// TIA Portal V20 export
// export: Created 2025-12-01T14:56:45.4401505Z, ExportSetting None, DisplayName Totally Integrated Automation Portal, DisplayVersion V20 Update 3, DisplayName TIA Portal Openness, DisplayVersion V20 Update 3, DisplayName TIA Portal Version Control Interface, DisplayVersion V20 Update 3, DisplayName STEP 7 Professional, DisplayVersion V20 Update 3, DisplayName STEP 7 Safety, DisplayVersion V20 Update 2, DisplayName WinCC Basic/Comfort/Advanced, DisplayVersion V20 Update 3, DisplayName WinCC Professional, DisplayVersion V20 Update 3, DisplayName WinCC Unified, DisplayVersion V20 Update 3
FUNCTION_BLOCK "FB262_M_FSS_Descarga"   // FB262, LAD
TITLE = Control del Ramal de Salidas
{ S7_Optimized_Access := 'FALSE' }
AUTHOR : TE_FSS
NAME : 20160509
VERSION : 3.3
// stored: AutoNumber false, SetENOAutomatically false
   VAR_INPUT
      Mesa : UInt;   // Mesa de la FB
      Error_Tx : Bool;   // Error en el Tx
      EnTension : Bool;   // Existe Tension en la Mesa
      Termico_T1 : Bool;   // Proteccion del T1
      Termico_T2 : Bool;   // Proteccion del T2
      Termico_T3 : Bool;   // Proteccion del T3
      Termico_T4 : Bool;   // Proteccion del T4
      pHsMx_1 : Bool;   // pHs 1 de la Mesa
      pHsMx_2 : Bool;   // pHs 2 de la Mesa
      pHsMx_3 : Bool;   // pHs 3 de la Mesa
      pHsMx_4 : Bool;   // pHs 4 de la Mesa
      Avance_T1 : Bool;   // Avance del T1
      Avance_T2 : Bool;   // Avance del T2
      Avance_T3 : Bool;   // Avance del T3
      Avance_T4 : Bool;   // Avance del T4
      Termico_TR1 : Bool;   // Proteccion del TR1
      Termico_TR2 : Bool;   // Proteccion del TR1
      Avance_TR1 : Bool;   // Avance del TR1
      Avance_TR2 : Bool;   // Avance del TR2
      TR1_Arriba : Bool;   // TR1 >> Arriba
      TR1_Abajo : Bool;   // TR1 >> Abajo
      TR1_EnMovimiento : Bool;   // TR1 >> En Movimiento
      TR2_Arriba : Bool;   // TR2 >> Arriba
      TR2_Abajo : Bool;   // TR2 >> Abajo
      TR2_EnMovimiento : Bool;   // TR2 >> En Movimiento
      TPE1_Arriba : Bool;   // TPE1 >> Arriba
      TPE1_Abajo : Bool;   // TPE1 >> Abajo
      TPE1_EnMovimiento : Bool;   // TPE1 >> En Movimiento
      TPE3_Arriba : Bool;   // TPE3 >> Arriba
      TPE3_Abajo : Bool;   // TPE3 >> Abajo
      TPE3_EnMovimiento : Bool;   // TPE3 >> En Movimiento
      MAnt_DescargaAct : Bool;   // E2 >> Mesa Anterior DescargaAct
      AVTF_MAnt_Mx_BGrande : Bool;   // E2 >> Mesa Anterior AVTF - Grande
      AVTF_MAnt_Mx_BPequena : Bool;   // E2 >> Mesa Anterior AVTF - Pequeña
      P_Mens_MAnt_Mx : Bool;   // E2 >> Mesa Anterior P_Mens
      E1_Arrival : Bool;   // E1 a FSS >> Arrival
      E1_Rotative : Bool;   // E1 a FSS >> Rotative
      E3_Arrival : Bool;   // E3 a FSS >> Arrival
      E3_Rotative : Bool;   // E3 a FSS >> Rotative
      PTF_Mx_MSig : Bool;   // S4 >> Mesa Siguiente PTF
      FTF_Mx_MSig : Bool;   // S4 >> Mesa Siguiente FTF
      MSig_CargaAct : Bool;
      F_EnvMens_Mx : Bool;   // Fin de Envio de Mensaje
      OrdSal_BGrande : Bool;   // Orden de Salida - Grande
      OrdSal_BPequena : Bool;   // Orden de Salida - Pequeña
      V_CNT_DesCargaFSS : Int := 1000;   // Valor de Posicionado FSS en la DesCarga
      V_CNT_PasarLentaFSS : Int := 100;
      V_CNT_pHsMx_E2 : Int := 100;   // Valor de Presencia
      V_CNT_pHsMx_FTF_E2 : Int := 250;   // Valor para activar FTF. Nota: < = V_CNT_pHsMx.
      V_CNTSeg_pHsMx_E2 : Int := 1000;   // Valor de Seguriadad para Presencia
      V_CNT_ApHsMx : Int := 200;   // Valor de Ausencia
      V_CNTSeg_ApHsMx : Int := 2000;   // Valor de Seguriadad para Ausencia
      V_CNT_Simultaneo : Int := 2000;   // Valor de Contador de Simultaneo
      V_TOut_Tx_Mx : Int := 7000;   // TImeOut de DesCarga del FSS
      V_TOut_TRx_Mx : Int := 7000;   // TimeOut de Entrada por E2
      V_TOut_TR : Int := 3000;   // TimeOut de Transfer
      V_TOut_TP : Int := 3000;   // TimeOut de Tope
      V_TOut_Interlock : Int := 5000;   // TimeOut de Interlock con el FSS
      V_CNT_PerdidapHs : Int := 1000;   // CNT de Perdida de pHs
      V_TIM_EstabilidadCarga : Time := T#100MS;   // Valor de Eastabilidad de Carga por DCC
      V_TIM_EsperaMesaLibre : Time;   // Valor de Espera para dar Mesa Libre
   END_VAR
   VAR_OUTPUT
      P_EnvMens_PMx : Bool;   // Permiso de Enviar Mensaje de Presencia
      P_RecepOK_Mx : Bool;   // Recepcion OK
      PTF_MAnt_Mx : Bool;   // E2 >> Mesa Anterior PTF
      FTF_MAnt_Mx : Bool;   // E2 >> Mesa Anterior FTF
      AVTF_Mx_Msig_BGrande : Bool;   // S4 >> Mesa Siguiente AVTF - Grande
      AVTF_Mx_MSig_BPequena : Bool;   // S4 >> Mesa Siguiente AVTF - Pequeña
      P_Mens_Mx_MSig : Bool;   // S4 >> Mesa Siguiente P_Mens
   END_VAR
   VAR
      Mx_ET00 : Bool;
      Mx_ET01 : Bool;
      Mx_ET02 : Bool;
      Mx_ET08_1PRE : Bool;
      Mx_ET08_1FIN : Bool;
      Mx_ET08_2PRE : Bool;
      Mx_ET08_2FIN : Bool;
      Mx_ET08_3PRE : Bool;
      Mx_ET08_3FIN : Bool;
      Mx_ET08_4PRE : Bool;
      Mx_ET08_4FIN : Bool;
      Mx_ET09 : Bool;
      Mx_ET10 : Bool;
      Mx_ET11 : Bool;
      Mx_ET12 : Bool;
      Mx_ET110_1PRE : Bool;
      Mx_ET110_1FIN : Bool;
      Mx_ET110_2PRE : Bool;
      Mx_ET110_2FIN : Bool;
      Mx_ET110_3PRE : Bool;
      Mx_ET110_3FIN : Bool;
      Mx_ET110_4PRE : Bool;
      Mx_ET110_4FIN : Bool;
      Mx_ET111 : Bool;
      Mx_ET20 : Bool;
      Mx_ET21 : Bool;
      Mx_ET22 : Bool;
      Mx_ET120 : Bool;
      Mx_ET121 : Bool;
      Mx_ET30 : Bool;
      Mx_ET31 : Bool;
      Mx_ET32 : Bool;
      Mx_ET130_1PRE : Bool;
      Mx_ET130_1FIN : Bool;
      Mx_ET130_2PRE : Bool;
      Mx_ET130_2FIN : Bool;
      Mx_ET130_3PRE : Bool;
      Mx_ET130_3FIN : Bool;
      Mx_ET130_4PRE : Bool;
      Mx_ET130_4FIN : Bool;
      Mx_ET131 : Bool;
      Mx_ET60 : Bool;
      Mx_ET61 : Bool;
      Mx_ET160 : Bool;
      Mx_ET161 : Bool;
      Mx_AutoArranque : Bool;   // Config >> Fin carga del FSS - Automatico
      Mx_NoEnvioPresEnFSS : Bool;   // Config >> No Envio de Presncia en la DesCarga del FSS
      FinDesCargaFSS_Auto : Bool;   // Intena >> AutoRearme Fin DesCarga del FSS
      Selec_E1 : Bool;   // Interna >> Selecionado Entrada por E1
      Selec_E2 : Bool;   // Interna >> Selecionado Entrada por E2
      Selec_E3 : Bool;   // Interna >> Selecionado Entrada por E3
      Selec_S4_BGrande : Bool;   // Interna >> Selecionado Salida por S4 - Grande
      Selec_S4_BPequena : Bool;   // Interna >> Selecionado Salida por S4 - Pequeña
      SaliendoCarga : Bool;   // Saliendo Carga de la Mesa
      Pos_TROK : Bool;   // Interna >> Posicion Correcta de los TRs
      Pos_TPOK : Bool;   // Interna >> Posicion Correcta de los TPs
      Entrando_BGrande : Bool;   // Interna >> Bandeja Grande en Entrada por E2
      PasarLenta_FSS : Bool;   // Interna >> Orden Pasar a Lenta la DesCarga FSS
      PosSalidaCarga_OK : Bool;   // Interna >> Posicionada la Carga para Salida
      ProtocoloIniciado : Bool;   // Iniciado el Envio del Mensaje de Presencia
      CNT_pHsMx_FTF_E2_OK : Bool;   // Enviar ya FTF
      Simultaneo_Mx : Bool;   // Activo Simultaneo E2
      STAT_EnvMens_PMx : Bool;   // Interna >> Envio del Mensaje de Presencia
      STAT_AVTF_MAnt_Mx : Bool;   // Interna >> Aviso de Entrada - Grande, Pequeña
      STAT_FTF_MAnt_Mx : Bool;   // Interna >> FTF de MAnt >> Mx
      STAT_AVTF_Mx_MSig : Bool;   // Interna >> AVTF de Mx >> MSig
      STAT_AvanceCarga_E1E3 : Bool;   // Interna >> Avance de Entrada de Carga por E1E3
      STAT_AvanceCarga_E2 : Bool;   // Interna >> Avance de Entrada de Carga por E2
      STAT_AvanceDescarga : Bool;   // Interna >> Avance de Salida de Carga
      STAT_Velocidad_TxBO : Bool;   // Interna >> Velocidad Bit 0 de los Rodillos
      STAT_Velocidad_TxB1 : Bool;   // Interna >> Velocidad Bit 1 de los Rodillos
      MA_Avance_T1 : Bool;
      MA_Avance_T2 : Bool;
      MA_Avance_T3 : Bool;
      MA_Avance_T4 : Bool;
      MA_Inversion_Tx : Bool;
      MA_VelocidadAnalogica : Int;
      MA_Avance_TR1 : Bool;
      MA_Avance_TR2 : Bool;
      MA_VelocidaLenta_TRx : Bool;
      MA_Subir_TR1 : Bool;
      MA_Bajar_TR1 : Bool;
      MA_Subir_TR2 : Bool;
      MA_Bajar_TR2 : Bool;
      MA_Subir_TPE1 : Bool;
      MA_Bajar_TPE1 : Bool;
      MA_Subir_TPE3 : Bool;
      MA_Bajar_TPE3 : Bool;
      MA_DepositOK_E1 : Bool;
      MA_Complete_E1 : Bool;
      MA_DepositOK_E3 : Bool;
      MA_Complete_E3 : Bool;
      TIM_EsperaMesaLibre { S7_SetPoint := 'True'} : TON_TIME;   // TIM De Espera para Dar la Mesa como Libre
      TIM_Estabilidad_E1 { S7_SetPoint := 'True'} : TON_TIME;   // TIM De Estabilidad de Carga en E1
      TIM_Estabilidad_E3 { S7_SetPoint := 'True'} : TON_TIME;   // TIM De Estabilidad de Carga en E3
      TIM_Estabilidad_E2 { S7_SetPoint := 'True'} : TON_TIME;   // TIM De Estabilidad de Carga en E2
      TIM_EstabilidadCarga { S7_SetPoint := 'True'} : TON_TIME;
      CNT_pHsMx_E1 { S7_SetPoint := 'True'} : "FB910_CNT_UHS";   // CNT de Presencia de FSS por E1
      CNT_pHsMx_E3 { S7_SetPoint := 'True'} : "FB910_CNT_UHS";   // CNT de Presencia de FSS por E3
      CNT_Reposiciona_E3 { S7_SetPoint := 'True'} : "FB910_CNT_UHS";   // CNT de Reposicionado de FSS por E3
      CNT_PasarLenta_FSS { S7_SetPoint := 'True'} : "FB910_CNT_UHS";   // CNT de Pasar a Lenta la DesCarga del FSS
      CNT_RecolocarCarga { S7_SetPoint := 'True'} : "FB910_CNT_UHS";   // CNT de Recolocar la Carga para la Salida
      CNT_pHsMx_E2 { S7_SetPoint := 'True'} : "FB910_CNT_UHS";   // CNT de la Presencia
      CNTSeg_pHsMx_E2 { S7_SetPoint := 'True'} : "FB910_CNT_UHS";   // CNT de Seguridad de la Presencia
      CNT_ApHsMx { S7_SetPoint := 'True'} : "FB910_CNT_UHS";   // CNT de la Ausencia
      CNTSeg_ApHsMx { S7_SetPoint := 'True'} : "FB910_CNT_UHS";   // CNT de Seguridad de la Ausencia
      CNT_Simultaneo { S7_SetPoint := 'True'} : "FB910_CNT_UHS";   // CNT de Simultaneo
      TMP_EnTension { S7_SetPoint := 'True'} : "FB910_CNT_UHS";
      TOut_Av_Tx { S7_SetPoint := 'True'} : "FB910_CNT_UHS";   // Time Out de Entrada de E1
      TOut_Rt_Tx { S7_SetPoint := 'True'} : "FB910_CNT_UHS";   // Time Out de Entrada de E3
      TOut_Av_TRx { S7_SetPoint := 'True'} : "FB910_CNT_UHS";   // Time Out de Entrada de E2
      TOut_Subir_TR { S7_SetPoint := 'True'} : "FB910_CNT_UHS";   // Time Out de Subida del TR
      TOut_Bajar_TR { S7_SetPoint := 'True'} : "FB910_CNT_UHS";   // Time Out de Bajada del TR
      TOut_Subir_TP_E1E3 { S7_SetPoint := 'True'} : "FB910_CNT_UHS";   // Time Out de Subida del TP >> E1E3
      TOut_Bajar_TP_E1E3 { S7_SetPoint := 'True'} : "FB910_CNT_UHS";   // Time Out de Bajada del TP >> E1E3
      TOut_Interlock { S7_SetPoint := 'True'} : "FB910_CNT_UHS";   // Time Out de Interlock con el FSS
      Interlock_manual { S7_SetPoint := 'True'} : "UDT_Interlock_manual_TE_FSS";
      Manual : "MoviManualMesa_FSS";
      CNT_PerdidapHs { S7_SetPoint := 'True'} : "FB910_CNT_UHS";   // CNT de Perdida de pHs
   END_VAR
   VAR_TEMP
      EstadoZona : "EstadoZona";   // Estado de Zona de la Mesa
      EstadoVI : "EstadosMesa_FSS";   // Estado del Vehiculo Inteliguente de la Mesa
      ConfigFB : "UDT_ConfigFB";   // Configuracion de la FB de la Mesa
      Interlock : "UDT_Interlock_TE_FSS";
      retval : Int;
      cero : USInt;
      Aux_ET00 : Bool;
      EvolucionEtapasEntrada : Bool;
      EvolucionEtapasSalida : Bool;
   END_VAR
   VAR_TEMP   // added for the SCL form of the ladder/FBD networks
      _w1 : Bool;
   END_VAR
BEGIN

REGION Network 1: CONFIGURACION ESPECIAL DE LA FB
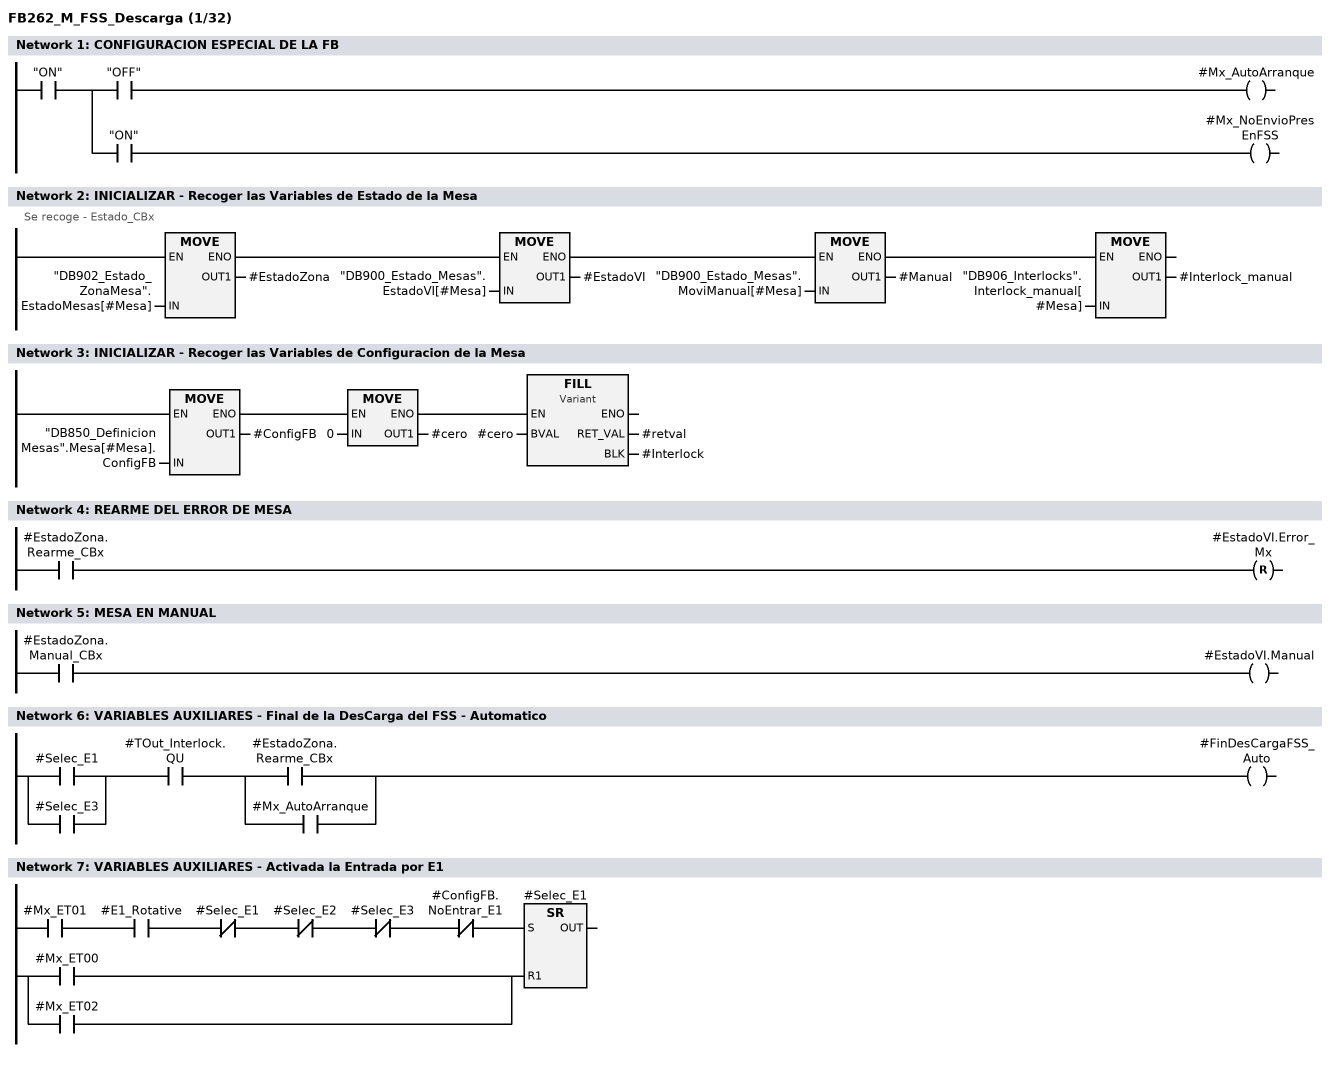
   RUNG wire#powerrail
      Contact( "ON" )
      wire#w1
      Contact( "OFF" )
      Coil( #Mx_AutoArranque )
   END_RUNG
   RUNG wire#w1
      Contact( "ON" )
      Coil( #Mx_NoEnvioPresEnFSS )
   END_RUNG
   // the same network as SCL:
   #Mx_AutoArranque := "ON" AND "OFF";
   #Mx_NoEnvioPresEnFSS := "ON" AND "ON";
END_REGION

REGION Network 2: INICIALIZAR - Recoger las Variables de Estado de la Mesa
   // Se recoge - Estado_CBx
   RUNG wire#powerrail
      Move(in := "DB902_Estado_ZonaMesa".EstadoMesas[#Mesa], out1 => #EstadoZona)
      Move(in := "DB900_Estado_Mesas".EstadoVI[#Mesa], out1 => #EstadoVI)
      Move(in := "DB900_Estado_Mesas".MoviManual[#Mesa], out1 => #Manual)
      Move(in := "DB906_Interlocks".Interlock_manual[#Mesa], out1 => #Interlock_manual)
   END_RUNG
   // the same network as SCL:
   #EstadoZona := "DB902_Estado_ZonaMesa".EstadoMesas[#Mesa];
   #EstadoVI := "DB900_Estado_Mesas".EstadoVI[#Mesa];
   #Manual := "DB900_Estado_Mesas".MoviManual[#Mesa];
   #Interlock_manual := "DB906_Interlocks".Interlock_manual[#Mesa];
END_REGION

REGION Network 3: INICIALIZAR - Recoger las Variables de Configuracion de la Mesa
   RUNG wire#powerrail
      Move(in := "DB850_DefinicionMesas".Mesa[#Mesa].ConfigFB, out1 => #ConfigFB)
      Move(in := 0, out1 => #cero)
      { S7_Templates := "ptr_type := Variant" } FILL(BVAL := #cero, RET_VAL => #retval, BLK => #Interlock)
   END_RUNG
   // the same network as SCL:
   #ConfigFB := "DB850_DefinicionMesas".Mesa[#Mesa].ConfigFB;
   #cero := 0;
   #retval := FILL(BVAL := #cero, BLK => #Interlock);
END_REGION

REGION Network 4: REARME DEL ERROR DE MESA
   RUNG wire#powerrail
      Contact( #EstadoZona.Rearme_CBx )
      R_Coil( #EstadoVI.Error_Mx )
   END_RUNG
   // the same network as SCL:
   IF #EstadoZona.Rearme_CBx THEN #EstadoVI.Error_Mx := FALSE; END_IF;
END_REGION

REGION Network 5: MESA EN MANUAL
   RUNG wire#powerrail
      Contact( #EstadoZona.Manual_CBx )
      Coil( #EstadoVI.Manual )
   END_RUNG
   // the same network as SCL:
   #EstadoVI.Manual := #EstadoZona.Manual_CBx;
END_REGION

REGION Network 6: VARIABLES AUXILIARES - Final de la DesCarga del FSS - Automatico
   RUNG wire#powerrail
      Contact( #Selec_E1 )
      wire#w1
      Contact( #TOut_Interlock.QU )
      wire#w2
      Contact( #EstadoZona.Rearme_CBx )
      wire#w3
      Coil( #FinDesCargaFSS_Auto )
   END_RUNG
   RUNG wire#powerrail
      Contact( #Selec_E3 )
   END_RUNG wire#w1
   RUNG wire#w2
      Contact( #Mx_AutoArranque )
   END_RUNG wire#w3
   // the same network as SCL:
   #FinDesCargaFSS_Auto := (#Selec_E1 OR #Selec_E3) AND #TOut_Interlock.QU AND (#EstadoZona.Rearme_CBx OR #Mx_AutoArranque);
END_REGION

REGION Network 7: VARIABLES AUXILIARES - Activada la Entrada por E1
   RUNG wire#powerrail
      Contact( #Mx_ET01 )
      Contact( #E1_Rotative )
      I_Contact( #Selec_E1 )
      I_Contact( #Selec_E2 )
      I_Contact( #Selec_E3 )
      I_Contact( #ConfigFB.NoEntrar_E1 )
      S_SR(operand := #Selec_E1, r1 := wire#w1)
   END_RUNG
   RUNG wire#powerrail
      Contact( #Mx_ET00 )
   END_RUNG wire#w1
   RUNG wire#powerrail
      Contact( #Mx_ET02 )
   END_RUNG wire#w1
   // the same network as SCL:
   IF #Mx_ET01 AND #E1_Rotative AND NOT #Selec_E1 AND NOT #Selec_E2 AND NOT #Selec_E3 AND NOT #ConfigFB.NoEntrar_E1 THEN
       #Selec_E1 := TRUE;   // SR flip-flop
   END_IF;
   IF #Mx_ET00 OR #Mx_ET02 THEN #Selec_E1 := FALSE; END_IF;
END_REGION

REGION Network 8: VARIABLES AUXILIARES - Activada la Entrada por E2
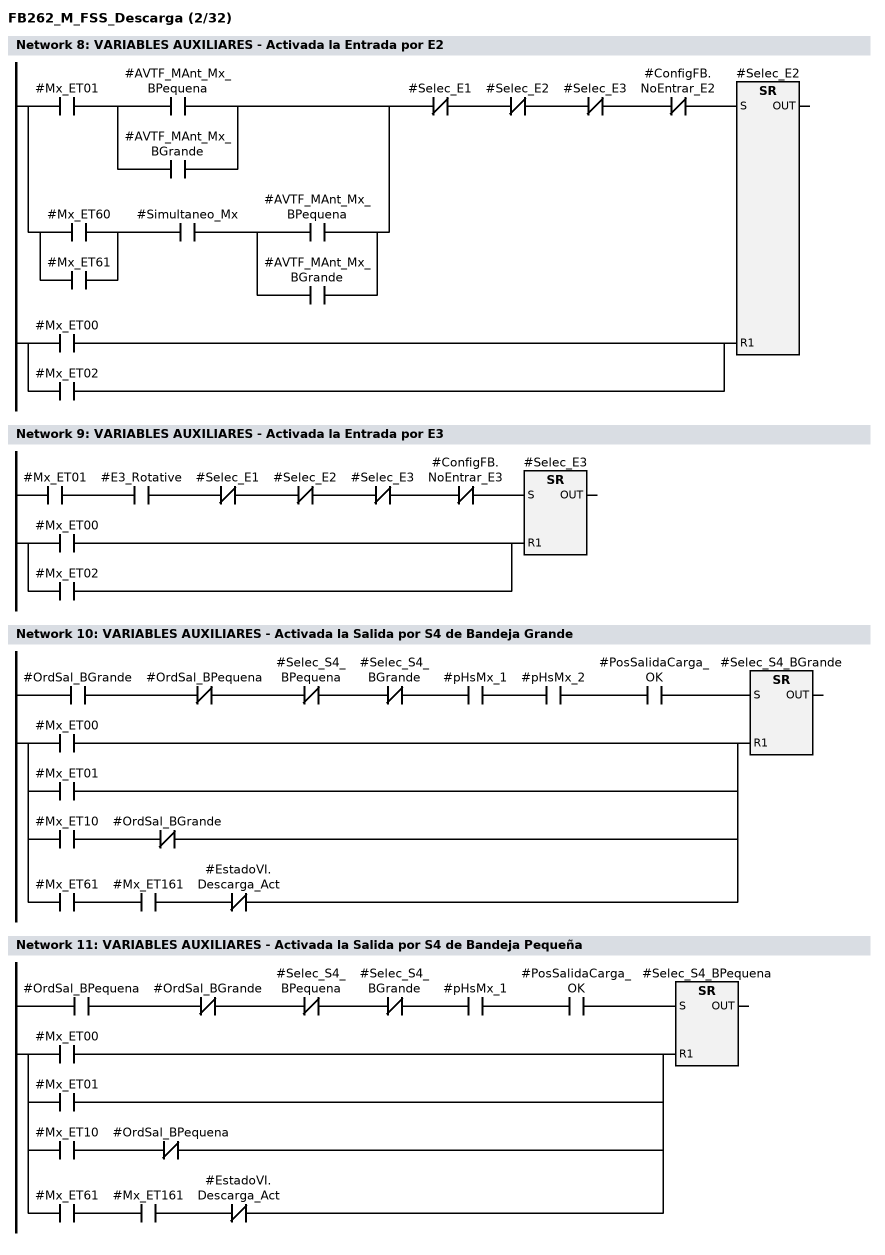
   RUNG wire#powerrail
      Contact( #Mx_ET01 )
      wire#w1
      Contact( #AVTF_MAnt_Mx_BPequena )
      wire#w2
      I_Contact( #Selec_E1 )
      I_Contact( #Selec_E2 )
      I_Contact( #Selec_E3 )
      I_Contact( #ConfigFB.NoEntrar_E2 )
      S_SR(operand := #Selec_E2, r1 := wire#w5)
   END_RUNG
   RUNG wire#w1
      Contact( #AVTF_MAnt_Mx_BGrande )
   END_RUNG wire#w2
   RUNG wire#powerrail
      Contact( #Mx_ET60 )
      wire#w3
      Contact( #Simultaneo_Mx )
      wire#w4
      Contact( #AVTF_MAnt_Mx_BPequena )
   END_RUNG wire#w2
   RUNG wire#powerrail
      Contact( #Mx_ET61 )
   END_RUNG wire#w3
   RUNG wire#w4
      Contact( #AVTF_MAnt_Mx_BGrande )
   END_RUNG wire#w2
   RUNG wire#powerrail
      Contact( #Mx_ET00 )
   END_RUNG wire#w5
   RUNG wire#powerrail
      Contact( #Mx_ET02 )
   END_RUNG wire#w5
   // the same network as SCL:
   IF ((#Mx_ET01 AND (#AVTF_MAnt_Mx_BPequena OR #AVTF_MAnt_Mx_BGrande)) OR ((#Mx_ET60 OR #Mx_ET61) AND #Simultaneo_Mx AND (#AVTF_MAnt_Mx_BPequena OR #AVTF_MAnt_Mx_BGrande))) AND NOT #Selec_E1 AND NOT #Selec_E2 AND NOT #Selec_E3 AND NOT #ConfigFB.NoEntrar_E2 THEN
       #Selec_E2 := TRUE;   // SR flip-flop
   END_IF;
   IF #Mx_ET00 OR #Mx_ET02 THEN #Selec_E2 := FALSE; END_IF;
END_REGION

REGION Network 9: VARIABLES AUXILIARES - Activada la Entrada por E3
   RUNG wire#powerrail
      Contact( #Mx_ET01 )
      Contact( #E3_Rotative )
      I_Contact( #Selec_E1 )
      I_Contact( #Selec_E2 )
      I_Contact( #Selec_E3 )
      I_Contact( #ConfigFB.NoEntrar_E3 )
      S_SR(operand := #Selec_E3, r1 := wire#w1)
   END_RUNG
   RUNG wire#powerrail
      Contact( #Mx_ET00 )
   END_RUNG wire#w1
   RUNG wire#powerrail
      Contact( #Mx_ET02 )
   END_RUNG wire#w1
   // the same network as SCL:
   IF #Mx_ET01 AND #E3_Rotative AND NOT #Selec_E1 AND NOT #Selec_E2 AND NOT #Selec_E3 AND NOT #ConfigFB.NoEntrar_E3 THEN
       #Selec_E3 := TRUE;   // SR flip-flop
   END_IF;
   IF #Mx_ET00 OR #Mx_ET02 THEN #Selec_E3 := FALSE; END_IF;
END_REGION

REGION Network 10: VARIABLES AUXILIARES - Activada la Salida por S4 de Bandeja Grande
   RUNG wire#powerrail
      Contact( #OrdSal_BGrande )
      I_Contact( #OrdSal_BPequena )
      I_Contact( #Selec_S4_BPequena )
      I_Contact( #Selec_S4_BGrande )
      Contact( #pHsMx_1 )
      Contact( #pHsMx_2 )
      Contact( #PosSalidaCarga_OK )
      S_SR(operand := #Selec_S4_BGrande, r1 := wire#w1)
   END_RUNG
   RUNG wire#powerrail
      Contact( #Mx_ET00 )
   END_RUNG wire#w1
   RUNG wire#powerrail
      Contact( #Mx_ET01 )
   END_RUNG wire#w1
   RUNG wire#powerrail
      Contact( #Mx_ET10 )
      I_Contact( #OrdSal_BGrande )
   END_RUNG wire#w1
   RUNG wire#powerrail
      Contact( #Mx_ET61 )
      Contact( #Mx_ET161 )
      I_Contact( #EstadoVI.Descarga_Act )
   END_RUNG wire#w1
   // the same network as SCL:
   IF #OrdSal_BGrande AND NOT #OrdSal_BPequena AND NOT #Selec_S4_BPequena AND NOT #Selec_S4_BGrande AND #pHsMx_1 AND #pHsMx_2 AND #PosSalidaCarga_OK THEN
       #Selec_S4_BGrande := TRUE;   // SR flip-flop
   END_IF;
   IF #Mx_ET00 OR #Mx_ET01 OR (#Mx_ET10 AND NOT #OrdSal_BGrande) OR (#Mx_ET61 AND #Mx_ET161 AND NOT #EstadoVI.Descarga_Act) THEN
       #Selec_S4_BGrande := FALSE;
   END_IF;
END_REGION

REGION Network 11: VARIABLES AUXILIARES - Activada la Salida por S4 de Bandeja Pequeña
   RUNG wire#powerrail
      Contact( #OrdSal_BPequena )
      I_Contact( #OrdSal_BGrande )
      I_Contact( #Selec_S4_BPequena )
      I_Contact( #Selec_S4_BGrande )
      Contact( #pHsMx_1 )
      Contact( #PosSalidaCarga_OK )
      S_SR(operand := #Selec_S4_BPequena, r1 := wire#w1)
   END_RUNG
   RUNG wire#powerrail
      Contact( #Mx_ET00 )
   END_RUNG wire#w1
   RUNG wire#powerrail
      Contact( #Mx_ET01 )
   END_RUNG wire#w1
   RUNG wire#powerrail
      Contact( #Mx_ET10 )
      I_Contact( #OrdSal_BPequena )
   END_RUNG wire#w1
   RUNG wire#powerrail
      Contact( #Mx_ET61 )
      Contact( #Mx_ET161 )
      I_Contact( #EstadoVI.Descarga_Act )
   END_RUNG wire#w1
   // the same network as SCL:
   IF #OrdSal_BPequena AND NOT #OrdSal_BGrande AND NOT #Selec_S4_BPequena AND NOT #Selec_S4_BGrande AND #pHsMx_1 AND #PosSalidaCarga_OK THEN
       #Selec_S4_BPequena := TRUE;   // SR flip-flop
   END_IF;
   IF #Mx_ET00 OR #Mx_ET01 OR (#Mx_ET10 AND NOT #OrdSal_BPequena) OR (#Mx_ET61 AND #Mx_ET161 AND NOT #EstadoVI.Descarga_Act) THEN
       #Selec_S4_BPequena := FALSE;
   END_IF;
END_REGION

REGION Network 12: VARIABLES AUXILIARES - Saliendo Carga de la Mesa
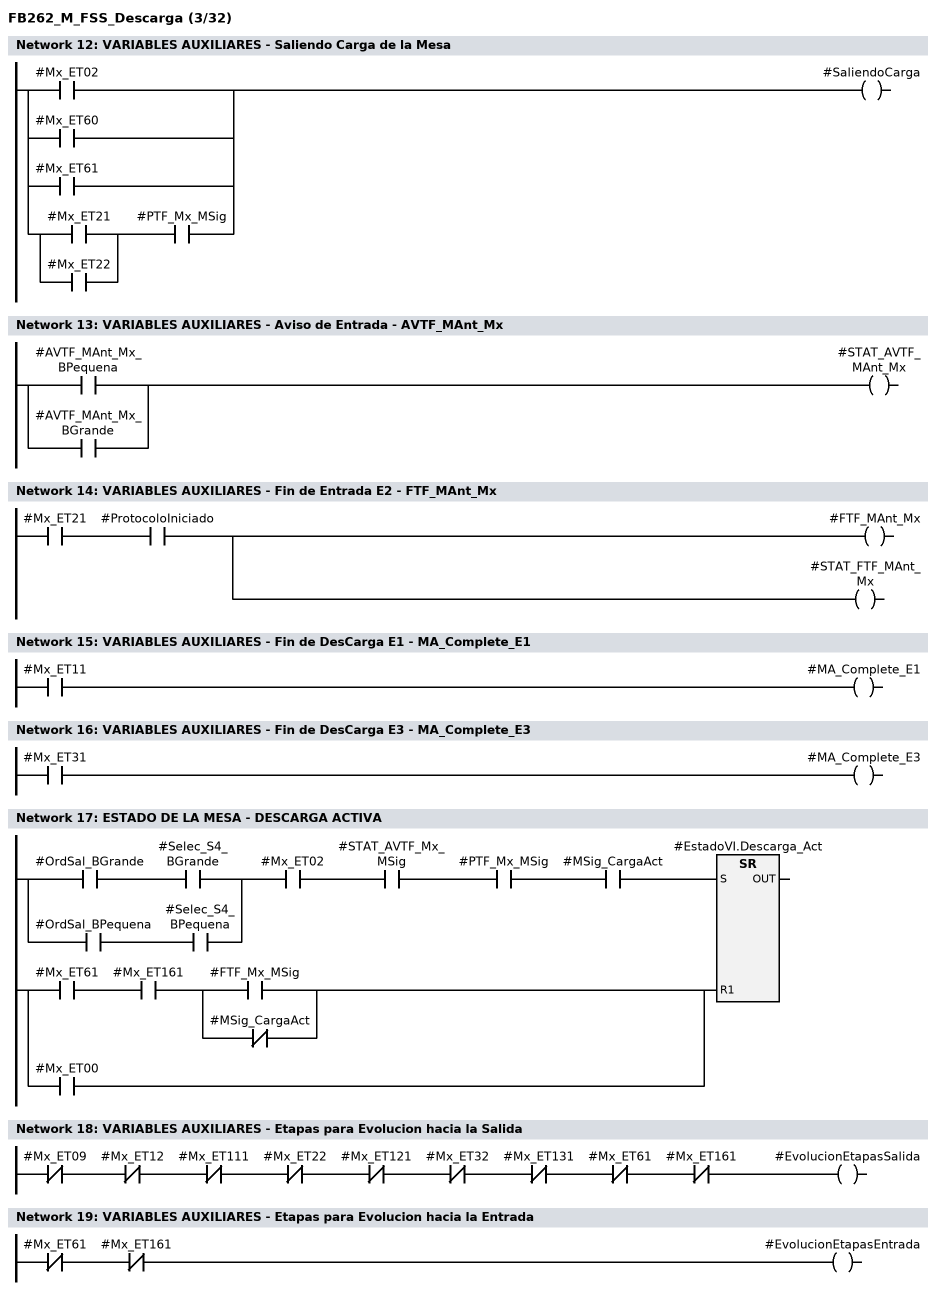
   RUNG wire#powerrail
      Contact( #Mx_ET02 )
      wire#w1
      Coil( #SaliendoCarga )
   END_RUNG
   RUNG wire#powerrail
      Contact( #Mx_ET60 )
   END_RUNG wire#w1
   RUNG wire#powerrail
      Contact( #Mx_ET61 )
   END_RUNG wire#w1
   RUNG wire#powerrail
      Contact( #Mx_ET21 )
      wire#w2
      Contact( #PTF_Mx_MSig )
   END_RUNG wire#w1
   RUNG wire#powerrail
      Contact( #Mx_ET22 )
   END_RUNG wire#w2
   // the same network as SCL:
   #SaliendoCarga := #Mx_ET02 OR #Mx_ET60 OR #Mx_ET61 OR ((#Mx_ET21 OR #Mx_ET22) AND #PTF_Mx_MSig);
END_REGION

REGION Network 13: VARIABLES AUXILIARES - Aviso de Entrada - AVTF_MAnt_Mx
   RUNG wire#powerrail
      Contact( #AVTF_MAnt_Mx_BPequena )
      wire#w1
      Coil( #STAT_AVTF_MAnt_Mx )
   END_RUNG
   RUNG wire#powerrail
      Contact( #AVTF_MAnt_Mx_BGrande )
   END_RUNG wire#w1
   // the same network as SCL:
   #STAT_AVTF_MAnt_Mx := #AVTF_MAnt_Mx_BPequena OR #AVTF_MAnt_Mx_BGrande;
END_REGION

REGION Network 14: VARIABLES AUXILIARES - Fin de Entrada E2 - FTF_MAnt_Mx
   RUNG wire#powerrail
      Contact( #Mx_ET21 )
      Contact( #ProtocoloIniciado )
      wire#w1
      Coil( #FTF_MAnt_Mx )
   END_RUNG
   RUNG wire#w1
      Coil( #STAT_FTF_MAnt_Mx )
   END_RUNG
   // the same network as SCL:
   #FTF_MAnt_Mx := #Mx_ET21 AND #ProtocoloIniciado;
   #STAT_FTF_MAnt_Mx := #FTF_MAnt_Mx;
END_REGION

REGION Network 15: VARIABLES AUXILIARES - Fin de DesCarga E1 - MA_Complete_E1
   RUNG wire#powerrail
      Contact( #Mx_ET11 )
      Coil( #MA_Complete_E1 )
   END_RUNG
   // the same network as SCL:
   #MA_Complete_E1 := #Mx_ET11;
END_REGION

REGION Network 16: VARIABLES AUXILIARES - Fin de DesCarga E3 - MA_Complete_E3
   RUNG wire#powerrail
      Contact( #Mx_ET31 )
      Coil( #MA_Complete_E3 )
   END_RUNG
   // the same network as SCL:
   #MA_Complete_E3 := #Mx_ET31;
END_REGION

REGION Network 17: ESTADO DE LA MESA - DESCARGA ACTIVA
   RUNG wire#powerrail
      Contact( #OrdSal_BGrande )
      Contact( #Selec_S4_BGrande )
      wire#w1
      Contact( #Mx_ET02 )
      Contact( #STAT_AVTF_Mx_MSig )
      Contact( #PTF_Mx_MSig )
      Contact( #MSig_CargaAct )
      S_SR(operand := #EstadoVI.Descarga_Act, r1 := wire#w3)
   END_RUNG
   RUNG wire#powerrail
      Contact( #OrdSal_BPequena )
      Contact( #Selec_S4_BPequena )
   END_RUNG wire#w1
   RUNG wire#powerrail
      Contact( #Mx_ET61 )
      Contact( #Mx_ET161 )
      wire#w2
      Contact( #FTF_Mx_MSig )
   END_RUNG wire#w3
   RUNG wire#w2
      I_Contact( #MSig_CargaAct )
   END_RUNG wire#w3
   RUNG wire#powerrail
      Contact( #Mx_ET00 )
   END_RUNG wire#w3
   // the same network as SCL:
   IF ((#OrdSal_BGrande AND #Selec_S4_BGrande) OR (#OrdSal_BPequena AND #Selec_S4_BPequena)) AND #Mx_ET02 AND #STAT_AVTF_Mx_MSig AND #PTF_Mx_MSig AND #MSig_CargaAct THEN
       #EstadoVI.Descarga_Act := TRUE;   // SR flip-flop
   END_IF;
   IF (#Mx_ET61 AND #Mx_ET161 AND (#FTF_Mx_MSig OR NOT #MSig_CargaAct)) OR #Mx_ET00 THEN
       #EstadoVI.Descarga_Act := FALSE;
   END_IF;
END_REGION

REGION Network 18: VARIABLES AUXILIARES - Etapas para Evolucion hacia la Salida
   RUNG wire#powerrail
      I_Contact( #Mx_ET09 )
      I_Contact( #Mx_ET12 )
      I_Contact( #Mx_ET111 )
      I_Contact( #Mx_ET22 )
      I_Contact( #Mx_ET121 )
      I_Contact( #Mx_ET32 )
      I_Contact( #Mx_ET131 )
      I_Contact( #Mx_ET61 )
      I_Contact( #Mx_ET161 )
      Coil( #EvolucionEtapasSalida )
   END_RUNG
   // the same network as SCL:
   #EvolucionEtapasSalida := NOT #Mx_ET09 AND NOT #Mx_ET12 AND NOT #Mx_ET111 AND NOT #Mx_ET22 AND NOT #Mx_ET121 AND NOT #Mx_ET32 AND NOT #Mx_ET131 AND NOT #Mx_ET61 AND NOT #Mx_ET161;
END_REGION

REGION Network 19: VARIABLES AUXILIARES - Etapas para Evolucion hacia la Entrada
   RUNG wire#powerrail
      I_Contact( #Mx_ET61 )
      I_Contact( #Mx_ET161 )
      Coil( #EvolucionEtapasEntrada )
   END_RUNG
   // the same network as SCL:
   #EvolucionEtapasEntrada := NOT #Mx_ET61 AND NOT #Mx_ET161;
END_REGION

REGION Network 20: ET161 - CONTROL DESCARGA MESA - PROTOCOLO ORDEN
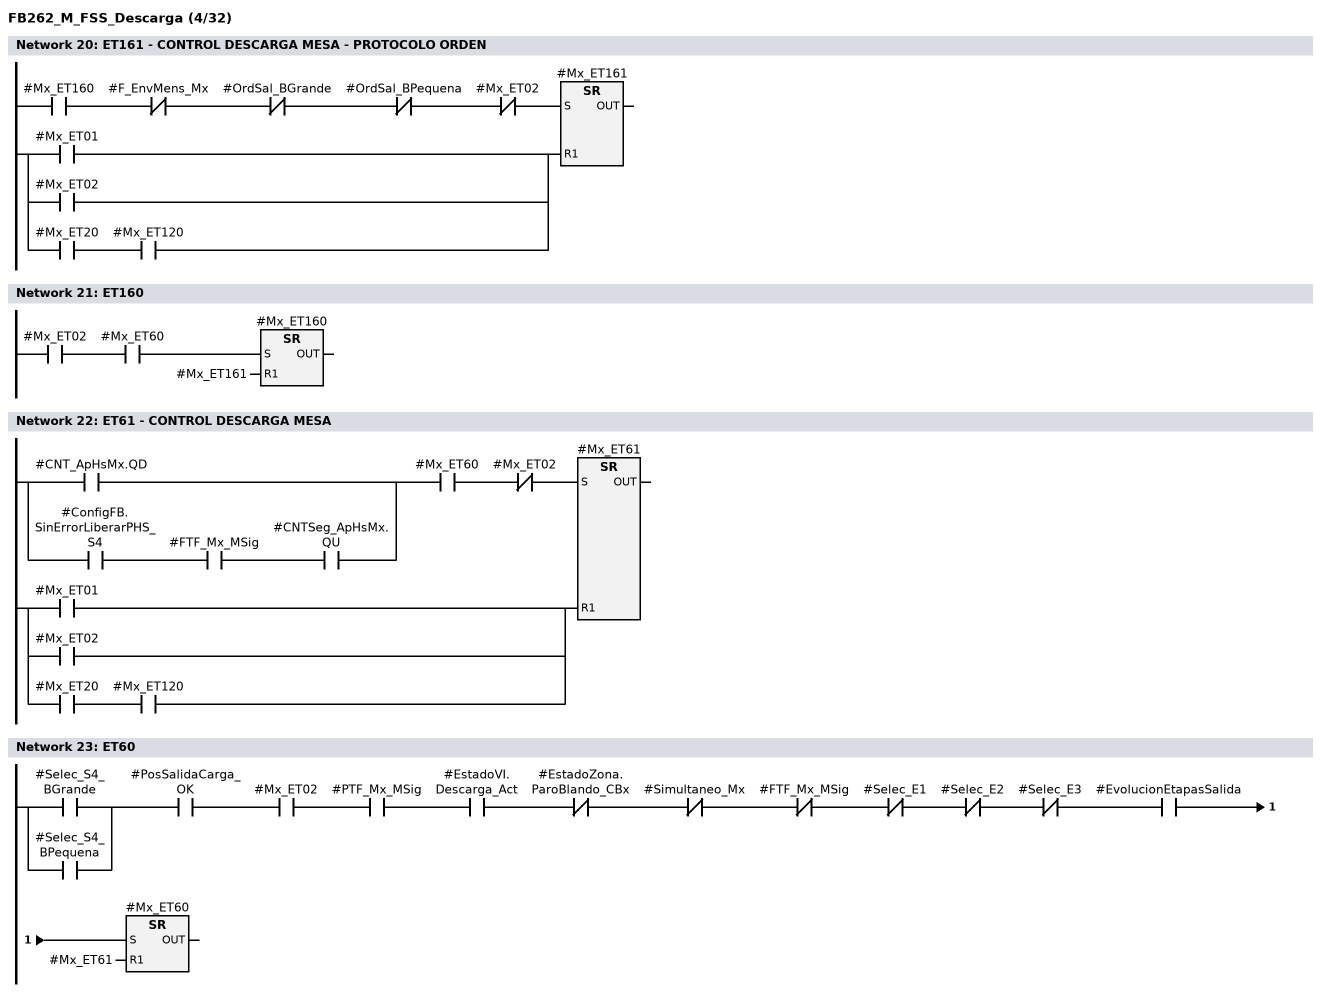
   RUNG wire#powerrail
      Contact( #Mx_ET160 )
      I_Contact( #F_EnvMens_Mx )
      I_Contact( #OrdSal_BGrande )
      I_Contact( #OrdSal_BPequena )
      I_Contact( #Mx_ET02 )
      S_SR(operand := #Mx_ET161, r1 := wire#w1)
   END_RUNG
   RUNG wire#powerrail
      Contact( #Mx_ET01 )
   END_RUNG wire#w1
   RUNG wire#powerrail
      Contact( #Mx_ET02 )
   END_RUNG wire#w1
   RUNG wire#powerrail
      Contact( #Mx_ET20 )
      Contact( #Mx_ET120 )
   END_RUNG wire#w1
   // the same network as SCL:
   IF #Mx_ET160 AND NOT #F_EnvMens_Mx AND NOT #OrdSal_BGrande AND NOT #OrdSal_BPequena AND NOT #Mx_ET02 THEN
       #Mx_ET161 := TRUE;   // SR flip-flop
   END_IF;
   IF #Mx_ET01 OR #Mx_ET02 OR (#Mx_ET20 AND #Mx_ET120) THEN #Mx_ET161 := FALSE; END_IF;
END_REGION

REGION Network 21: ET160
   RUNG wire#powerrail
      Contact( #Mx_ET02 )
      Contact( #Mx_ET60 )
      S_SR(operand := #Mx_ET160, r1 := #Mx_ET161)
   END_RUNG
   // the same network as SCL:
   IF #Mx_ET02 AND #Mx_ET60 THEN
       #Mx_ET160 := TRUE;   // SR flip-flop
   END_IF;
   IF #Mx_ET161 THEN #Mx_ET160 := FALSE; END_IF;
END_REGION

REGION Network 22: ET61 - CONTROL DESCARGA MESA
   RUNG wire#powerrail
      Contact( #CNT_ApHsMx.QD )
      wire#w1
      Contact( #Mx_ET60 )
      I_Contact( #Mx_ET02 )
      S_SR(operand := #Mx_ET61, r1 := wire#w2)
   END_RUNG
   RUNG wire#powerrail
      Contact( #ConfigFB.SinErrorLiberarPHS_S4 )
      Contact( #FTF_Mx_MSig )
      Contact( #CNTSeg_ApHsMx.QU )
   END_RUNG wire#w1
   RUNG wire#powerrail
      Contact( #Mx_ET01 )
   END_RUNG wire#w2
   RUNG wire#powerrail
      Contact( #Mx_ET02 )
   END_RUNG wire#w2
   RUNG wire#powerrail
      Contact( #Mx_ET20 )
      Contact( #Mx_ET120 )
   END_RUNG wire#w2
   // the same network as SCL:
   IF (#CNT_ApHsMx.QD OR (#ConfigFB.SinErrorLiberarPHS_S4 AND #FTF_Mx_MSig AND #CNTSeg_ApHsMx.QU)) AND #Mx_ET60 AND NOT #Mx_ET02 THEN
       #Mx_ET61 := TRUE;   // SR flip-flop
   END_IF;
   IF #Mx_ET01 OR #Mx_ET02 OR (#Mx_ET20 AND #Mx_ET120) THEN #Mx_ET61 := FALSE; END_IF;
END_REGION

REGION Network 23: ET60
   RUNG wire#powerrail
      Contact( #Selec_S4_BGrande )
      wire#w1
      Contact( #PosSalidaCarga_OK )
      Contact( #Mx_ET02 )
      Contact( #PTF_Mx_MSig )
      Contact( #EstadoVI.Descarga_Act )
      I_Contact( #EstadoZona.ParoBlando_CBx )
      I_Contact( #Simultaneo_Mx )
      I_Contact( #FTF_Mx_MSig )
      I_Contact( #Selec_E1 )
      I_Contact( #Selec_E2 )
      I_Contact( #Selec_E3 )
      Contact( #EvolucionEtapasSalida )
      S_SR(operand := #Mx_ET60, r1 := #Mx_ET61)
   END_RUNG
   RUNG wire#powerrail
      Contact( #Selec_S4_BPequena )
   END_RUNG wire#w1
   // the same network as SCL:
   IF (#Selec_S4_BGrande OR #Selec_S4_BPequena) AND #PosSalidaCarga_OK AND #Mx_ET02 AND #PTF_Mx_MSig AND #EstadoVI.Descarga_Act AND NOT #EstadoZona.ParoBlando_CBx AND NOT #Simultaneo_Mx AND NOT #FTF_Mx_MSig AND NOT #Selec_E1 AND NOT #Selec_E2 AND NOT #Selec_E3 AND #EvolucionEtapasSalida THEN
       #Mx_ET60 := TRUE;   // SR flip-flop
   END_IF;
   IF #Mx_ET61 THEN #Mx_ET60 := FALSE; END_IF;
END_REGION

REGION Network 24: ET02 - ESTADO REPOSO CARGADA
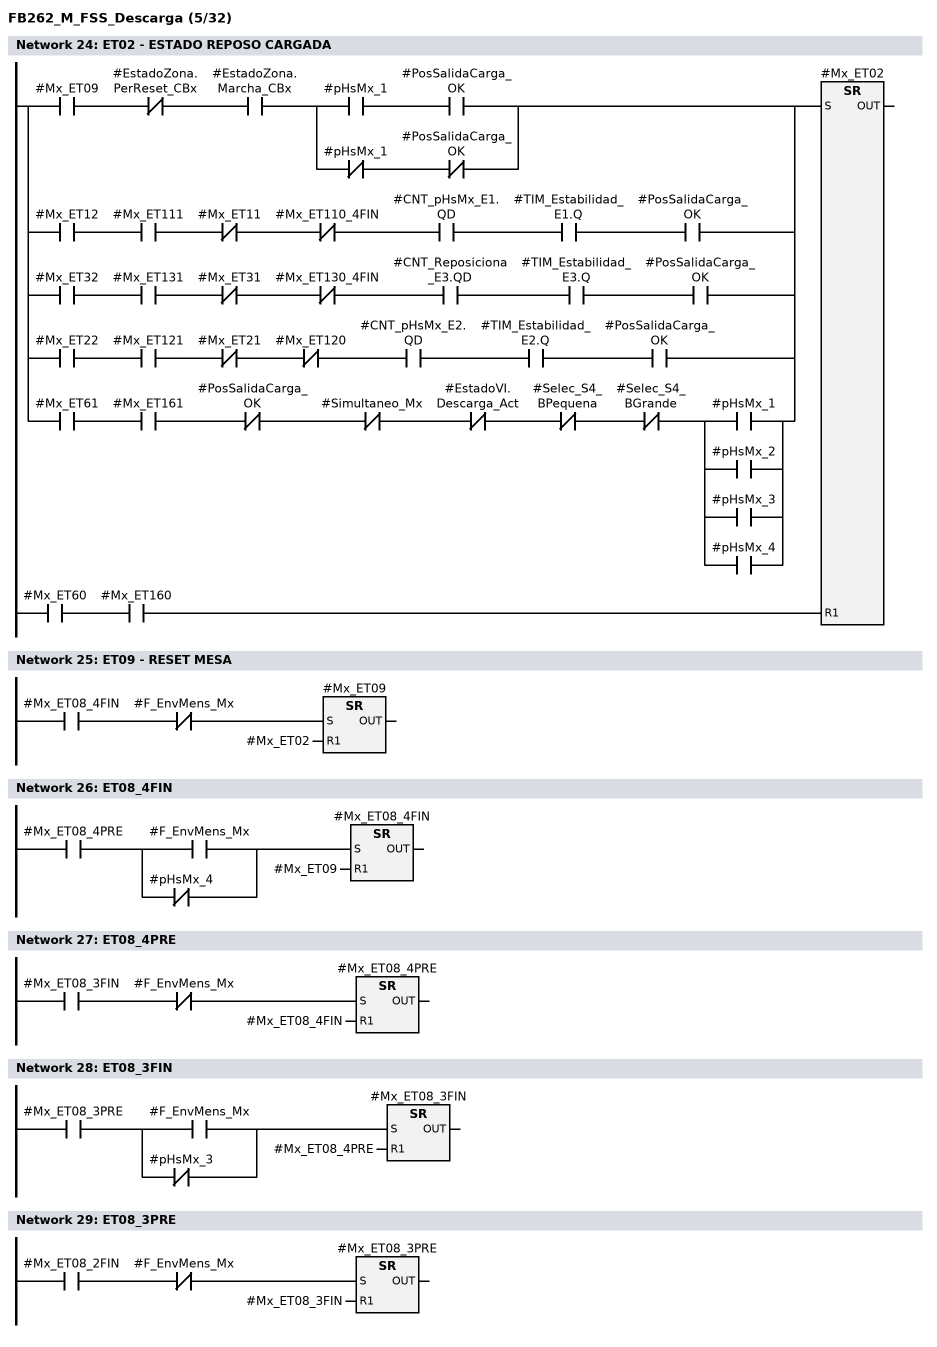
   RUNG wire#powerrail
      Contact( #Mx_ET09 )
      I_Contact( #EstadoZona.PerReset_CBx )
      Contact( #EstadoZona.Marcha_CBx )
      wire#w1
      Contact( #pHsMx_1 )
      Contact( #PosSalidaCarga_OK )
      wire#w2
      S_SR(operand := #Mx_ET02, r1 := wire#w4)
   END_RUNG
   RUNG wire#w1
      I_Contact( #pHsMx_1 )
      I_Contact( #PosSalidaCarga_OK )
   END_RUNG wire#w2
   RUNG wire#powerrail
      Contact( #Mx_ET12 )
      Contact( #Mx_ET111 )
      I_Contact( #Mx_ET11 )
      I_Contact( #Mx_ET110_4FIN )
      Contact( #CNT_pHsMx_E1.QD )
      Contact( #TIM_Estabilidad_E1.Q )
      Contact( #PosSalidaCarga_OK )
   END_RUNG wire#w2
   RUNG wire#powerrail
      Contact( #Mx_ET32 )
      Contact( #Mx_ET131 )
      I_Contact( #Mx_ET31 )
      I_Contact( #Mx_ET130_4FIN )
      Contact( #CNT_Reposiciona_E3.QD )
      Contact( #TIM_Estabilidad_E3.Q )
      Contact( #PosSalidaCarga_OK )
   END_RUNG wire#w2
   RUNG wire#powerrail
      Contact( #Mx_ET22 )
      Contact( #Mx_ET121 )
      I_Contact( #Mx_ET21 )
      I_Contact( #Mx_ET120 )
      Contact( #CNT_pHsMx_E2.QD )
      Contact( #TIM_Estabilidad_E2.Q )
      Contact( #PosSalidaCarga_OK )
   END_RUNG wire#w2
   RUNG wire#powerrail
      Contact( #Mx_ET61 )
      Contact( #Mx_ET161 )
      I_Contact( #PosSalidaCarga_OK )
      I_Contact( #Simultaneo_Mx )
      I_Contact( #EstadoVI.Descarga_Act )
      I_Contact( #Selec_S4_BPequena )
      I_Contact( #Selec_S4_BGrande )
      wire#w3
      Contact( #pHsMx_1 )
   END_RUNG wire#w2
   RUNG wire#w3
      Contact( #pHsMx_2 )
   END_RUNG wire#w2
   RUNG wire#w3
      Contact( #pHsMx_3 )
   END_RUNG wire#w2
   RUNG wire#w3
      Contact( #pHsMx_4 )
   END_RUNG wire#w2
   RUNG wire#powerrail
      Contact( #Mx_ET60 )
      Contact( #Mx_ET160 )
   END_RUNG wire#w4
   // the same network as SCL:
   IF (#Mx_ET09 AND NOT #EstadoZona.PerReset_CBx AND #EstadoZona.Marcha_CBx AND ((#pHsMx_1 AND #PosSalidaCarga_OK) OR (NOT #pHsMx_1 AND NOT #PosSalidaCarga_OK))) OR (#Mx_ET12 AND #Mx_ET111 AND NOT #Mx_ET11 AND NOT #Mx_ET110_4FIN AND #CNT_pHsMx_E1.QD AND #TIM_Estabilidad_E1.Q AND #PosSalidaCarga_OK) OR (#Mx_ET32 AND #Mx_ET131 AND NOT #Mx_ET31 AND NOT #Mx_ET130_4FIN AND #CNT_Reposiciona_E3.QD AND #TIM_Estabilidad_E3.Q AND #PosSalidaCarga_OK) OR (#Mx_ET22 AND #Mx_ET121 AND NOT #Mx_ET21 AND NOT #Mx_ET120 AND #CNT_pHsMx_E2.QD AND #TIM_Estabilidad_E2.Q AND #PosSalidaCarga_OK) OR (#Mx_ET61 AND #Mx_ET161 AND NOT #PosSalidaCarga_OK AND NOT #Simultaneo_Mx AND NOT #EstadoVI.Descarga_Act AND NOT #Selec_S4_BPequena AND NOT #Selec_S4_BGrande AND (#pHsMx_1 OR #pHsMx_2 OR #pHsMx_3 OR #pHsMx_4)) THEN
       #Mx_ET02 := TRUE;   // SR flip-flop
   END_IF;
   IF #Mx_ET60 AND #Mx_ET160 THEN #Mx_ET02 := FALSE; END_IF;
END_REGION

REGION Network 25: ET09 - RESET MESA
   RUNG wire#powerrail
      Contact( #Mx_ET08_4FIN )
      I_Contact( #F_EnvMens_Mx )
      S_SR(operand := #Mx_ET09, r1 := #Mx_ET02)
   END_RUNG
   // the same network as SCL:
   IF #Mx_ET08_4FIN AND NOT #F_EnvMens_Mx THEN
       #Mx_ET09 := TRUE;   // SR flip-flop
   END_IF;
   IF #Mx_ET02 THEN #Mx_ET09 := FALSE; END_IF;
END_REGION

REGION Network 26: ET08_4FIN
   RUNG wire#powerrail
      Contact( #Mx_ET08_4PRE )
      wire#w1
      Contact( #F_EnvMens_Mx )
      wire#w2
      S_SR(operand := #Mx_ET08_4FIN, r1 := #Mx_ET09)
   END_RUNG
   RUNG wire#w1
      I_Contact( #pHsMx_4 )
   END_RUNG wire#w2
   // the same network as SCL:
   IF #Mx_ET08_4PRE AND (#F_EnvMens_Mx OR NOT #pHsMx_4) THEN
       #Mx_ET08_4FIN := TRUE;   // SR flip-flop
   END_IF;
   IF #Mx_ET09 THEN #Mx_ET08_4FIN := FALSE; END_IF;
END_REGION

REGION Network 27: ET08_4PRE
   RUNG wire#powerrail
      Contact( #Mx_ET08_3FIN )
      I_Contact( #F_EnvMens_Mx )
      S_SR(operand := #Mx_ET08_4PRE, r1 := #Mx_ET08_4FIN)
   END_RUNG
   // the same network as SCL:
   IF #Mx_ET08_3FIN AND NOT #F_EnvMens_Mx THEN
       #Mx_ET08_4PRE := TRUE;   // SR flip-flop
   END_IF;
   IF #Mx_ET08_4FIN THEN #Mx_ET08_4PRE := FALSE; END_IF;
END_REGION

REGION Network 28: ET08_3FIN
   RUNG wire#powerrail
      Contact( #Mx_ET08_3PRE )
      wire#w1
      Contact( #F_EnvMens_Mx )
      wire#w2
      S_SR(operand := #Mx_ET08_3FIN, r1 := #Mx_ET08_4PRE)
   END_RUNG
   RUNG wire#w1
      I_Contact( #pHsMx_3 )
   END_RUNG wire#w2
   // the same network as SCL:
   IF #Mx_ET08_3PRE AND (#F_EnvMens_Mx OR NOT #pHsMx_3) THEN
       #Mx_ET08_3FIN := TRUE;   // SR flip-flop
   END_IF;
   IF #Mx_ET08_4PRE THEN #Mx_ET08_3FIN := FALSE; END_IF;
END_REGION

REGION Network 29: ET08_3PRE
   RUNG wire#powerrail
      Contact( #Mx_ET08_2FIN )
      I_Contact( #F_EnvMens_Mx )
      S_SR(operand := #Mx_ET08_3PRE, r1 := #Mx_ET08_3FIN)
   END_RUNG
   // the same network as SCL:
   IF #Mx_ET08_2FIN AND NOT #F_EnvMens_Mx THEN
       #Mx_ET08_3PRE := TRUE;   // SR flip-flop
   END_IF;
   IF #Mx_ET08_3FIN THEN #Mx_ET08_3PRE := FALSE; END_IF;
END_REGION

REGION Network 30: ET08_2FIN
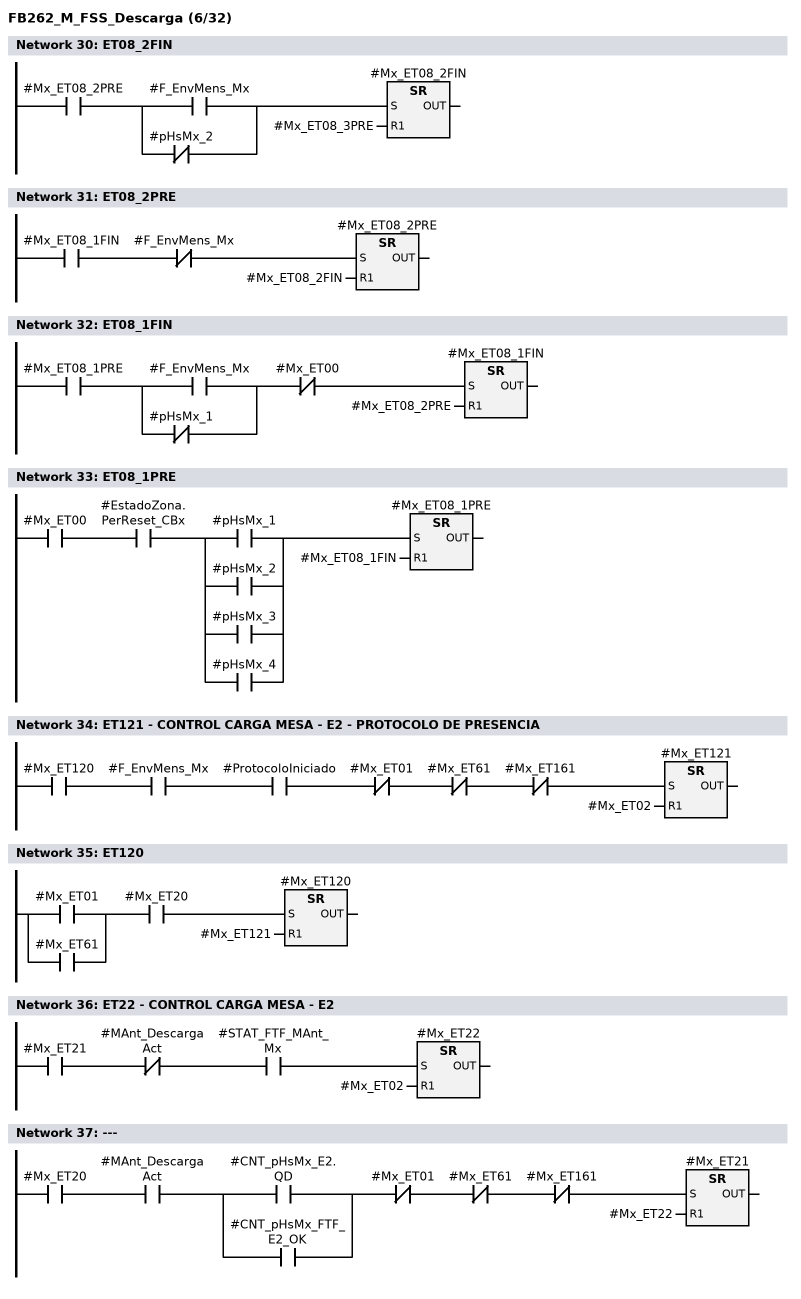
   RUNG wire#powerrail
      Contact( #Mx_ET08_2PRE )
      wire#w1
      Contact( #F_EnvMens_Mx )
      wire#w2
      S_SR(operand := #Mx_ET08_2FIN, r1 := #Mx_ET08_3PRE)
   END_RUNG
   RUNG wire#w1
      I_Contact( #pHsMx_2 )
   END_RUNG wire#w2
   // the same network as SCL:
   IF #Mx_ET08_2PRE AND (#F_EnvMens_Mx OR NOT #pHsMx_2) THEN
       #Mx_ET08_2FIN := TRUE;   // SR flip-flop
   END_IF;
   IF #Mx_ET08_3PRE THEN #Mx_ET08_2FIN := FALSE; END_IF;
END_REGION

REGION Network 31: ET08_2PRE
   RUNG wire#powerrail
      Contact( #Mx_ET08_1FIN )
      I_Contact( #F_EnvMens_Mx )
      S_SR(operand := #Mx_ET08_2PRE, r1 := #Mx_ET08_2FIN)
   END_RUNG
   // the same network as SCL:
   IF #Mx_ET08_1FIN AND NOT #F_EnvMens_Mx THEN
       #Mx_ET08_2PRE := TRUE;   // SR flip-flop
   END_IF;
   IF #Mx_ET08_2FIN THEN #Mx_ET08_2PRE := FALSE; END_IF;
END_REGION

REGION Network 32: ET08_1FIN
   RUNG wire#powerrail
      Contact( #Mx_ET08_1PRE )
      wire#w1
      Contact( #F_EnvMens_Mx )
      wire#w2
      I_Contact( #Mx_ET00 )
      S_SR(operand := #Mx_ET08_1FIN, r1 := #Mx_ET08_2PRE)
   END_RUNG
   RUNG wire#w1
      I_Contact( #pHsMx_1 )
   END_RUNG wire#w2
   // the same network as SCL:
   IF #Mx_ET08_1PRE AND (#F_EnvMens_Mx OR NOT #pHsMx_1) AND NOT #Mx_ET00 THEN
       #Mx_ET08_1FIN := TRUE;   // SR flip-flop
   END_IF;
   IF #Mx_ET08_2PRE THEN #Mx_ET08_1FIN := FALSE; END_IF;
END_REGION

REGION Network 33: ET08_1PRE
   RUNG wire#powerrail
      Contact( #Mx_ET00 )
      Contact( #EstadoZona.PerReset_CBx )
      wire#w1
      Contact( #pHsMx_1 )
      wire#w2
      S_SR(operand := #Mx_ET08_1PRE, r1 := #Mx_ET08_1FIN)
   END_RUNG
   RUNG wire#w1
      Contact( #pHsMx_2 )
   END_RUNG wire#w2
   RUNG wire#w1
      Contact( #pHsMx_3 )
   END_RUNG wire#w2
   RUNG wire#w1
      Contact( #pHsMx_4 )
   END_RUNG wire#w2
   // the same network as SCL:
   IF #Mx_ET00 AND #EstadoZona.PerReset_CBx AND (#pHsMx_1 OR #pHsMx_2 OR #pHsMx_3 OR #pHsMx_4) THEN
       #Mx_ET08_1PRE := TRUE;   // SR flip-flop
   END_IF;
   IF #Mx_ET08_1FIN THEN #Mx_ET08_1PRE := FALSE; END_IF;
END_REGION

REGION Network 34: ET121 - CONTROL CARGA MESA - E2 - PROTOCOLO DE PRESENCIA
   RUNG wire#powerrail
      Contact( #Mx_ET120 )
      Contact( #F_EnvMens_Mx )
      Contact( #ProtocoloIniciado )
      I_Contact( #Mx_ET01 )
      I_Contact( #Mx_ET61 )
      I_Contact( #Mx_ET161 )
      S_SR(operand := #Mx_ET121, r1 := #Mx_ET02)
   END_RUNG
   // the same network as SCL:
   IF #Mx_ET120 AND #F_EnvMens_Mx AND #ProtocoloIniciado AND NOT #Mx_ET01 AND NOT #Mx_ET61 AND NOT #Mx_ET161 THEN
       #Mx_ET121 := TRUE;   // SR flip-flop
   END_IF;
   IF #Mx_ET02 THEN #Mx_ET121 := FALSE; END_IF;
END_REGION

REGION Network 35: ET120
   RUNG wire#powerrail
      Contact( #Mx_ET01 )
      wire#w1
      Contact( #Mx_ET20 )
      S_SR(operand := #Mx_ET120, r1 := #Mx_ET121)
   END_RUNG
   RUNG wire#powerrail
      Contact( #Mx_ET61 )
   END_RUNG wire#w1
   // the same network as SCL:
   IF (#Mx_ET01 OR #Mx_ET61) AND #Mx_ET20 THEN
       #Mx_ET120 := TRUE;   // SR flip-flop
   END_IF;
   IF #Mx_ET121 THEN #Mx_ET120 := FALSE; END_IF;
END_REGION

REGION Network 36: ET22 - CONTROL CARGA MESA - E2
   RUNG wire#powerrail
      Contact( #Mx_ET21 )
      I_Contact( #MAnt_DescargaAct )
      Contact( #STAT_FTF_MAnt_Mx )
      S_SR(operand := #Mx_ET22, r1 := #Mx_ET02)
   END_RUNG
   // the same network as SCL:
   IF #Mx_ET21 AND NOT #MAnt_DescargaAct AND #STAT_FTF_MAnt_Mx THEN
       #Mx_ET22 := TRUE;   // SR flip-flop
   END_IF;
   IF #Mx_ET02 THEN #Mx_ET22 := FALSE; END_IF;
END_REGION

REGION Network 37: ---
   RUNG wire#powerrail
      Contact( #Mx_ET20 )
      Contact( #MAnt_DescargaAct )
      wire#w1
      Contact( #CNT_pHsMx_E2.QD )
      wire#w2
      I_Contact( #Mx_ET01 )
      I_Contact( #Mx_ET61 )
      I_Contact( #Mx_ET161 )
      S_SR(operand := #Mx_ET21, r1 := #Mx_ET22)
   END_RUNG
   RUNG wire#w1
      Contact( #CNT_pHsMx_FTF_E2_OK )
   END_RUNG wire#w2
   // the same network as SCL:
   IF #Mx_ET20 AND #MAnt_DescargaAct AND (#CNT_pHsMx_E2.QD OR #CNT_pHsMx_FTF_E2_OK) AND NOT #Mx_ET01 AND NOT #Mx_ET61 AND NOT #Mx_ET161 THEN
       #Mx_ET21 := TRUE;   // SR flip-flop
   END_IF;
   IF #Mx_ET22 THEN #Mx_ET21 := FALSE; END_IF;
END_REGION

REGION Network 38: ---
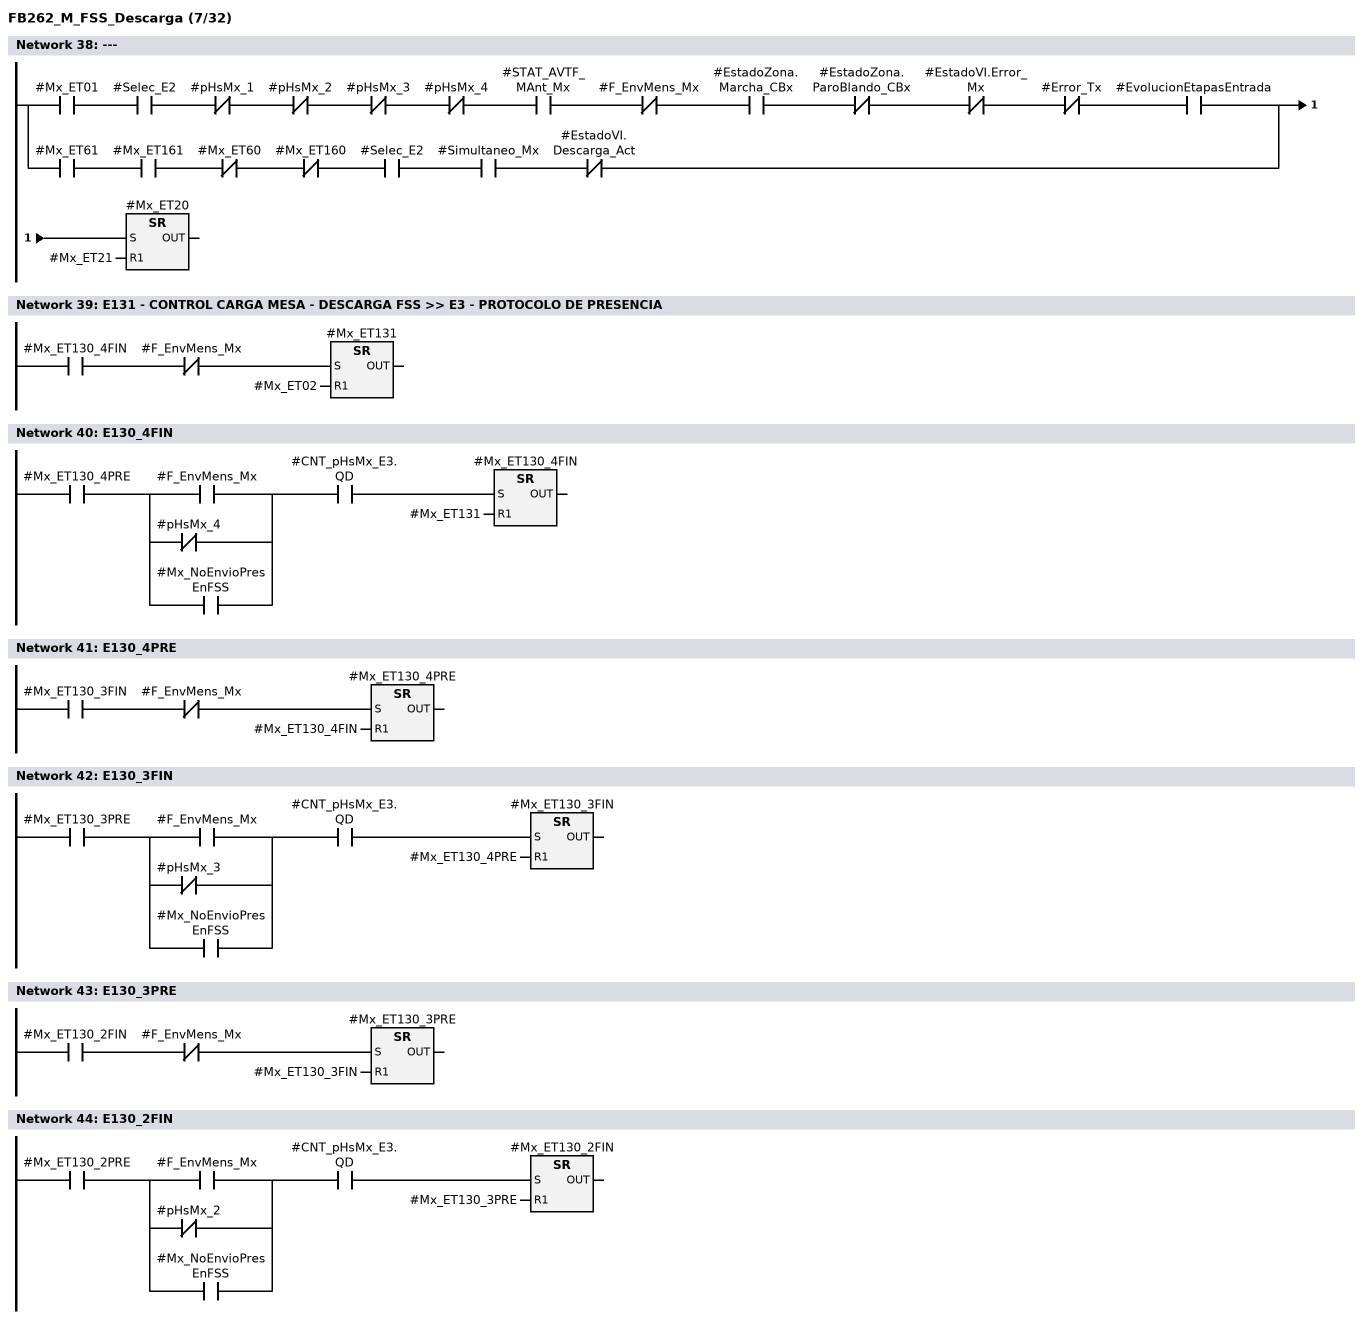
   RUNG wire#powerrail
      Contact( #Mx_ET01 )
      Contact( #Selec_E2 )
      I_Contact( #pHsMx_1 )
      I_Contact( #pHsMx_2 )
      I_Contact( #pHsMx_3 )
      I_Contact( #pHsMx_4 )
      Contact( #STAT_AVTF_MAnt_Mx )
      I_Contact( #F_EnvMens_Mx )
      Contact( #EstadoZona.Marcha_CBx )
      I_Contact( #EstadoZona.ParoBlando_CBx )
      I_Contact( #EstadoVI.Error_Mx )
      I_Contact( #Error_Tx )
      Contact( #EvolucionEtapasEntrada )
      wire#w1
      S_SR(operand := #Mx_ET20, r1 := #Mx_ET21)
   END_RUNG
   RUNG wire#powerrail
      Contact( #Mx_ET61 )
      Contact( #Mx_ET161 )
      I_Contact( #Mx_ET60 )
      I_Contact( #Mx_ET160 )
      Contact( #Selec_E2 )
      Contact( #Simultaneo_Mx )
      I_Contact( #EstadoVI.Descarga_Act )
   END_RUNG wire#w1
   // the same network as SCL:
   IF (#Mx_ET01 AND #Selec_E2 AND NOT #pHsMx_1 AND NOT #pHsMx_2 AND NOT #pHsMx_3 AND NOT #pHsMx_4 AND #STAT_AVTF_MAnt_Mx AND NOT #F_EnvMens_Mx AND #EstadoZona.Marcha_CBx AND NOT #EstadoZona.ParoBlando_CBx AND NOT #EstadoVI.Error_Mx AND NOT #Error_Tx AND #EvolucionEtapasEntrada) OR (#Mx_ET61 AND #Mx_ET161 AND NOT #Mx_ET60 AND NOT #Mx_ET160 AND #Selec_E2 AND #Simultaneo_Mx AND NOT #EstadoVI.Descarga_Act) THEN
       #Mx_ET20 := TRUE;   // SR flip-flop
   END_IF;
   IF #Mx_ET21 THEN #Mx_ET20 := FALSE; END_IF;
END_REGION

REGION Network 39: E131 - CONTROL CARGA MESA - DESCARGA FSS >> E3 - PROTOCOLO DE PRESENCIA
   RUNG wire#powerrail
      Contact( #Mx_ET130_4FIN )
      I_Contact( #F_EnvMens_Mx )
      S_SR(operand := #Mx_ET131, r1 := #Mx_ET02)
   END_RUNG
   // the same network as SCL:
   IF #Mx_ET130_4FIN AND NOT #F_EnvMens_Mx THEN
       #Mx_ET131 := TRUE;   // SR flip-flop
   END_IF;
   IF #Mx_ET02 THEN #Mx_ET131 := FALSE; END_IF;
END_REGION

REGION Network 40: E130_4FIN
   RUNG wire#powerrail
      Contact( #Mx_ET130_4PRE )
      wire#w1
      Contact( #F_EnvMens_Mx )
      wire#w2
      Contact( #CNT_pHsMx_E3.QD )
      S_SR(operand := #Mx_ET130_4FIN, r1 := #Mx_ET131)
   END_RUNG
   RUNG wire#w1
      I_Contact( #pHsMx_4 )
   END_RUNG wire#w2
   RUNG wire#w1
      Contact( #Mx_NoEnvioPresEnFSS )
   END_RUNG wire#w2
   // the same network as SCL:
   IF #Mx_ET130_4PRE AND (#F_EnvMens_Mx OR NOT #pHsMx_4 OR #Mx_NoEnvioPresEnFSS) AND #CNT_pHsMx_E3.QD THEN
       #Mx_ET130_4FIN := TRUE;   // SR flip-flop
   END_IF;
   IF #Mx_ET131 THEN #Mx_ET130_4FIN := FALSE; END_IF;
END_REGION

REGION Network 41: E130_4PRE
   RUNG wire#powerrail
      Contact( #Mx_ET130_3FIN )
      I_Contact( #F_EnvMens_Mx )
      S_SR(operand := #Mx_ET130_4PRE, r1 := #Mx_ET130_4FIN)
   END_RUNG
   // the same network as SCL:
   IF #Mx_ET130_3FIN AND NOT #F_EnvMens_Mx THEN
       #Mx_ET130_4PRE := TRUE;   // SR flip-flop
   END_IF;
   IF #Mx_ET130_4FIN THEN #Mx_ET130_4PRE := FALSE; END_IF;
END_REGION

REGION Network 42: E130_3FIN
   RUNG wire#powerrail
      Contact( #Mx_ET130_3PRE )
      wire#w1
      Contact( #F_EnvMens_Mx )
      wire#w2
      Contact( #CNT_pHsMx_E3.QD )
      S_SR(operand := #Mx_ET130_3FIN, r1 := #Mx_ET130_4PRE)
   END_RUNG
   RUNG wire#w1
      I_Contact( #pHsMx_3 )
   END_RUNG wire#w2
   RUNG wire#w1
      Contact( #Mx_NoEnvioPresEnFSS )
   END_RUNG wire#w2
   // the same network as SCL:
   IF #Mx_ET130_3PRE AND (#F_EnvMens_Mx OR NOT #pHsMx_3 OR #Mx_NoEnvioPresEnFSS) AND #CNT_pHsMx_E3.QD THEN
       #Mx_ET130_3FIN := TRUE;   // SR flip-flop
   END_IF;
   IF #Mx_ET130_4PRE THEN #Mx_ET130_3FIN := FALSE; END_IF;
END_REGION

REGION Network 43: E130_3PRE
   RUNG wire#powerrail
      Contact( #Mx_ET130_2FIN )
      I_Contact( #F_EnvMens_Mx )
      S_SR(operand := #Mx_ET130_3PRE, r1 := #Mx_ET130_3FIN)
   END_RUNG
   // the same network as SCL:
   IF #Mx_ET130_2FIN AND NOT #F_EnvMens_Mx THEN
       #Mx_ET130_3PRE := TRUE;   // SR flip-flop
   END_IF;
   IF #Mx_ET130_3FIN THEN #Mx_ET130_3PRE := FALSE; END_IF;
END_REGION

REGION Network 44: E130_2FIN
   RUNG wire#powerrail
      Contact( #Mx_ET130_2PRE )
      wire#w1
      Contact( #F_EnvMens_Mx )
      wire#w2
      Contact( #CNT_pHsMx_E3.QD )
      S_SR(operand := #Mx_ET130_2FIN, r1 := #Mx_ET130_3PRE)
   END_RUNG
   RUNG wire#w1
      I_Contact( #pHsMx_2 )
   END_RUNG wire#w2
   RUNG wire#w1
      Contact( #Mx_NoEnvioPresEnFSS )
   END_RUNG wire#w2
   // the same network as SCL:
   IF #Mx_ET130_2PRE AND (#F_EnvMens_Mx OR NOT #pHsMx_2 OR #Mx_NoEnvioPresEnFSS) AND #CNT_pHsMx_E3.QD THEN
       #Mx_ET130_2FIN := TRUE;   // SR flip-flop
   END_IF;
   IF #Mx_ET130_3PRE THEN #Mx_ET130_2FIN := FALSE; END_IF;
END_REGION

REGION Network 45: E130_2PRE
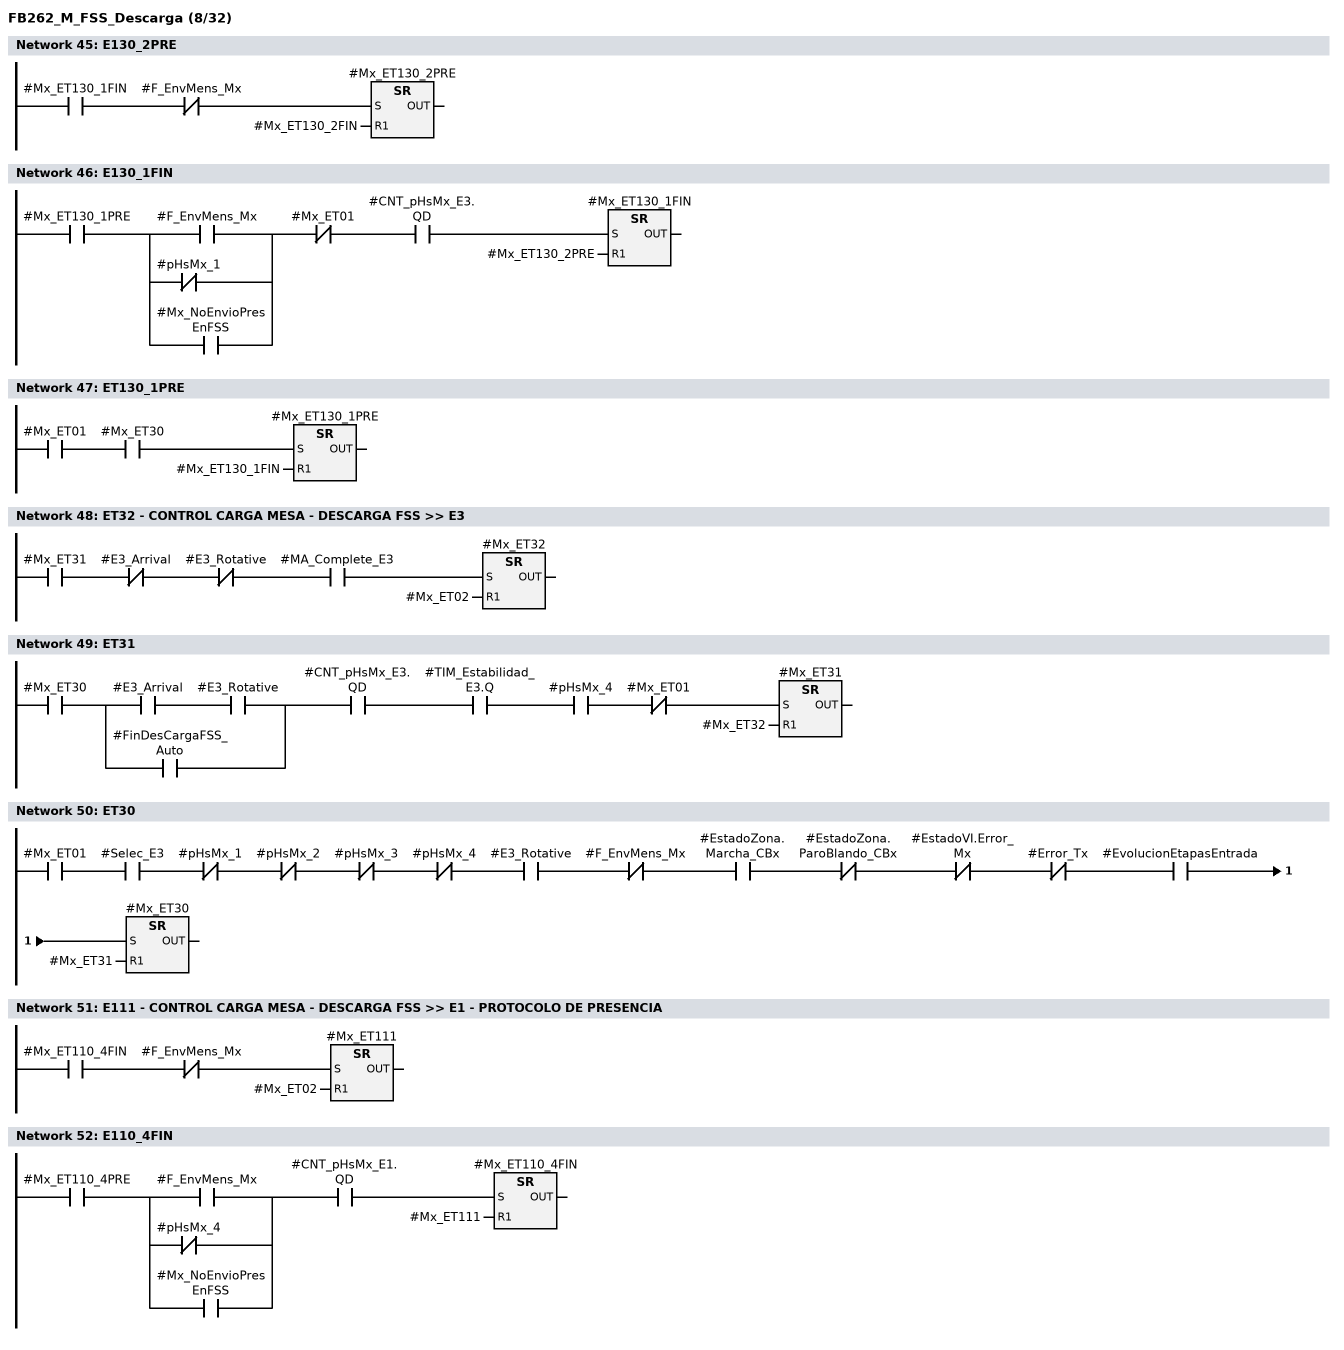
   RUNG wire#powerrail
      Contact( #Mx_ET130_1FIN )
      I_Contact( #F_EnvMens_Mx )
      S_SR(operand := #Mx_ET130_2PRE, r1 := #Mx_ET130_2FIN)
   END_RUNG
   // the same network as SCL:
   IF #Mx_ET130_1FIN AND NOT #F_EnvMens_Mx THEN
       #Mx_ET130_2PRE := TRUE;   // SR flip-flop
   END_IF;
   IF #Mx_ET130_2FIN THEN #Mx_ET130_2PRE := FALSE; END_IF;
END_REGION

REGION Network 46: E130_1FIN
   RUNG wire#powerrail
      Contact( #Mx_ET130_1PRE )
      wire#w1
      Contact( #F_EnvMens_Mx )
      wire#w2
      I_Contact( #Mx_ET01 )
      Contact( #CNT_pHsMx_E3.QD )
      S_SR(operand := #Mx_ET130_1FIN, r1 := #Mx_ET130_2PRE)
   END_RUNG
   RUNG wire#w1
      I_Contact( #pHsMx_1 )
   END_RUNG wire#w2
   RUNG wire#w1
      Contact( #Mx_NoEnvioPresEnFSS )
   END_RUNG wire#w2
   // the same network as SCL:
   IF #Mx_ET130_1PRE AND (#F_EnvMens_Mx OR NOT #pHsMx_1 OR #Mx_NoEnvioPresEnFSS) AND NOT #Mx_ET01 AND #CNT_pHsMx_E3.QD THEN
       #Mx_ET130_1FIN := TRUE;   // SR flip-flop
   END_IF;
   IF #Mx_ET130_2PRE THEN #Mx_ET130_1FIN := FALSE; END_IF;
END_REGION

REGION Network 47: ET130_1PRE
   RUNG wire#powerrail
      Contact( #Mx_ET01 )
      Contact( #Mx_ET30 )
      S_SR(operand := #Mx_ET130_1PRE, r1 := #Mx_ET130_1FIN)
   END_RUNG
   // the same network as SCL:
   IF #Mx_ET01 AND #Mx_ET30 THEN
       #Mx_ET130_1PRE := TRUE;   // SR flip-flop
   END_IF;
   IF #Mx_ET130_1FIN THEN #Mx_ET130_1PRE := FALSE; END_IF;
END_REGION

REGION Network 48: ET32 - CONTROL CARGA MESA - DESCARGA FSS >> E3
   RUNG wire#powerrail
      Contact( #Mx_ET31 )
      I_Contact( #E3_Arrival )
      I_Contact( #E3_Rotative )
      Contact( #MA_Complete_E3 )
      S_SR(operand := #Mx_ET32, r1 := #Mx_ET02)
   END_RUNG
   // the same network as SCL:
   IF #Mx_ET31 AND NOT #E3_Arrival AND NOT #E3_Rotative AND #MA_Complete_E3 THEN
       #Mx_ET32 := TRUE;   // SR flip-flop
   END_IF;
   IF #Mx_ET02 THEN #Mx_ET32 := FALSE; END_IF;
END_REGION

REGION Network 49: ET31
   RUNG wire#powerrail
      Contact( #Mx_ET30 )
      wire#w1
      Contact( #E3_Arrival )
      Contact( #E3_Rotative )
      wire#w2
      Contact( #CNT_pHsMx_E3.QD )
      Contact( #TIM_Estabilidad_E3.Q )
      Contact( #pHsMx_4 )
      I_Contact( #Mx_ET01 )
      S_SR(operand := #Mx_ET31, r1 := #Mx_ET32)
   END_RUNG
   RUNG wire#w1
      Contact( #FinDesCargaFSS_Auto )
   END_RUNG wire#w2
   // the same network as SCL:
   IF #Mx_ET30 AND ((#E3_Arrival AND #E3_Rotative) OR #FinDesCargaFSS_Auto) AND #CNT_pHsMx_E3.QD AND #TIM_Estabilidad_E3.Q AND #pHsMx_4 AND NOT #Mx_ET01 THEN
       #Mx_ET31 := TRUE;   // SR flip-flop
   END_IF;
   IF #Mx_ET32 THEN #Mx_ET31 := FALSE; END_IF;
END_REGION

REGION Network 50: ET30
   RUNG wire#powerrail
      Contact( #Mx_ET01 )
      Contact( #Selec_E3 )
      I_Contact( #pHsMx_1 )
      I_Contact( #pHsMx_2 )
      I_Contact( #pHsMx_3 )
      I_Contact( #pHsMx_4 )
      Contact( #E3_Rotative )
      I_Contact( #F_EnvMens_Mx )
      Contact( #EstadoZona.Marcha_CBx )
      I_Contact( #EstadoZona.ParoBlando_CBx )
      I_Contact( #EstadoVI.Error_Mx )
      I_Contact( #Error_Tx )
      Contact( #EvolucionEtapasEntrada )
      S_SR(operand := #Mx_ET30, r1 := #Mx_ET31)
   END_RUNG
   // the same network as SCL:
   IF #Mx_ET01 AND #Selec_E3 AND NOT #pHsMx_1 AND NOT #pHsMx_2 AND NOT #pHsMx_3 AND NOT #pHsMx_4 AND #E3_Rotative AND NOT #F_EnvMens_Mx AND #EstadoZona.Marcha_CBx AND NOT #EstadoZona.ParoBlando_CBx AND NOT #EstadoVI.Error_Mx AND NOT #Error_Tx AND #EvolucionEtapasEntrada THEN
       #Mx_ET30 := TRUE;   // SR flip-flop
   END_IF;
   IF #Mx_ET31 THEN #Mx_ET30 := FALSE; END_IF;
END_REGION

REGION Network 51: E111 - CONTROL CARGA MESA - DESCARGA FSS >> E1 - PROTOCOLO DE PRESENCIA
   RUNG wire#powerrail
      Contact( #Mx_ET110_4FIN )
      I_Contact( #F_EnvMens_Mx )
      S_SR(operand := #Mx_ET111, r1 := #Mx_ET02)
   END_RUNG
   // the same network as SCL:
   IF #Mx_ET110_4FIN AND NOT #F_EnvMens_Mx THEN
       #Mx_ET111 := TRUE;   // SR flip-flop
   END_IF;
   IF #Mx_ET02 THEN #Mx_ET111 := FALSE; END_IF;
END_REGION

REGION Network 52: E110_4FIN
   RUNG wire#powerrail
      Contact( #Mx_ET110_4PRE )
      wire#w1
      Contact( #F_EnvMens_Mx )
      wire#w2
      Contact( #CNT_pHsMx_E1.QD )
      S_SR(operand := #Mx_ET110_4FIN, r1 := #Mx_ET111)
   END_RUNG
   RUNG wire#w1
      I_Contact( #pHsMx_4 )
   END_RUNG wire#w2
   RUNG wire#w1
      Contact( #Mx_NoEnvioPresEnFSS )
   END_RUNG wire#w2
   // the same network as SCL:
   IF #Mx_ET110_4PRE AND (#F_EnvMens_Mx OR NOT #pHsMx_4 OR #Mx_NoEnvioPresEnFSS) AND #CNT_pHsMx_E1.QD THEN
       #Mx_ET110_4FIN := TRUE;   // SR flip-flop
   END_IF;
   IF #Mx_ET111 THEN #Mx_ET110_4FIN := FALSE; END_IF;
END_REGION

REGION Network 53: E110_4PRE
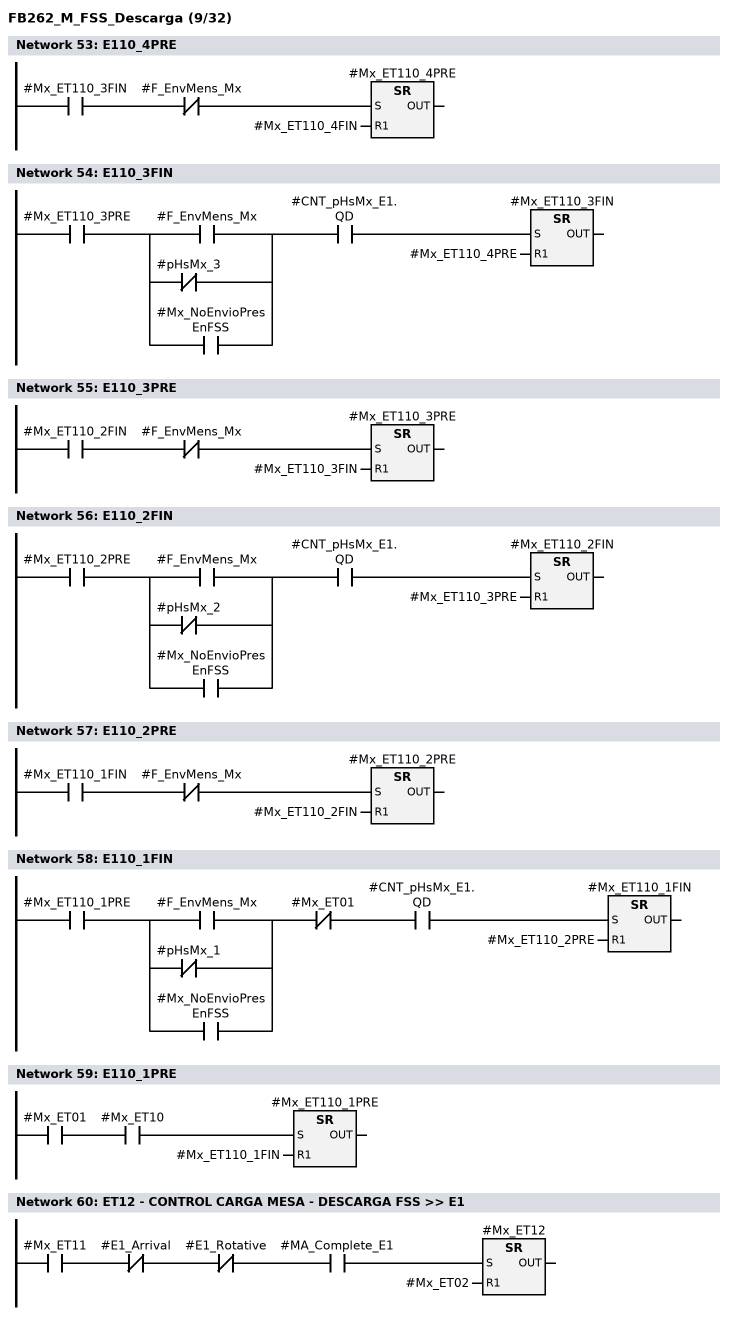
   RUNG wire#powerrail
      Contact( #Mx_ET110_3FIN )
      I_Contact( #F_EnvMens_Mx )
      S_SR(operand := #Mx_ET110_4PRE, r1 := #Mx_ET110_4FIN)
   END_RUNG
   // the same network as SCL:
   IF #Mx_ET110_3FIN AND NOT #F_EnvMens_Mx THEN
       #Mx_ET110_4PRE := TRUE;   // SR flip-flop
   END_IF;
   IF #Mx_ET110_4FIN THEN #Mx_ET110_4PRE := FALSE; END_IF;
END_REGION

REGION Network 54: E110_3FIN
   RUNG wire#powerrail
      Contact( #Mx_ET110_3PRE )
      wire#w1
      Contact( #F_EnvMens_Mx )
      wire#w2
      Contact( #CNT_pHsMx_E1.QD )
      S_SR(operand := #Mx_ET110_3FIN, r1 := #Mx_ET110_4PRE)
   END_RUNG
   RUNG wire#w1
      I_Contact( #pHsMx_3 )
   END_RUNG wire#w2
   RUNG wire#w1
      Contact( #Mx_NoEnvioPresEnFSS )
   END_RUNG wire#w2
   // the same network as SCL:
   IF #Mx_ET110_3PRE AND (#F_EnvMens_Mx OR NOT #pHsMx_3 OR #Mx_NoEnvioPresEnFSS) AND #CNT_pHsMx_E1.QD THEN
       #Mx_ET110_3FIN := TRUE;   // SR flip-flop
   END_IF;
   IF #Mx_ET110_4PRE THEN #Mx_ET110_3FIN := FALSE; END_IF;
END_REGION

REGION Network 55: E110_3PRE
   RUNG wire#powerrail
      Contact( #Mx_ET110_2FIN )
      I_Contact( #F_EnvMens_Mx )
      S_SR(operand := #Mx_ET110_3PRE, r1 := #Mx_ET110_3FIN)
   END_RUNG
   // the same network as SCL:
   IF #Mx_ET110_2FIN AND NOT #F_EnvMens_Mx THEN
       #Mx_ET110_3PRE := TRUE;   // SR flip-flop
   END_IF;
   IF #Mx_ET110_3FIN THEN #Mx_ET110_3PRE := FALSE; END_IF;
END_REGION

REGION Network 56: E110_2FIN
   RUNG wire#powerrail
      Contact( #Mx_ET110_2PRE )
      wire#w1
      Contact( #F_EnvMens_Mx )
      wire#w2
      Contact( #CNT_pHsMx_E1.QD )
      S_SR(operand := #Mx_ET110_2FIN, r1 := #Mx_ET110_3PRE)
   END_RUNG
   RUNG wire#w1
      I_Contact( #pHsMx_2 )
   END_RUNG wire#w2
   RUNG wire#w1
      Contact( #Mx_NoEnvioPresEnFSS )
   END_RUNG wire#w2
   // the same network as SCL:
   IF #Mx_ET110_2PRE AND (#F_EnvMens_Mx OR NOT #pHsMx_2 OR #Mx_NoEnvioPresEnFSS) AND #CNT_pHsMx_E1.QD THEN
       #Mx_ET110_2FIN := TRUE;   // SR flip-flop
   END_IF;
   IF #Mx_ET110_3PRE THEN #Mx_ET110_2FIN := FALSE; END_IF;
END_REGION

REGION Network 57: E110_2PRE
   RUNG wire#powerrail
      Contact( #Mx_ET110_1FIN )
      I_Contact( #F_EnvMens_Mx )
      S_SR(operand := #Mx_ET110_2PRE, r1 := #Mx_ET110_2FIN)
   END_RUNG
   // the same network as SCL:
   IF #Mx_ET110_1FIN AND NOT #F_EnvMens_Mx THEN
       #Mx_ET110_2PRE := TRUE;   // SR flip-flop
   END_IF;
   IF #Mx_ET110_2FIN THEN #Mx_ET110_2PRE := FALSE; END_IF;
END_REGION

REGION Network 58: E110_1FIN
   RUNG wire#powerrail
      Contact( #Mx_ET110_1PRE )
      wire#w1
      Contact( #F_EnvMens_Mx )
      wire#w2
      I_Contact( #Mx_ET01 )
      Contact( #CNT_pHsMx_E1.QD )
      S_SR(operand := #Mx_ET110_1FIN, r1 := #Mx_ET110_2PRE)
   END_RUNG
   RUNG wire#w1
      I_Contact( #pHsMx_1 )
   END_RUNG wire#w2
   RUNG wire#w1
      Contact( #Mx_NoEnvioPresEnFSS )
   END_RUNG wire#w2
   // the same network as SCL:
   IF #Mx_ET110_1PRE AND (#F_EnvMens_Mx OR NOT #pHsMx_1 OR #Mx_NoEnvioPresEnFSS) AND NOT #Mx_ET01 AND #CNT_pHsMx_E1.QD THEN
       #Mx_ET110_1FIN := TRUE;   // SR flip-flop
   END_IF;
   IF #Mx_ET110_2PRE THEN #Mx_ET110_1FIN := FALSE; END_IF;
END_REGION

REGION Network 59: E110_1PRE
   RUNG wire#powerrail
      Contact( #Mx_ET01 )
      Contact( #Mx_ET10 )
      S_SR(operand := #Mx_ET110_1PRE, r1 := #Mx_ET110_1FIN)
   END_RUNG
   // the same network as SCL:
   IF #Mx_ET01 AND #Mx_ET10 THEN
       #Mx_ET110_1PRE := TRUE;   // SR flip-flop
   END_IF;
   IF #Mx_ET110_1FIN THEN #Mx_ET110_1PRE := FALSE; END_IF;
END_REGION

REGION Network 60: ET12 - CONTROL CARGA MESA - DESCARGA FSS >> E1
   RUNG wire#powerrail
      Contact( #Mx_ET11 )
      I_Contact( #E1_Arrival )
      I_Contact( #E1_Rotative )
      Contact( #MA_Complete_E1 )
      S_SR(operand := #Mx_ET12, r1 := #Mx_ET02)
   END_RUNG
   // the same network as SCL:
   IF #Mx_ET11 AND NOT #E1_Arrival AND NOT #E1_Rotative AND #MA_Complete_E1 THEN
       #Mx_ET12 := TRUE;   // SR flip-flop
   END_IF;
   IF #Mx_ET02 THEN #Mx_ET12 := FALSE; END_IF;
END_REGION

REGION Network 61: ET11
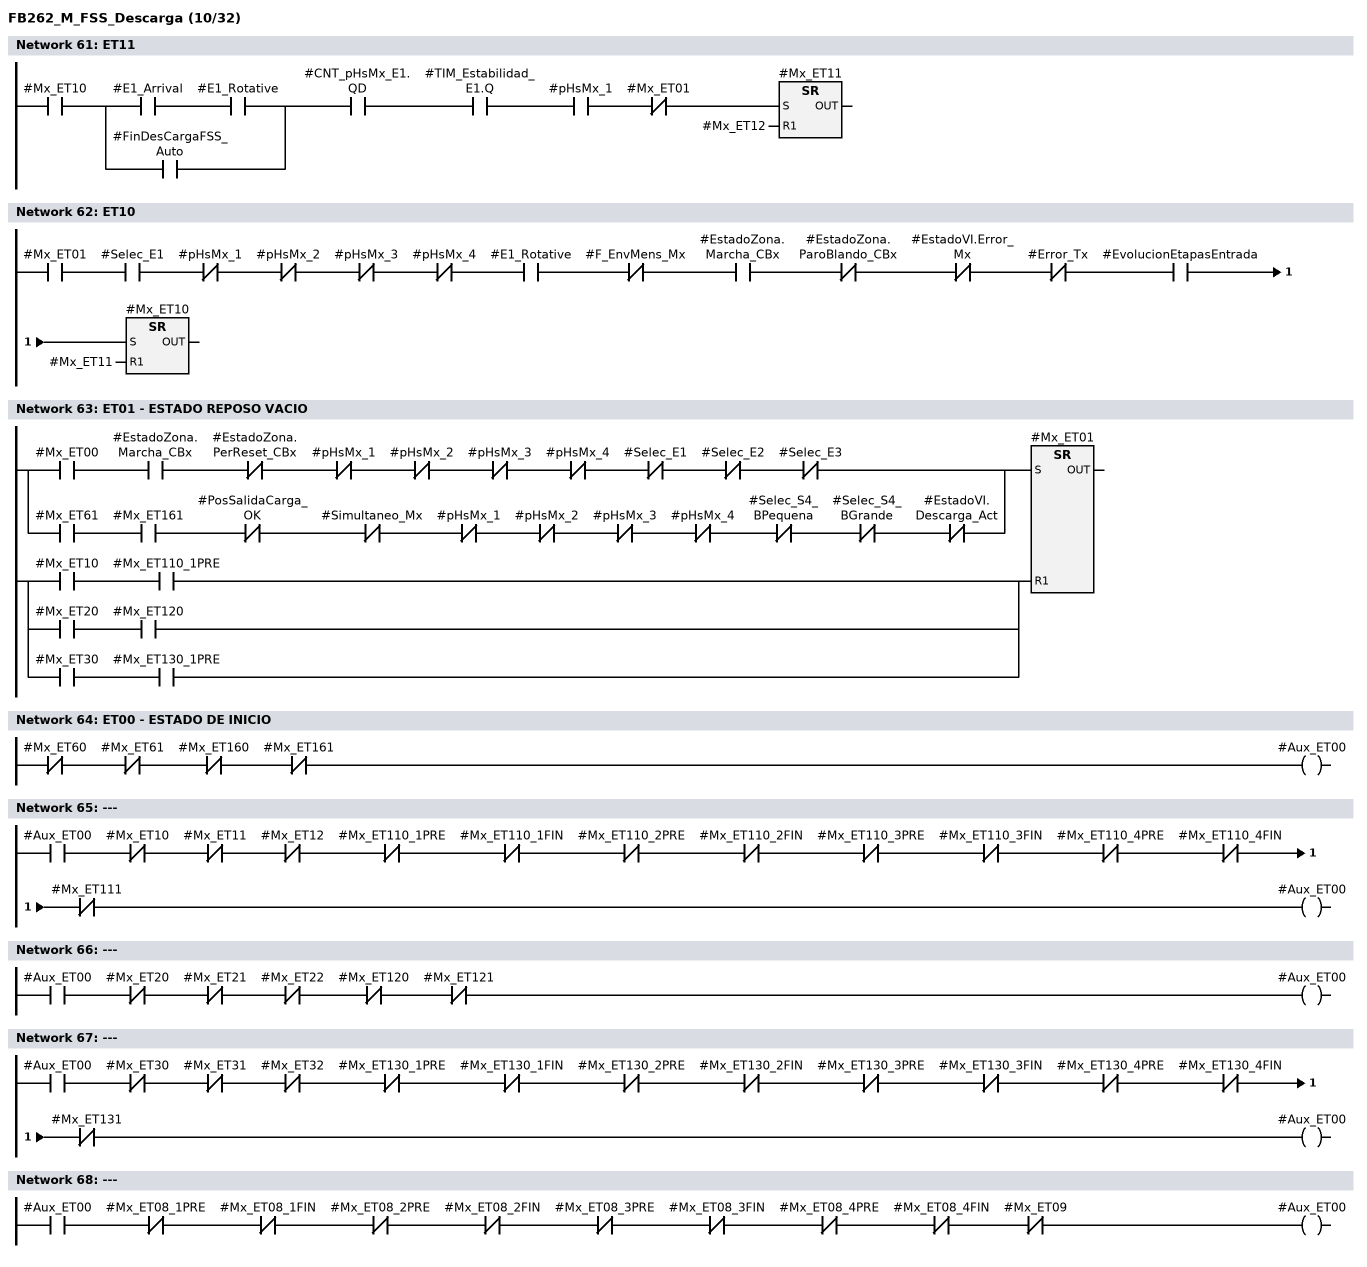
   RUNG wire#powerrail
      Contact( #Mx_ET10 )
      wire#w1
      Contact( #E1_Arrival )
      Contact( #E1_Rotative )
      wire#w2
      Contact( #CNT_pHsMx_E1.QD )
      Contact( #TIM_Estabilidad_E1.Q )
      Contact( #pHsMx_1 )
      I_Contact( #Mx_ET01 )
      S_SR(operand := #Mx_ET11, r1 := #Mx_ET12)
   END_RUNG
   RUNG wire#w1
      Contact( #FinDesCargaFSS_Auto )
   END_RUNG wire#w2
   // the same network as SCL:
   IF #Mx_ET10 AND ((#E1_Arrival AND #E1_Rotative) OR #FinDesCargaFSS_Auto) AND #CNT_pHsMx_E1.QD AND #TIM_Estabilidad_E1.Q AND #pHsMx_1 AND NOT #Mx_ET01 THEN
       #Mx_ET11 := TRUE;   // SR flip-flop
   END_IF;
   IF #Mx_ET12 THEN #Mx_ET11 := FALSE; END_IF;
END_REGION

REGION Network 62: ET10
   RUNG wire#powerrail
      Contact( #Mx_ET01 )
      Contact( #Selec_E1 )
      I_Contact( #pHsMx_1 )
      I_Contact( #pHsMx_2 )
      I_Contact( #pHsMx_3 )
      I_Contact( #pHsMx_4 )
      Contact( #E1_Rotative )
      I_Contact( #F_EnvMens_Mx )
      Contact( #EstadoZona.Marcha_CBx )
      I_Contact( #EstadoZona.ParoBlando_CBx )
      I_Contact( #EstadoVI.Error_Mx )
      I_Contact( #Error_Tx )
      Contact( #EvolucionEtapasEntrada )
      S_SR(operand := #Mx_ET10, r1 := #Mx_ET11)
   END_RUNG
   // the same network as SCL:
   IF #Mx_ET01 AND #Selec_E1 AND NOT #pHsMx_1 AND NOT #pHsMx_2 AND NOT #pHsMx_3 AND NOT #pHsMx_4 AND #E1_Rotative AND NOT #F_EnvMens_Mx AND #EstadoZona.Marcha_CBx AND NOT #EstadoZona.ParoBlando_CBx AND NOT #EstadoVI.Error_Mx AND NOT #Error_Tx AND #EvolucionEtapasEntrada THEN
       #Mx_ET10 := TRUE;   // SR flip-flop
   END_IF;
   IF #Mx_ET11 THEN #Mx_ET10 := FALSE; END_IF;
END_REGION

REGION Network 63: ET01 - ESTADO REPOSO VACIO
   RUNG wire#powerrail
      Contact( #Mx_ET00 )
      Contact( #EstadoZona.Marcha_CBx )
      I_Contact( #EstadoZona.PerReset_CBx )
      I_Contact( #pHsMx_1 )
      I_Contact( #pHsMx_2 )
      I_Contact( #pHsMx_3 )
      I_Contact( #pHsMx_4 )
      I_Contact( #Selec_E1 )
      I_Contact( #Selec_E2 )
      I_Contact( #Selec_E3 )
      wire#w1
      S_SR(operand := #Mx_ET01, r1 := wire#w2)
   END_RUNG
   RUNG wire#powerrail
      Contact( #Mx_ET61 )
      Contact( #Mx_ET161 )
      I_Contact( #PosSalidaCarga_OK )
      I_Contact( #Simultaneo_Mx )
      I_Contact( #pHsMx_1 )
      I_Contact( #pHsMx_2 )
      I_Contact( #pHsMx_3 )
      I_Contact( #pHsMx_4 )
      I_Contact( #Selec_S4_BPequena )
      I_Contact( #Selec_S4_BGrande )
      I_Contact( #EstadoVI.Descarga_Act )
   END_RUNG wire#w1
   RUNG wire#powerrail
      Contact( #Mx_ET10 )
      Contact( #Mx_ET110_1PRE )
   END_RUNG wire#w2
   RUNG wire#powerrail
      Contact( #Mx_ET20 )
      Contact( #Mx_ET120 )
   END_RUNG wire#w2
   RUNG wire#powerrail
      Contact( #Mx_ET30 )
      Contact( #Mx_ET130_1PRE )
   END_RUNG wire#w2
   // the same network as SCL:
   IF (#Mx_ET00 AND #EstadoZona.Marcha_CBx AND NOT #EstadoZona.PerReset_CBx AND NOT #pHsMx_1 AND NOT #pHsMx_2 AND NOT #pHsMx_3 AND NOT #pHsMx_4 AND NOT #Selec_E1 AND NOT #Selec_E2 AND NOT #Selec_E3) OR (#Mx_ET61 AND #Mx_ET161 AND NOT #PosSalidaCarga_OK AND NOT #Simultaneo_Mx AND NOT #pHsMx_1 AND NOT #pHsMx_2 AND NOT #pHsMx_3 AND NOT #pHsMx_4 AND NOT #Selec_S4_BPequena AND NOT #Selec_S4_BGrande AND NOT #EstadoVI.Descarga_Act) THEN
       #Mx_ET01 := TRUE;   // SR flip-flop
   END_IF;
   IF (#Mx_ET10 AND #Mx_ET110_1PRE) OR (#Mx_ET20 AND #Mx_ET120) OR (#Mx_ET30 AND #Mx_ET130_1PRE) THEN
       #Mx_ET01 := FALSE;
   END_IF;
END_REGION

REGION Network 64: ET00 - ESTADO DE INICIO
   RUNG wire#powerrail
      I_Contact( #Mx_ET60 )
      I_Contact( #Mx_ET61 )
      I_Contact( #Mx_ET160 )
      I_Contact( #Mx_ET161 )
      Coil( #Aux_ET00 )
   END_RUNG
   // the same network as SCL:
   #Aux_ET00 := NOT #Mx_ET60 AND NOT #Mx_ET61 AND NOT #Mx_ET160 AND NOT #Mx_ET161;
END_REGION

REGION Network 65: ---
   RUNG wire#powerrail
      Contact( #Aux_ET00 )
      I_Contact( #Mx_ET10 )
      I_Contact( #Mx_ET11 )
      I_Contact( #Mx_ET12 )
      I_Contact( #Mx_ET110_1PRE )
      I_Contact( #Mx_ET110_1FIN )
      I_Contact( #Mx_ET110_2PRE )
      I_Contact( #Mx_ET110_2FIN )
      I_Contact( #Mx_ET110_3PRE )
      I_Contact( #Mx_ET110_3FIN )
      I_Contact( #Mx_ET110_4PRE )
      I_Contact( #Mx_ET110_4FIN )
      I_Contact( #Mx_ET111 )
      Coil( #Aux_ET00 )
   END_RUNG
   // the same network as SCL:
   #Aux_ET00 := #Aux_ET00 AND NOT #Mx_ET10 AND NOT #Mx_ET11 AND NOT #Mx_ET12 AND NOT #Mx_ET110_1PRE AND NOT #Mx_ET110_1FIN AND NOT #Mx_ET110_2PRE AND NOT #Mx_ET110_2FIN AND NOT #Mx_ET110_3PRE AND NOT #Mx_ET110_3FIN AND NOT #Mx_ET110_4PRE AND NOT #Mx_ET110_4FIN AND NOT #Mx_ET111;
END_REGION

REGION Network 66: ---
   RUNG wire#powerrail
      Contact( #Aux_ET00 )
      I_Contact( #Mx_ET20 )
      I_Contact( #Mx_ET21 )
      I_Contact( #Mx_ET22 )
      I_Contact( #Mx_ET120 )
      I_Contact( #Mx_ET121 )
      Coil( #Aux_ET00 )
   END_RUNG
   // the same network as SCL:
   #Aux_ET00 := #Aux_ET00 AND NOT #Mx_ET20 AND NOT #Mx_ET21 AND NOT #Mx_ET22 AND NOT #Mx_ET120 AND NOT #Mx_ET121;
END_REGION

REGION Network 67: ---
   RUNG wire#powerrail
      Contact( #Aux_ET00 )
      I_Contact( #Mx_ET30 )
      I_Contact( #Mx_ET31 )
      I_Contact( #Mx_ET32 )
      I_Contact( #Mx_ET130_1PRE )
      I_Contact( #Mx_ET130_1FIN )
      I_Contact( #Mx_ET130_2PRE )
      I_Contact( #Mx_ET130_2FIN )
      I_Contact( #Mx_ET130_3PRE )
      I_Contact( #Mx_ET130_3FIN )
      I_Contact( #Mx_ET130_4PRE )
      I_Contact( #Mx_ET130_4FIN )
      I_Contact( #Mx_ET131 )
      Coil( #Aux_ET00 )
   END_RUNG
   // the same network as SCL:
   #Aux_ET00 := #Aux_ET00 AND NOT #Mx_ET30 AND NOT #Mx_ET31 AND NOT #Mx_ET32 AND NOT #Mx_ET130_1PRE AND NOT #Mx_ET130_1FIN AND NOT #Mx_ET130_2PRE AND NOT #Mx_ET130_2FIN AND NOT #Mx_ET130_3PRE AND NOT #Mx_ET130_3FIN AND NOT #Mx_ET130_4PRE AND NOT #Mx_ET130_4FIN AND NOT #Mx_ET131;
END_REGION

REGION Network 68: ---
   RUNG wire#powerrail
      Contact( #Aux_ET00 )
      I_Contact( #Mx_ET08_1PRE )
      I_Contact( #Mx_ET08_1FIN )
      I_Contact( #Mx_ET08_2PRE )
      I_Contact( #Mx_ET08_2FIN )
      I_Contact( #Mx_ET08_3PRE )
      I_Contact( #Mx_ET08_3FIN )
      I_Contact( #Mx_ET08_4PRE )
      I_Contact( #Mx_ET08_4FIN )
      I_Contact( #Mx_ET09 )
      Coil( #Aux_ET00 )
   END_RUNG
   // the same network as SCL:
   #Aux_ET00 := #Aux_ET00 AND NOT #Mx_ET08_1PRE AND NOT #Mx_ET08_1FIN AND NOT #Mx_ET08_2PRE AND NOT #Mx_ET08_2FIN AND NOT #Mx_ET08_3PRE AND NOT #Mx_ET08_3FIN AND NOT #Mx_ET08_4PRE AND NOT #Mx_ET08_4FIN AND NOT #Mx_ET09;
END_REGION

REGION Network 69: ---
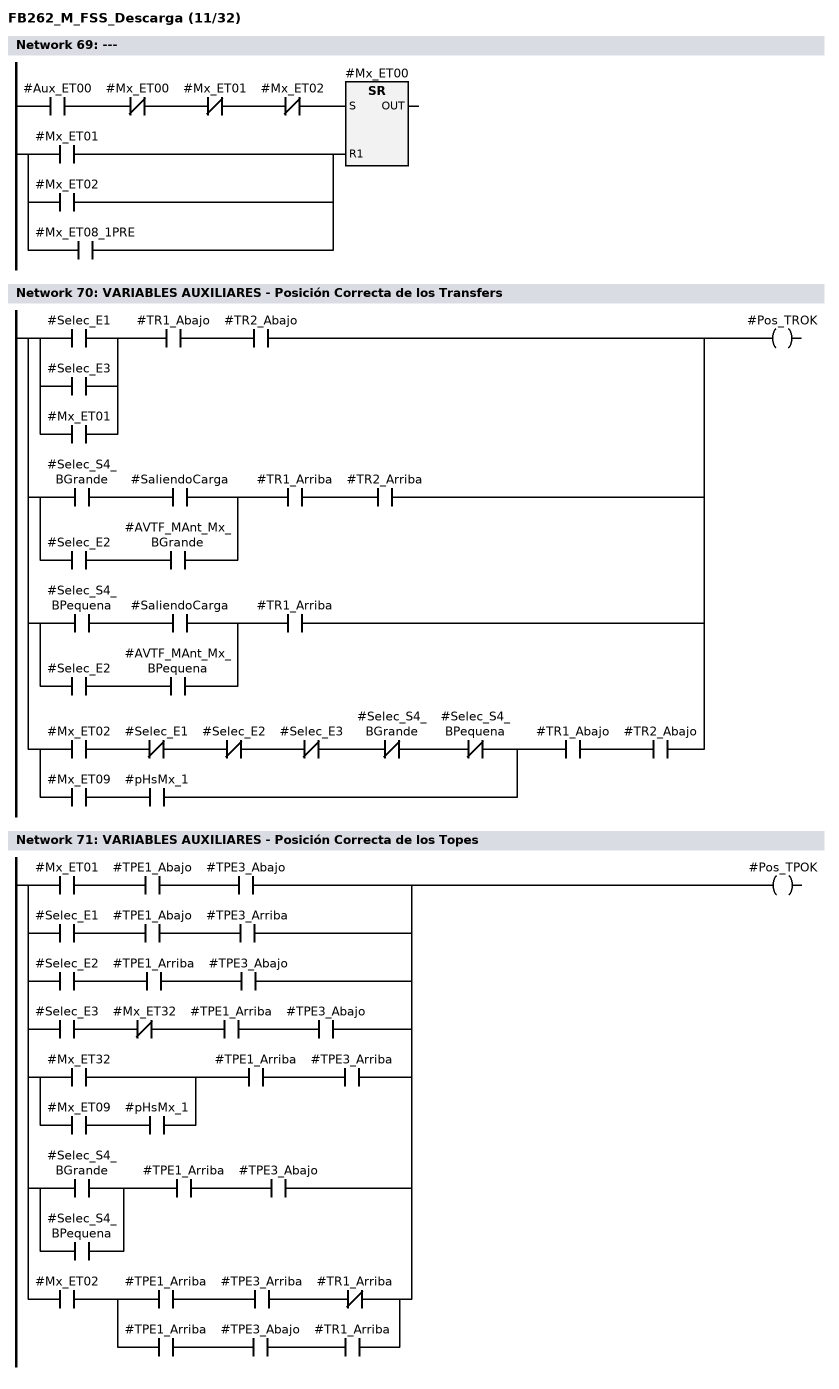
   RUNG wire#powerrail
      Contact( #Aux_ET00 )
      I_Contact( #Mx_ET00 )
      I_Contact( #Mx_ET01 )
      I_Contact( #Mx_ET02 )
      S_SR(operand := #Mx_ET00, r1 := wire#w1)
   END_RUNG
   RUNG wire#powerrail
      Contact( #Mx_ET01 )
   END_RUNG wire#w1
   RUNG wire#powerrail
      Contact( #Mx_ET02 )
   END_RUNG wire#w1
   RUNG wire#powerrail
      Contact( #Mx_ET08_1PRE )
   END_RUNG wire#w1
   // the same network as SCL:
   IF #Aux_ET00 AND NOT #Mx_ET00 AND NOT #Mx_ET01 AND NOT #Mx_ET02 THEN
       #Mx_ET00 := TRUE;   // SR flip-flop
   END_IF;
   IF #Mx_ET01 OR #Mx_ET02 OR #Mx_ET08_1PRE THEN #Mx_ET00 := FALSE; END_IF;
END_REGION

REGION Network 70: VARIABLES AUXILIARES - Posición Correcta de los Transfers
   RUNG wire#powerrail
      Contact( #Selec_E1 )
      wire#w1
      Contact( #TR1_Abajo )
      Contact( #TR2_Abajo )
      wire#w2
      Coil( #Pos_TROK )
   END_RUNG
   RUNG wire#powerrail
      Contact( #Selec_E3 )
   END_RUNG wire#w1
   RUNG wire#powerrail
      Contact( #Mx_ET01 )
   END_RUNG wire#w1
   RUNG wire#powerrail
      Contact( #Selec_S4_BGrande )
      Contact( #SaliendoCarga )
      wire#w3
      Contact( #TR1_Arriba )
      Contact( #TR2_Arriba )
   END_RUNG wire#w2
   RUNG wire#powerrail
      Contact( #Selec_E2 )
      Contact( #AVTF_MAnt_Mx_BGrande )
   END_RUNG wire#w3
   RUNG wire#powerrail
      Contact( #Selec_S4_BPequena )
      Contact( #SaliendoCarga )
      wire#w4
      Contact( #TR1_Arriba )
   END_RUNG wire#w2
   RUNG wire#powerrail
      Contact( #Selec_E2 )
      Contact( #AVTF_MAnt_Mx_BPequena )
   END_RUNG wire#w4
   RUNG wire#powerrail
      Contact( #Mx_ET02 )
      I_Contact( #Selec_E1 )
      I_Contact( #Selec_E2 )
      I_Contact( #Selec_E3 )
      I_Contact( #Selec_S4_BGrande )
      I_Contact( #Selec_S4_BPequena )
      wire#w5
      Contact( #TR1_Abajo )
      Contact( #TR2_Abajo )
   END_RUNG wire#w2
   RUNG wire#powerrail
      Contact( #Mx_ET09 )
      Contact( #pHsMx_1 )
   END_RUNG wire#w5
   // the same network as SCL:
   #Pos_TROK := ((#Selec_E1 OR #Selec_E3 OR #Mx_ET01) AND #TR1_Abajo AND #TR2_Abajo) OR (((#Selec_S4_BGrande AND #SaliendoCarga) OR (#Selec_E2 AND #AVTF_MAnt_Mx_BGrande)) AND #TR1_Arriba AND #TR2_Arriba) OR (((#Selec_S4_BPequena AND #SaliendoCarga) OR (#Selec_E2 AND #AVTF_MAnt_Mx_BPequena)) AND #TR1_Arriba) OR (((#Mx_ET02 AND NOT #Selec_E1 AND NOT #Selec_E2 AND NOT #Selec_E3 AND NOT #Selec_S4_BGrande AND NOT #Selec_S4_BPequena) OR (#Mx_ET09 AND #pHsMx_1)) AND #TR1_Abajo AND #TR2_Abajo);
END_REGION

REGION Network 71: VARIABLES AUXILIARES - Posición Correcta de los Topes
   RUNG wire#powerrail
      Contact( #Mx_ET01 )
      Contact( #TPE1_Abajo )
      Contact( #TPE3_Abajo )
      wire#w1
      Coil( #Pos_TPOK )
   END_RUNG
   RUNG wire#powerrail
      Contact( #Selec_E1 )
      Contact( #TPE1_Abajo )
      Contact( #TPE3_Arriba )
   END_RUNG wire#w1
   RUNG wire#powerrail
      Contact( #Selec_E2 )
      Contact( #TPE1_Arriba )
      Contact( #TPE3_Abajo )
   END_RUNG wire#w1
   RUNG wire#powerrail
      Contact( #Selec_E3 )
      I_Contact( #Mx_ET32 )
      Contact( #TPE1_Arriba )
      Contact( #TPE3_Abajo )
   END_RUNG wire#w1
   RUNG wire#powerrail
      Contact( #Mx_ET32 )
      wire#w2
      Contact( #TPE1_Arriba )
      Contact( #TPE3_Arriba )
   END_RUNG wire#w1
   RUNG wire#powerrail
      Contact( #Mx_ET09 )
      Contact( #pHsMx_1 )
   END_RUNG wire#w2
   RUNG wire#powerrail
      Contact( #Selec_S4_BGrande )
      wire#w3
      Contact( #TPE1_Arriba )
      Contact( #TPE3_Abajo )
   END_RUNG wire#w1
   RUNG wire#powerrail
      Contact( #Selec_S4_BPequena )
   END_RUNG wire#w3
   RUNG wire#powerrail
      Contact( #Mx_ET02 )
      wire#w4
      Contact( #TPE1_Arriba )
      Contact( #TPE3_Arriba )
      I_Contact( #TR1_Arriba )
   END_RUNG wire#w1
   RUNG wire#w4
      Contact( #TPE1_Arriba )
      Contact( #TPE3_Abajo )
      Contact( #TR1_Arriba )
   END_RUNG wire#w1
   // the same network as SCL:
   #Pos_TPOK := (#Mx_ET01 AND #TPE1_Abajo AND #TPE3_Abajo) OR (#Selec_E1 AND #TPE1_Abajo AND #TPE3_Arriba) OR (#Selec_E2 AND #TPE1_Arriba AND #TPE3_Abajo) OR (#Selec_E3 AND NOT #Mx_ET32 AND #TPE1_Arriba AND #TPE3_Abajo) OR ((#Mx_ET32 OR (#Mx_ET09 AND #pHsMx_1)) AND #TPE1_Arriba AND #TPE3_Arriba) OR ((#Selec_S4_BGrande OR #Selec_S4_BPequena) AND #TPE1_Arriba AND #TPE3_Abajo) OR (#Mx_ET02 AND ((#TPE1_Arriba AND #TPE3_Arriba AND NOT #TR1_Arriba) OR (#TPE1_Arriba AND #TPE3_Abajo AND #TR1_Arriba)));
END_REGION

REGION Network 72: VARIABLES AUXILIARES - Memoria >> Entrando Bandeja Grande
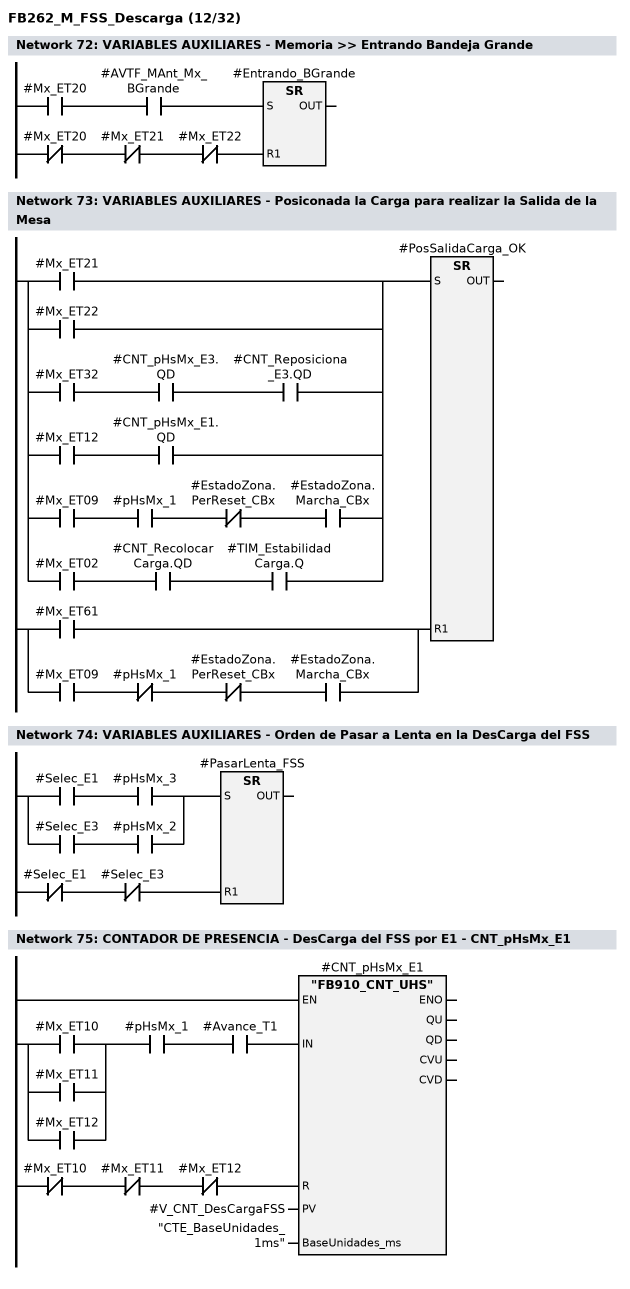
   RUNG wire#powerrail
      Contact( #Mx_ET20 )
      Contact( #AVTF_MAnt_Mx_BGrande )
      S_SR(operand := #Entrando_BGrande, r1 := wire#w1)
   END_RUNG
   RUNG wire#powerrail
      I_Contact( #Mx_ET20 )
      I_Contact( #Mx_ET21 )
      I_Contact( #Mx_ET22 )
   END_RUNG wire#w1
   // the same network as SCL:
   IF #Mx_ET20 AND #AVTF_MAnt_Mx_BGrande THEN
       #Entrando_BGrande := TRUE;   // SR flip-flop
   END_IF;
   IF NOT #Mx_ET20 AND NOT #Mx_ET21 AND NOT #Mx_ET22 THEN #Entrando_BGrande := FALSE; END_IF;
END_REGION

REGION Network 73: VARIABLES AUXILIARES - Posiconada la Carga para realizar la Salida de la Mesa
   RUNG wire#powerrail
      Contact( #Mx_ET21 )
      wire#w1
      S_SR(operand := #PosSalidaCarga_OK, r1 := wire#w2)
   END_RUNG
   RUNG wire#powerrail
      Contact( #Mx_ET22 )
   END_RUNG wire#w1
   RUNG wire#powerrail
      Contact( #Mx_ET32 )
      Contact( #CNT_pHsMx_E3.QD )
      Contact( #CNT_Reposiciona_E3.QD )
   END_RUNG wire#w1
   RUNG wire#powerrail
      Contact( #Mx_ET12 )
      Contact( #CNT_pHsMx_E1.QD )
   END_RUNG wire#w1
   RUNG wire#powerrail
      Contact( #Mx_ET09 )
      Contact( #pHsMx_1 )
      I_Contact( #EstadoZona.PerReset_CBx )
      Contact( #EstadoZona.Marcha_CBx )
   END_RUNG wire#w1
   RUNG wire#powerrail
      Contact( #Mx_ET02 )
      Contact( #CNT_RecolocarCarga.QD )
      Contact( #TIM_EstabilidadCarga.Q )
   END_RUNG wire#w1
   RUNG wire#powerrail
      Contact( #Mx_ET61 )
   END_RUNG wire#w2
   RUNG wire#powerrail
      Contact( #Mx_ET09 )
      I_Contact( #pHsMx_1 )
      I_Contact( #EstadoZona.PerReset_CBx )
      Contact( #EstadoZona.Marcha_CBx )
   END_RUNG wire#w2
   // the same network as SCL:
   IF #Mx_ET21 OR #Mx_ET22 OR (#Mx_ET32 AND #CNT_pHsMx_E3.QD AND #CNT_Reposiciona_E3.QD) OR (#Mx_ET12 AND #CNT_pHsMx_E1.QD) OR (#Mx_ET09 AND #pHsMx_1 AND NOT #EstadoZona.PerReset_CBx AND #EstadoZona.Marcha_CBx) OR (#Mx_ET02 AND #CNT_RecolocarCarga.QD AND #TIM_EstabilidadCarga.Q) THEN
       #PosSalidaCarga_OK := TRUE;   // SR flip-flop
   END_IF;
   IF #Mx_ET61 OR (#Mx_ET09 AND NOT #pHsMx_1 AND NOT #EstadoZona.PerReset_CBx AND #EstadoZona.Marcha_CBx) THEN
       #PosSalidaCarga_OK := FALSE;
   END_IF;
END_REGION

REGION Network 74: VARIABLES AUXILIARES - Orden de Pasar a Lenta en la DesCarga del FSS
   RUNG wire#powerrail
      Contact( #Selec_E1 )
      Contact( #pHsMx_3 )
      wire#w1
      S_SR(operand := #PasarLenta_FSS, r1 := wire#w2)
   END_RUNG
   RUNG wire#powerrail
      Contact( #Selec_E3 )
      Contact( #pHsMx_2 )
   END_RUNG wire#w1
   RUNG wire#powerrail
      I_Contact( #Selec_E1 )
      I_Contact( #Selec_E3 )
   END_RUNG wire#w2
   // the same network as SCL:
   IF (#Selec_E1 AND #pHsMx_3) OR (#Selec_E3 AND #pHsMx_2) THEN
       #PasarLenta_FSS := TRUE;   // SR flip-flop
   END_IF;
   IF NOT #Selec_E1 AND NOT #Selec_E3 THEN #PasarLenta_FSS := FALSE; END_IF;
END_REGION

REGION Network 75: CONTADOR DE PRESENCIA - DesCarga del FSS por E1 - CNT_pHsMx_E1
   RUNG wire#powerrail
      #CNT_pHsMx_E1(IN := wire#w2, R := wire#w3, PV := #V_CNT_DesCargaFSS, BaseUnidades_ms := "CTE_BaseUnidades_1ms", QU =>, QD =>, CVU =>, CVD =>)
   END_RUNG
   RUNG wire#powerrail
      Contact( #Mx_ET10 )
      wire#w1
      Contact( #pHsMx_1 )
      Contact( #Avance_T1 )
   END_RUNG wire#w2
   RUNG wire#powerrail
      Contact( #Mx_ET11 )
   END_RUNG wire#w1
   RUNG wire#powerrail
      Contact( #Mx_ET12 )
   END_RUNG wire#w1
   RUNG wire#powerrail
      I_Contact( #Mx_ET10 )
      I_Contact( #Mx_ET11 )
      I_Contact( #Mx_ET12 )
   END_RUNG wire#w3
   // the same network as SCL:
   #CNT_pHsMx_E1(IN := (#Mx_ET10 OR #Mx_ET11 OR #Mx_ET12) AND #pHsMx_1 AND #Avance_T1,   // "FB910_CNT_UHS"
                 R := NOT #Mx_ET10 AND NOT #Mx_ET11 AND NOT #Mx_ET12,
                 PV := #V_CNT_DesCargaFSS,
                 BaseUnidades_ms := "CTE_BaseUnidades_1ms");
END_REGION

REGION Network 76: TIM DE ESTABILIDAD DE CARGA - DesCarga del FSS por E1 - TIM_Estabilidad_E1
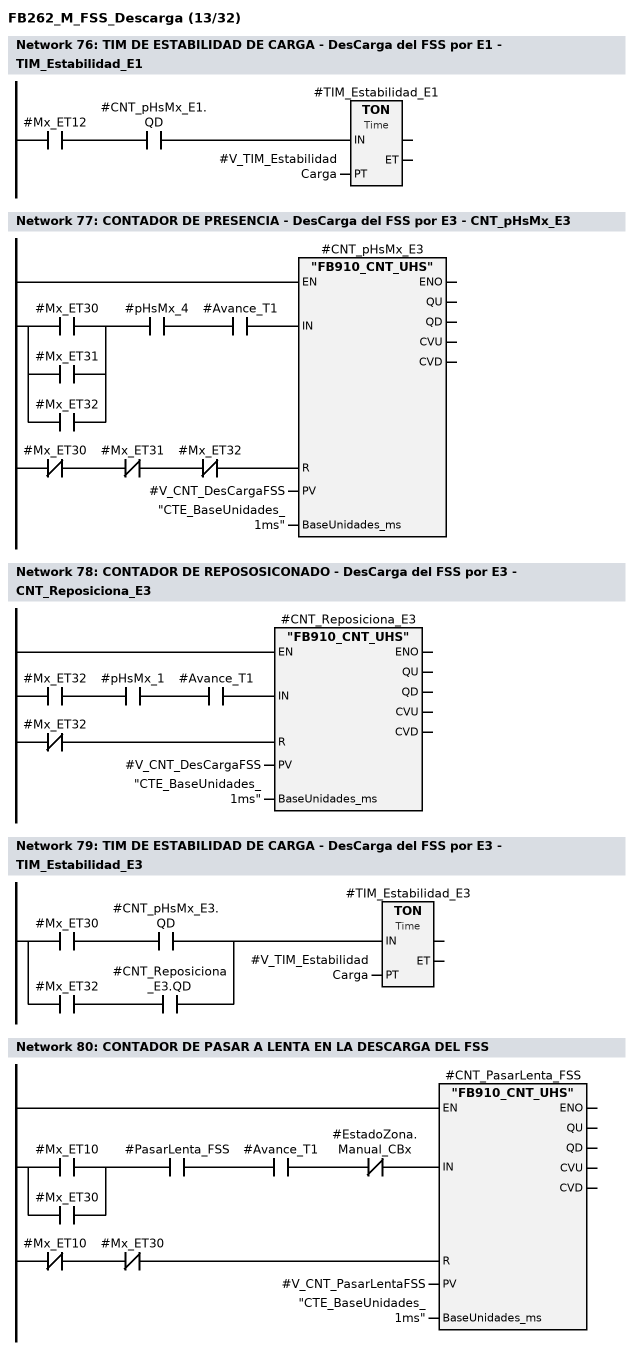
   RUNG wire#powerrail
      Contact( #Mx_ET12 )
      Contact( #CNT_pHsMx_E1.QD )
      { S7_Templates := "time_type := Time" } #TIM_Estabilidad_E1.TON(pt := #V_TIM_EstabilidadCarga, et =>)
   END_RUNG
   // the same network as SCL:
   #TIM_Estabilidad_E1(IN := #Mx_ET12 AND #CNT_pHsMx_E1.QD, PT := #V_TIM_EstabilidadCarga);   // TON
END_REGION

REGION Network 77: CONTADOR DE PRESENCIA - DesCarga del FSS por E3 - CNT_pHsMx_E3
   RUNG wire#powerrail
      #CNT_pHsMx_E3(IN := wire#w2, R := wire#w3, PV := #V_CNT_DesCargaFSS, BaseUnidades_ms := "CTE_BaseUnidades_1ms", QU =>, QD =>, CVU =>, CVD =>)
   END_RUNG
   RUNG wire#powerrail
      Contact( #Mx_ET30 )
      wire#w1
      Contact( #pHsMx_4 )
      Contact( #Avance_T1 )
   END_RUNG wire#w2
   RUNG wire#powerrail
      Contact( #Mx_ET31 )
   END_RUNG wire#w1
   RUNG wire#powerrail
      Contact( #Mx_ET32 )
   END_RUNG wire#w1
   RUNG wire#powerrail
      I_Contact( #Mx_ET30 )
      I_Contact( #Mx_ET31 )
      I_Contact( #Mx_ET32 )
   END_RUNG wire#w3
   // the same network as SCL:
   #CNT_pHsMx_E3(IN := (#Mx_ET30 OR #Mx_ET31 OR #Mx_ET32) AND #pHsMx_4 AND #Avance_T1,   // "FB910_CNT_UHS"
                 R := NOT #Mx_ET30 AND NOT #Mx_ET31 AND NOT #Mx_ET32,
                 PV := #V_CNT_DesCargaFSS,
                 BaseUnidades_ms := "CTE_BaseUnidades_1ms");
END_REGION

REGION Network 78: CONTADOR DE REPOSOSICONADO - DesCarga del FSS por E3 - CNT_Reposiciona_E3
   RUNG wire#powerrail
      #CNT_Reposiciona_E3(IN := wire#w1, R := wire#w2, PV := #V_CNT_DesCargaFSS, BaseUnidades_ms := "CTE_BaseUnidades_1ms", QU =>, QD =>, CVU =>, CVD =>)
   END_RUNG
   RUNG wire#powerrail
      Contact( #Mx_ET32 )
      Contact( #pHsMx_1 )
      Contact( #Avance_T1 )
   END_RUNG wire#w1
   RUNG wire#powerrail
      I_Contact( #Mx_ET32 )
   END_RUNG wire#w2
   // the same network as SCL:
   #CNT_Reposiciona_E3(IN := #Mx_ET32 AND #pHsMx_1 AND #Avance_T1,   // "FB910_CNT_UHS"
                       R := NOT #Mx_ET32,
                       PV := #V_CNT_DesCargaFSS,
                       BaseUnidades_ms := "CTE_BaseUnidades_1ms");
END_REGION

REGION Network 79: TIM DE ESTABILIDAD DE CARGA - DesCarga del FSS por E3 - TIM_Estabilidad_E3
   RUNG wire#powerrail
      Contact( #Mx_ET30 )
      Contact( #CNT_pHsMx_E3.QD )
      wire#w1
      { S7_Templates := "time_type := Time" } #TIM_Estabilidad_E3.TON(pt := #V_TIM_EstabilidadCarga, et =>)
   END_RUNG
   RUNG wire#powerrail
      Contact( #Mx_ET32 )
      Contact( #CNT_Reposiciona_E3.QD )
   END_RUNG wire#w1
   // the same network as SCL:
   #TIM_Estabilidad_E3(IN := (#Mx_ET30 AND #CNT_pHsMx_E3.QD) OR (#Mx_ET32 AND #CNT_Reposiciona_E3.QD),   // TON
                       PT := #V_TIM_EstabilidadCarga);
END_REGION

REGION Network 80: CONTADOR DE PASAR A LENTA EN LA DESCARGA DEL FSS
   RUNG wire#powerrail
      #CNT_PasarLenta_FSS(IN := wire#w2, R := wire#w3, PV := #V_CNT_PasarLentaFSS, BaseUnidades_ms := "CTE_BaseUnidades_1ms", QU =>, QD =>, CVU =>, CVD =>)
   END_RUNG
   RUNG wire#powerrail
      Contact( #Mx_ET10 )
      wire#w1
      Contact( #PasarLenta_FSS )
      Contact( #Avance_T1 )
      I_Contact( #EstadoZona.Manual_CBx )
   END_RUNG wire#w2
   RUNG wire#powerrail
      Contact( #Mx_ET30 )
   END_RUNG wire#w1
   RUNG wire#powerrail
      I_Contact( #Mx_ET10 )
      I_Contact( #Mx_ET30 )
   END_RUNG wire#w3
   // the same network as SCL:
   #CNT_PasarLenta_FSS(IN := (#Mx_ET10 OR #Mx_ET30) AND #PasarLenta_FSS AND #Avance_T1 AND NOT #EstadoZona.Manual_CBx,   // "FB910_CNT_UHS"
                       R := NOT #Mx_ET10 AND NOT #Mx_ET30,
                       PV := #V_CNT_PasarLentaFSS,
                       BaseUnidades_ms := "CTE_BaseUnidades_1ms");
END_REGION

REGION Network 81: CONTADOR DE SEGURIDAD DE PRESENCIA - CNTSeg_pHsMx_E2
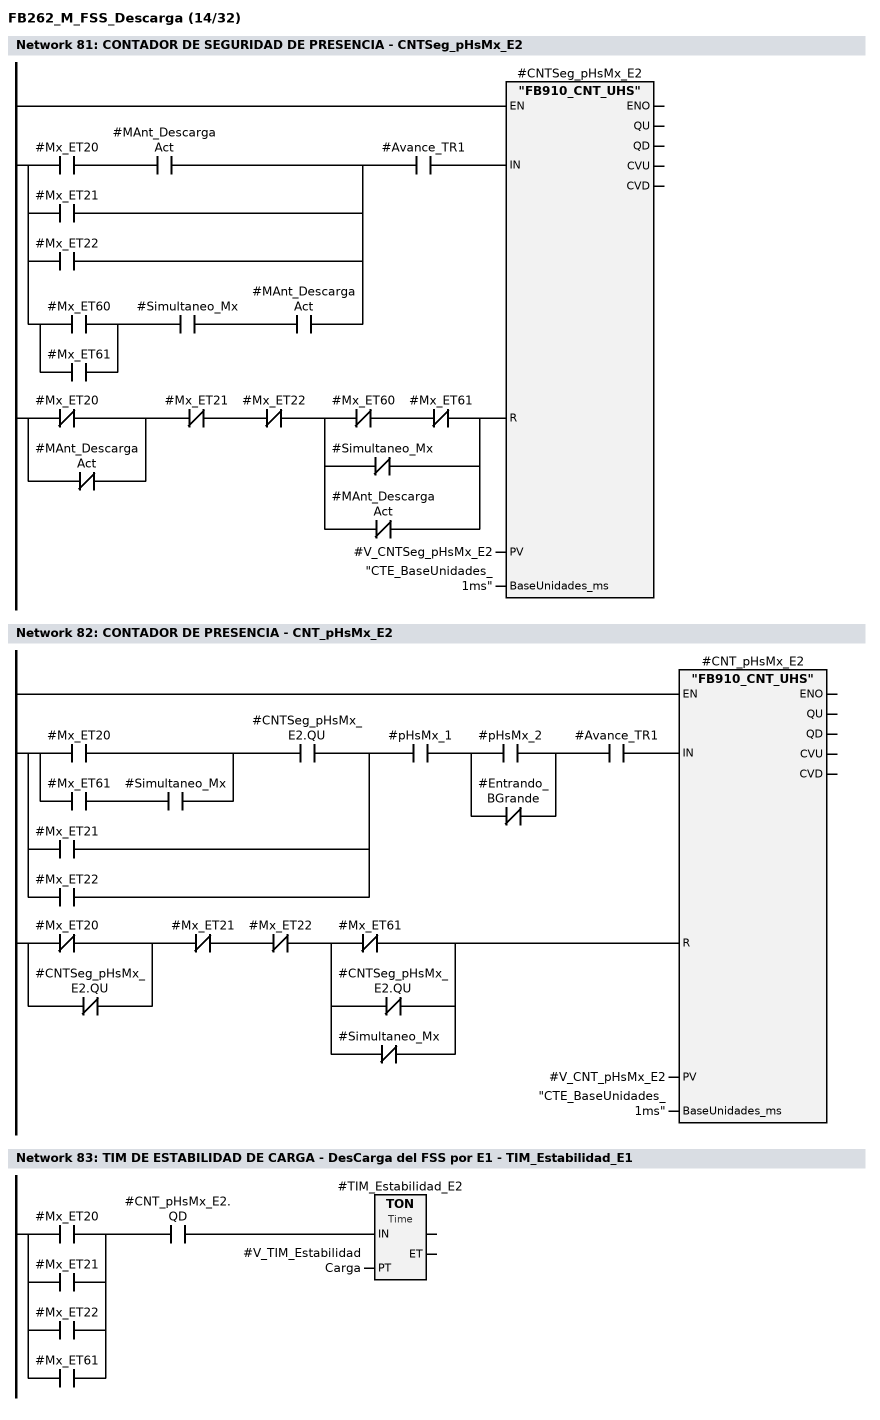
   RUNG wire#powerrail
      #CNTSeg_pHsMx_E2(IN := wire#w3, R := wire#w6, PV := #V_CNTSeg_pHsMx_E2, BaseUnidades_ms := "CTE_BaseUnidades_1ms", QU =>, QD =>, CVU =>, CVD =>)
   END_RUNG
   RUNG wire#powerrail
      Contact( #Mx_ET20 )
      Contact( #MAnt_DescargaAct )
      wire#w1
      Contact( #Avance_TR1 )
   END_RUNG wire#w3
   RUNG wire#powerrail
      Contact( #Mx_ET21 )
   END_RUNG wire#w1
   RUNG wire#powerrail
      Contact( #Mx_ET22 )
   END_RUNG wire#w1
   RUNG wire#powerrail
      Contact( #Mx_ET60 )
      wire#w2
      Contact( #Simultaneo_Mx )
      Contact( #MAnt_DescargaAct )
   END_RUNG wire#w1
   RUNG wire#powerrail
      Contact( #Mx_ET61 )
   END_RUNG wire#w2
   RUNG wire#powerrail
      I_Contact( #Mx_ET20 )
      wire#w4
      I_Contact( #Mx_ET21 )
      I_Contact( #Mx_ET22 )
      wire#w5
      I_Contact( #Mx_ET60 )
      I_Contact( #Mx_ET61 )
   END_RUNG wire#w6
   RUNG wire#powerrail
      I_Contact( #MAnt_DescargaAct )
   END_RUNG wire#w4
   RUNG wire#w5
      I_Contact( #Simultaneo_Mx )
   END_RUNG wire#w6
   RUNG wire#w5
      I_Contact( #MAnt_DescargaAct )
   END_RUNG wire#w6
   // the same network as SCL:
   #CNTSeg_pHsMx_E2(IN := ((#Mx_ET20 AND #MAnt_DescargaAct) OR #Mx_ET21 OR #Mx_ET22 OR ((#Mx_ET60 OR #Mx_ET61) AND #Simultaneo_Mx AND #MAnt_DescargaAct)) AND #Avance_TR1,   // "FB910_CNT_UHS"
                    R := (NOT #Mx_ET20 OR NOT #MAnt_DescargaAct) AND NOT #Mx_ET21 AND NOT #Mx_ET22 AND ((NOT #Mx_ET60 AND NOT #Mx_ET61) OR NOT #Simultaneo_Mx OR NOT #MAnt_DescargaAct),
                    PV := #V_CNTSeg_pHsMx_E2,
                    BaseUnidades_ms := "CTE_BaseUnidades_1ms");
END_REGION

REGION Network 82: CONTADOR DE PRESENCIA - CNT_pHsMx_E2
   RUNG wire#powerrail
      #CNT_pHsMx_E2(IN := wire#w5, R := wire#w8, PV := #V_CNT_pHsMx_E2, BaseUnidades_ms := "CTE_BaseUnidades_1ms", QU =>, QD =>, CVU =>, CVD =>)
   END_RUNG
   RUNG wire#powerrail
      Contact( #Mx_ET20 )
      wire#w1
      Contact( #CNTSeg_pHsMx_E2.QU )
      wire#w2
      Contact( #pHsMx_1 )
      wire#w3
      Contact( #pHsMx_2 )
      wire#w4
      Contact( #Avance_TR1 )
   END_RUNG wire#w5
   RUNG wire#powerrail
      Contact( #Mx_ET61 )
      Contact( #Simultaneo_Mx )
   END_RUNG wire#w1
   RUNG wire#powerrail
      Contact( #Mx_ET21 )
   END_RUNG wire#w2
   RUNG wire#powerrail
      Contact( #Mx_ET22 )
   END_RUNG wire#w2
   RUNG wire#w3
      I_Contact( #Entrando_BGrande )
   END_RUNG wire#w4
   RUNG wire#powerrail
      I_Contact( #Mx_ET20 )
      wire#w6
      I_Contact( #Mx_ET21 )
      I_Contact( #Mx_ET22 )
      wire#w7
      I_Contact( #Mx_ET61 )
   END_RUNG wire#w8
   RUNG wire#powerrail
      I_Contact( #CNTSeg_pHsMx_E2.QU )
   END_RUNG wire#w6
   RUNG wire#w7
      I_Contact( #CNTSeg_pHsMx_E2.QU )
   END_RUNG wire#w8
   RUNG wire#w7
      I_Contact( #Simultaneo_Mx )
   END_RUNG wire#w8
   // the same network as SCL:
   #CNT_pHsMx_E2(IN := (((#Mx_ET20 OR (#Mx_ET61 AND #Simultaneo_Mx)) AND #CNTSeg_pHsMx_E2.QU) OR #Mx_ET21 OR #Mx_ET22) AND #pHsMx_1 AND (#pHsMx_2 OR NOT #Entrando_BGrande) AND #Avance_TR1,   // "FB910_CNT_UHS"
                 R := (NOT #Mx_ET20 OR NOT #CNTSeg_pHsMx_E2.QU) AND NOT #Mx_ET21 AND NOT #Mx_ET22 AND (NOT #Mx_ET61 OR NOT #CNTSeg_pHsMx_E2.QU OR NOT #Simultaneo_Mx),
                 PV := #V_CNT_pHsMx_E2,
                 BaseUnidades_ms := "CTE_BaseUnidades_1ms");
END_REGION

REGION Network 83: TIM DE ESTABILIDAD DE CARGA - DesCarga del FSS por E1 - TIM_Estabilidad_E1
   RUNG wire#powerrail
      Contact( #Mx_ET20 )
      wire#w1
      Contact( #CNT_pHsMx_E2.QD )
      { S7_Templates := "time_type := Time" } #TIM_Estabilidad_E2.TON(pt := #V_TIM_EstabilidadCarga, et =>)
   END_RUNG
   RUNG wire#powerrail
      Contact( #Mx_ET21 )
   END_RUNG wire#w1
   RUNG wire#powerrail
      Contact( #Mx_ET22 )
   END_RUNG wire#w1
   RUNG wire#powerrail
      Contact( #Mx_ET61 )
   END_RUNG wire#w1
   // the same network as SCL:
   #TIM_Estabilidad_E2(IN := (#Mx_ET20 OR #Mx_ET21 OR #Mx_ET22 OR #Mx_ET61) AND #CNT_pHsMx_E2.QD,   // TON
                       PT := #V_TIM_EstabilidadCarga);
END_REGION

REGION Network 84: DETERMINA PASO ET20 - ET21 (Nota: Control de Tiempo para dar el FTF a la Mesa Anterior)
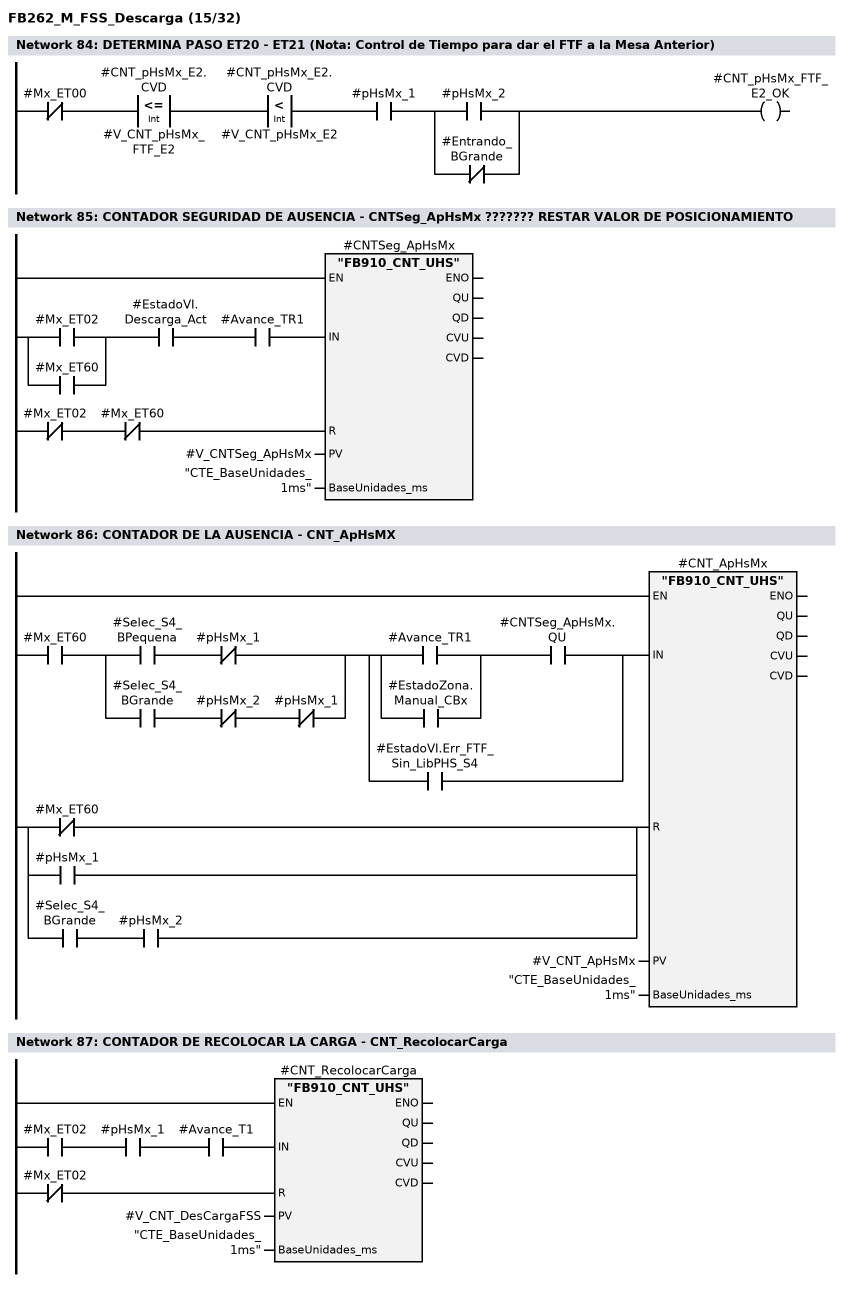
   RUNG wire#powerrail
      I_Contact( #Mx_ET00 )
      { S7_Templates := "SrcType := Int" } LE_Contact(in1 := #CNT_pHsMx_E2.CVD, in2 := #V_CNT_pHsMx_FTF_E2)
      { S7_Templates := "SrcType := Int" } LT_Contact(in1 := #CNT_pHsMx_E2.CVD, in2 := #V_CNT_pHsMx_E2)
      Contact( #pHsMx_1 )
      wire#w1
      Contact( #pHsMx_2 )
      wire#w2
      Coil( #CNT_pHsMx_FTF_E2_OK )
   END_RUNG
   RUNG wire#w1
      I_Contact( #Entrando_BGrande )
   END_RUNG wire#w2
   // the same network as SCL:
   #CNT_pHsMx_FTF_E2_OK := NOT #Mx_ET00 AND (#CNT_pHsMx_E2.CVD <= #V_CNT_pHsMx_FTF_E2) AND (#CNT_pHsMx_E2.CVD < #V_CNT_pHsMx_E2) AND #pHsMx_1 AND (#pHsMx_2 OR NOT #Entrando_BGrande);
END_REGION

REGION Network 85: CONTADOR SEGURIDAD DE AUSENCIA - CNTSeg_ApHsMx ??????? RESTAR VALOR DE POSICIONAMIENTO
   RUNG wire#powerrail
      #CNTSeg_ApHsMx(IN := wire#w2, R := wire#w3, PV := #V_CNTSeg_ApHsMx, BaseUnidades_ms := "CTE_BaseUnidades_1ms", QU =>, QD =>, CVU =>, CVD =>)
   END_RUNG
   RUNG wire#powerrail
      Contact( #Mx_ET02 )
      wire#w1
      Contact( #EstadoVI.Descarga_Act )
      Contact( #Avance_TR1 )
   END_RUNG wire#w2
   RUNG wire#powerrail
      Contact( #Mx_ET60 )
   END_RUNG wire#w1
   RUNG wire#powerrail
      I_Contact( #Mx_ET02 )
      I_Contact( #Mx_ET60 )
   END_RUNG wire#w3
   // the same network as SCL:
   #CNTSeg_ApHsMx(IN := (#Mx_ET02 OR #Mx_ET60) AND #EstadoVI.Descarga_Act AND #Avance_TR1,   // "FB910_CNT_UHS"
                  R := NOT #Mx_ET02 AND NOT #Mx_ET60,
                  PV := #V_CNTSeg_ApHsMx,
                  BaseUnidades_ms := "CTE_BaseUnidades_1ms");
END_REGION

REGION Network 86: CONTADOR DE LA AUSENCIA - CNT_ApHsMX
   RUNG wire#powerrail
      #CNT_ApHsMx(IN := wire#w4, R := wire#w5, PV := #V_CNT_ApHsMx, BaseUnidades_ms := "CTE_BaseUnidades_1ms", QU =>, QD =>, CVU =>, CVD =>)
   END_RUNG
   RUNG wire#powerrail
      Contact( #Mx_ET60 )
      wire#w1
      Contact( #Selec_S4_BPequena )
      I_Contact( #pHsMx_1 )
      wire#w2
      Contact( #Avance_TR1 )
      wire#w3
      Contact( #CNTSeg_ApHsMx.QU )
   END_RUNG wire#w4
   RUNG wire#w1
      Contact( #Selec_S4_BGrande )
      I_Contact( #pHsMx_2 )
      I_Contact( #pHsMx_1 )
   END_RUNG wire#w2
   RUNG wire#w2
      Contact( #EstadoZona.Manual_CBx )
   END_RUNG wire#w3
   RUNG wire#w2
      Contact( #EstadoVI.Err_FTF_Sin_LibPHS_S4 )
   END_RUNG wire#w4
   RUNG wire#powerrail
      I_Contact( #Mx_ET60 )
   END_RUNG wire#w5
   RUNG wire#powerrail
      Contact( #pHsMx_1 )
   END_RUNG wire#w5
   RUNG wire#powerrail
      Contact( #Selec_S4_BGrande )
      Contact( #pHsMx_2 )
   END_RUNG wire#w5
   // the same network as SCL:
   #CNT_ApHsMx(IN := #Mx_ET60 AND ((#Selec_S4_BPequena AND NOT #pHsMx_1) OR (#Selec_S4_BGrande AND NOT #pHsMx_2 AND NOT #pHsMx_1)) AND (((#Avance_TR1 OR #EstadoZona.Manual_CBx) AND #CNTSeg_ApHsMx.QU) OR #EstadoVI.Err_FTF_Sin_LibPHS_S4),   // "FB910_CNT_UHS"
               R := NOT #Mx_ET60 OR #pHsMx_1 OR (#Selec_S4_BGrande AND #pHsMx_2),
               PV := #V_CNT_ApHsMx,
               BaseUnidades_ms := "CTE_BaseUnidades_1ms");
END_REGION

REGION Network 87: CONTADOR DE RECOLOCAR LA CARGA - CNT_RecolocarCarga
   RUNG wire#powerrail
      #CNT_RecolocarCarga(IN := wire#w1, R := wire#w2, PV := #V_CNT_DesCargaFSS, BaseUnidades_ms := "CTE_BaseUnidades_1ms", QU =>, QD =>, CVU =>, CVD =>)
   END_RUNG
   RUNG wire#powerrail
      Contact( #Mx_ET02 )
      Contact( #pHsMx_1 )
      Contact( #Avance_T1 )
   END_RUNG wire#w1
   RUNG wire#powerrail
      I_Contact( #Mx_ET02 )
   END_RUNG wire#w2
   // the same network as SCL:
   #CNT_RecolocarCarga(IN := #Mx_ET02 AND #pHsMx_1 AND #Avance_T1,   // "FB910_CNT_UHS"
                       R := NOT #Mx_ET02,
                       PV := #V_CNT_DesCargaFSS,
                       BaseUnidades_ms := "CTE_BaseUnidades_1ms");
END_REGION

REGION Network 88: TIM DE ESTABILIDAD DE CARGA - Recolocacion de la Carga - TIM_EstabilidadCarga
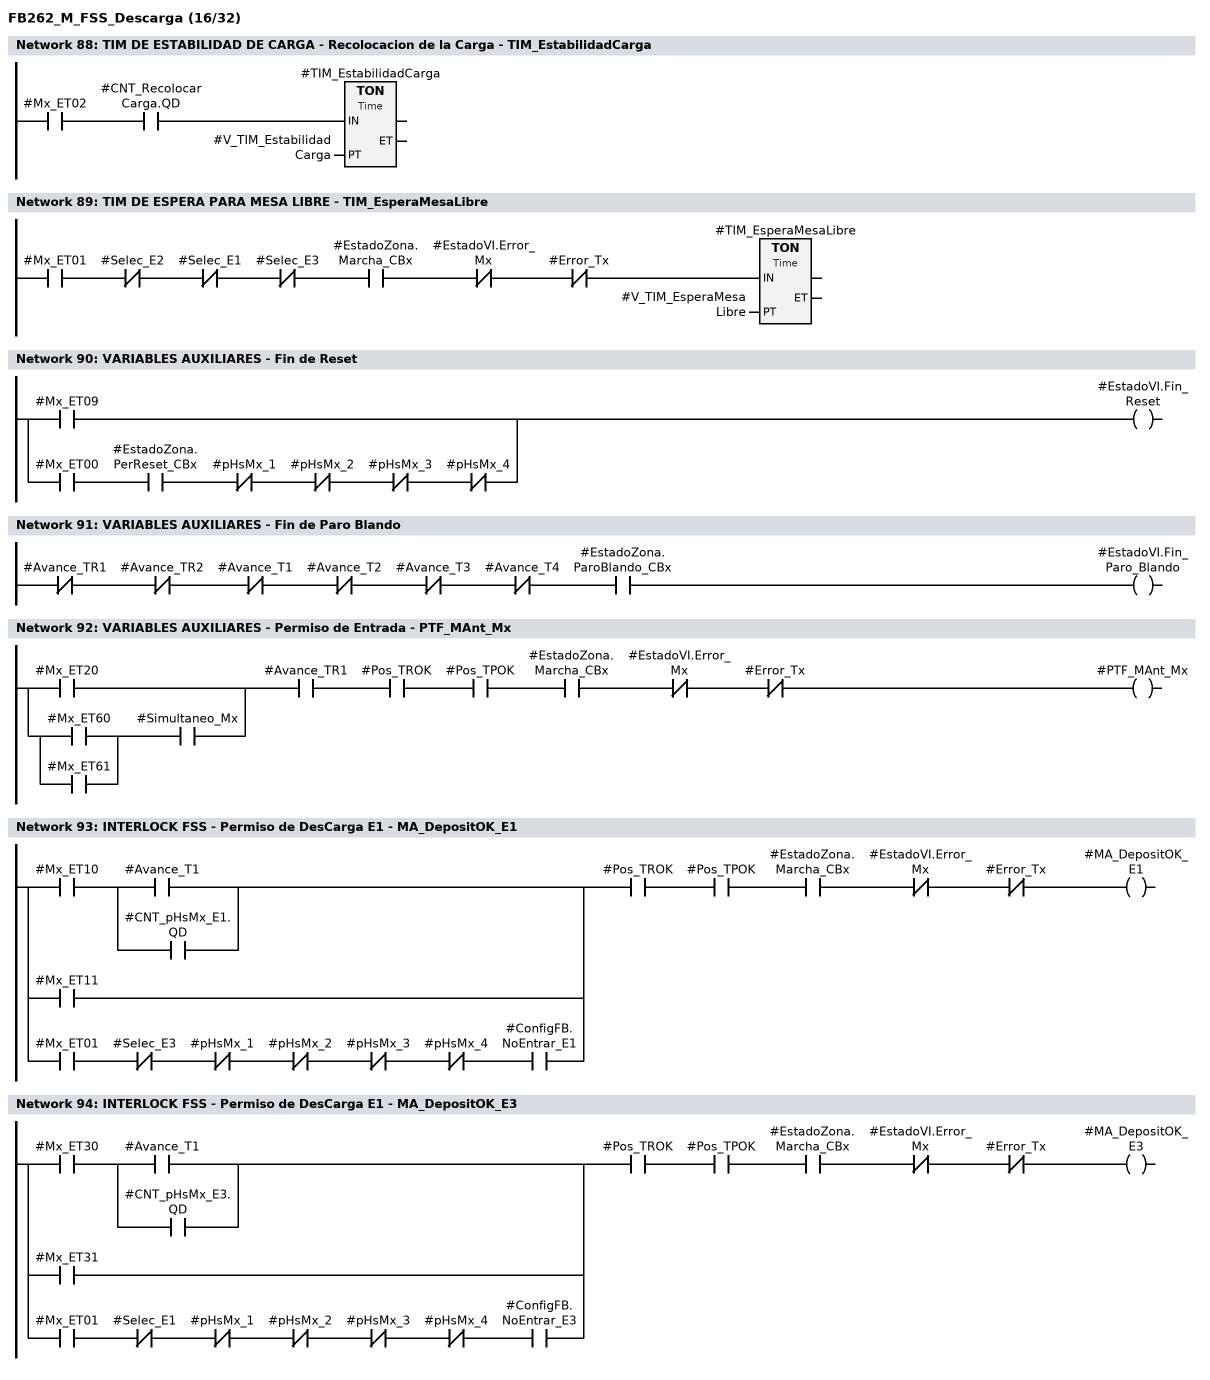
   RUNG wire#powerrail
      Contact( #Mx_ET02 )
      Contact( #CNT_RecolocarCarga.QD )
      { S7_Templates := "time_type := Time" } #TIM_EstabilidadCarga.TON(pt := #V_TIM_EstabilidadCarga, et =>)
   END_RUNG
   // the same network as SCL:
   #TIM_EstabilidadCarga(IN := #Mx_ET02 AND #CNT_RecolocarCarga.QD, PT := #V_TIM_EstabilidadCarga);   // TON
END_REGION

REGION Network 89: TIM DE ESPERA PARA MESA LIBRE - TIM_EsperaMesaLibre
   RUNG wire#powerrail
      Contact( #Mx_ET01 )
      I_Contact( #Selec_E2 )
      I_Contact( #Selec_E1 )
      I_Contact( #Selec_E3 )
      Contact( #EstadoZona.Marcha_CBx )
      I_Contact( #EstadoVI.Error_Mx )
      I_Contact( #Error_Tx )
      { S7_Templates := "time_type := Time" } #TIM_EsperaMesaLibre.TON(pt := #V_TIM_EsperaMesaLibre, et =>)
   END_RUNG
   // the same network as SCL:
   #TIM_EsperaMesaLibre(IN := #Mx_ET01 AND NOT #Selec_E2 AND NOT #Selec_E1 AND NOT #Selec_E3 AND #EstadoZona.Marcha_CBx AND NOT #EstadoVI.Error_Mx AND NOT #Error_Tx,   // TON
                        PT := #V_TIM_EsperaMesaLibre);
END_REGION

REGION Network 90: VARIABLES AUXILIARES - Fin de Reset
   RUNG wire#powerrail
      Contact( #Mx_ET09 )
      wire#w1
      Coil( #EstadoVI.Fin_Reset )
   END_RUNG
   RUNG wire#powerrail
      Contact( #Mx_ET00 )
      Contact( #EstadoZona.PerReset_CBx )
      I_Contact( #pHsMx_1 )
      I_Contact( #pHsMx_2 )
      I_Contact( #pHsMx_3 )
      I_Contact( #pHsMx_4 )
   END_RUNG wire#w1
   // the same network as SCL:
   #EstadoVI.Fin_Reset := #Mx_ET09 OR (#Mx_ET00 AND #EstadoZona.PerReset_CBx AND NOT #pHsMx_1 AND NOT #pHsMx_2 AND NOT #pHsMx_3 AND NOT #pHsMx_4);
END_REGION

REGION Network 91: VARIABLES AUXILIARES - Fin de Paro Blando
   RUNG wire#powerrail
      I_Contact( #Avance_TR1 )
      I_Contact( #Avance_TR2 )
      I_Contact( #Avance_T1 )
      I_Contact( #Avance_T2 )
      I_Contact( #Avance_T3 )
      I_Contact( #Avance_T4 )
      Contact( #EstadoZona.ParoBlando_CBx )
      Coil( #EstadoVI.Fin_Paro_Blando )
   END_RUNG
   // the same network as SCL:
   #EstadoVI.Fin_Paro_Blando := NOT #Avance_TR1 AND NOT #Avance_TR2 AND NOT #Avance_T1 AND NOT #Avance_T2 AND NOT #Avance_T3 AND NOT #Avance_T4 AND #EstadoZona.ParoBlando_CBx;
END_REGION

REGION Network 92: VARIABLES AUXILIARES - Permiso de Entrada - PTF_MAnt_Mx
   RUNG wire#powerrail
      Contact( #Mx_ET20 )
      wire#w1
      Contact( #Avance_TR1 )
      Contact( #Pos_TROK )
      Contact( #Pos_TPOK )
      Contact( #EstadoZona.Marcha_CBx )
      I_Contact( #EstadoVI.Error_Mx )
      I_Contact( #Error_Tx )
      Coil( #PTF_MAnt_Mx )
   END_RUNG
   RUNG wire#powerrail
      Contact( #Mx_ET60 )
      wire#w2
      Contact( #Simultaneo_Mx )
   END_RUNG wire#w1
   RUNG wire#powerrail
      Contact( #Mx_ET61 )
   END_RUNG wire#w2
   // the same network as SCL:
   #PTF_MAnt_Mx := (#Mx_ET20 OR ((#Mx_ET60 OR #Mx_ET61) AND #Simultaneo_Mx)) AND #Avance_TR1 AND #Pos_TROK AND #Pos_TPOK AND #EstadoZona.Marcha_CBx AND NOT #EstadoVI.Error_Mx AND NOT #Error_Tx;
END_REGION

REGION Network 93: INTERLOCK FSS - Permiso de DesCarga E1 - MA_DepositOK_E1
   RUNG wire#powerrail
      Contact( #Mx_ET10 )
      wire#w1
      Contact( #Avance_T1 )
      wire#w2
      Contact( #Pos_TROK )
      Contact( #Pos_TPOK )
      Contact( #EstadoZona.Marcha_CBx )
      I_Contact( #EstadoVI.Error_Mx )
      I_Contact( #Error_Tx )
      Coil( #MA_DepositOK_E1 )
   END_RUNG
   RUNG wire#w1
      Contact( #CNT_pHsMx_E1.QD )
   END_RUNG wire#w2
   RUNG wire#powerrail
      Contact( #Mx_ET11 )
   END_RUNG wire#w2
   RUNG wire#powerrail
      Contact( #Mx_ET01 )
      I_Contact( #Selec_E3 )
      I_Contact( #pHsMx_1 )
      I_Contact( #pHsMx_2 )
      I_Contact( #pHsMx_3 )
      I_Contact( #pHsMx_4 )
      Contact( #ConfigFB.NoEntrar_E1 )
   END_RUNG wire#w2
   // the same network as SCL:
   #MA_DepositOK_E1 := ((#Mx_ET10 AND (#Avance_T1 OR #CNT_pHsMx_E1.QD)) OR #Mx_ET11 OR (#Mx_ET01 AND NOT #Selec_E3 AND NOT #pHsMx_1 AND NOT #pHsMx_2 AND NOT #pHsMx_3 AND NOT #pHsMx_4 AND #ConfigFB.NoEntrar_E1)) AND #Pos_TROK AND #Pos_TPOK AND #EstadoZona.Marcha_CBx AND NOT #EstadoVI.Error_Mx AND NOT #Error_Tx;
END_REGION

REGION Network 94: INTERLOCK FSS - Permiso de DesCarga E1 - MA_DepositOK_E3
   RUNG wire#powerrail
      Contact( #Mx_ET30 )
      wire#w1
      Contact( #Avance_T1 )
      wire#w2
      Contact( #Pos_TROK )
      Contact( #Pos_TPOK )
      Contact( #EstadoZona.Marcha_CBx )
      I_Contact( #EstadoVI.Error_Mx )
      I_Contact( #Error_Tx )
      Coil( #MA_DepositOK_E3 )
   END_RUNG
   RUNG wire#w1
      Contact( #CNT_pHsMx_E3.QD )
   END_RUNG wire#w2
   RUNG wire#powerrail
      Contact( #Mx_ET31 )
   END_RUNG wire#w2
   RUNG wire#powerrail
      Contact( #Mx_ET01 )
      I_Contact( #Selec_E1 )
      I_Contact( #pHsMx_1 )
      I_Contact( #pHsMx_2 )
      I_Contact( #pHsMx_3 )
      I_Contact( #pHsMx_4 )
      Contact( #ConfigFB.NoEntrar_E3 )
   END_RUNG wire#w2
   // the same network as SCL:
   #MA_DepositOK_E3 := ((#Mx_ET30 AND (#Avance_T1 OR #CNT_pHsMx_E3.QD)) OR #Mx_ET31 OR (#Mx_ET01 AND NOT #Selec_E1 AND NOT #pHsMx_1 AND NOT #pHsMx_2 AND NOT #pHsMx_3 AND NOT #pHsMx_4 AND #ConfigFB.NoEntrar_E3)) AND #Pos_TROK AND #Pos_TPOK AND #EstadoZona.Marcha_CBx AND NOT #EstadoVI.Error_Mx AND NOT #Error_Tx;
END_REGION

REGION Network 95: VARIABLES AUXILIARES - Aviso de Salida - AVTF_Mx_MSig - Grande y Pequeña
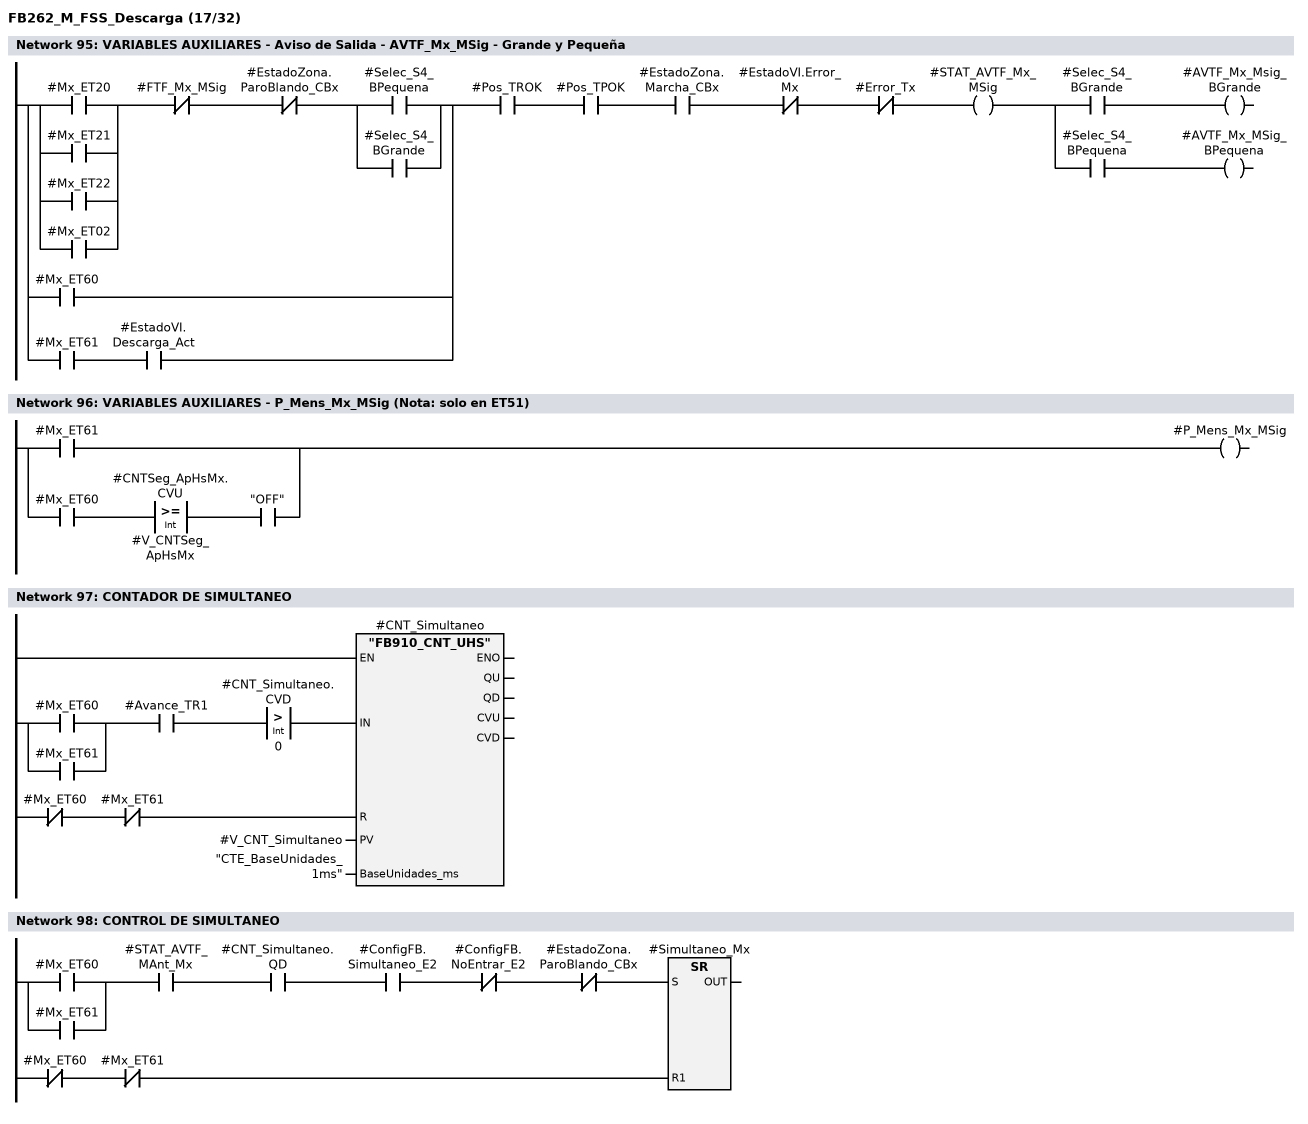
   RUNG wire#powerrail
      Contact( #Mx_ET20 )
      wire#w1
      I_Contact( #FTF_Mx_MSig )
      I_Contact( #EstadoZona.ParoBlando_CBx )
      wire#w2
      Contact( #Selec_S4_BPequena )
      wire#w3
      Contact( #Pos_TROK )
      Contact( #Pos_TPOK )
      Contact( #EstadoZona.Marcha_CBx )
      I_Contact( #EstadoVI.Error_Mx )
      I_Contact( #Error_Tx )
      Coil( #STAT_AVTF_Mx_MSig )
      wire#w4
      Contact( #Selec_S4_BGrande )
      Coil( #AVTF_Mx_Msig_BGrande )
   END_RUNG
   RUNG wire#powerrail
      Contact( #Mx_ET21 )
   END_RUNG wire#w1
   RUNG wire#powerrail
      Contact( #Mx_ET22 )
   END_RUNG wire#w1
   RUNG wire#powerrail
      Contact( #Mx_ET02 )
   END_RUNG wire#w1
   RUNG wire#w2
      Contact( #Selec_S4_BGrande )
   END_RUNG wire#w3
   RUNG wire#powerrail
      Contact( #Mx_ET60 )
   END_RUNG wire#w3
   RUNG wire#powerrail
      Contact( #Mx_ET61 )
      Contact( #EstadoVI.Descarga_Act )
   END_RUNG wire#w3
   RUNG wire#w4
      Contact( #Selec_S4_BPequena )
      Coil( #AVTF_Mx_MSig_BPequena )
   END_RUNG
   // the same network as SCL:
   #STAT_AVTF_Mx_MSig := (((#Mx_ET20 OR #Mx_ET21 OR #Mx_ET22 OR #Mx_ET02) AND NOT #FTF_Mx_MSig AND NOT #EstadoZona.ParoBlando_CBx AND (#Selec_S4_BPequena OR #Selec_S4_BGrande)) OR #Mx_ET60 OR (#Mx_ET61 AND #EstadoVI.Descarga_Act)) AND #Pos_TROK AND #Pos_TPOK AND #EstadoZona.Marcha_CBx AND NOT #EstadoVI.Error_Mx AND NOT #Error_Tx;
   #AVTF_Mx_Msig_BGrande := #STAT_AVTF_Mx_MSig AND #Selec_S4_BGrande;
   #AVTF_Mx_MSig_BPequena := #STAT_AVTF_Mx_MSig AND #Selec_S4_BPequena;
END_REGION

REGION Network 96: VARIABLES AUXILIARES - P_Mens_Mx_MSig (Nota: solo en ET51)
   RUNG wire#powerrail
      Contact( #Mx_ET61 )
      wire#w1
      Coil( #P_Mens_Mx_MSig )
   END_RUNG
   RUNG wire#powerrail
      Contact( #Mx_ET60 )
      { S7_Templates := "SrcType := Int" } GE_Contact(in1 := #CNTSeg_ApHsMx.CVU, in2 := #V_CNTSeg_ApHsMx)
      Contact( "OFF" )
   END_RUNG wire#w1
   // the same network as SCL:
   #P_Mens_Mx_MSig := #Mx_ET61 OR (#Mx_ET60 AND (#CNTSeg_ApHsMx.CVU >= #V_CNTSeg_ApHsMx) AND "OFF");
END_REGION

REGION Network 97: CONTADOR DE SIMULTANEO
   RUNG wire#powerrail
      #CNT_Simultaneo(IN := wire#w2, R := wire#w3, PV := #V_CNT_Simultaneo, BaseUnidades_ms := "CTE_BaseUnidades_1ms", QU =>, QD =>, CVU =>, CVD =>)
   END_RUNG
   RUNG wire#powerrail
      Contact( #Mx_ET60 )
      wire#w1
      Contact( #Avance_TR1 )
      { S7_Templates := "SrcType := Int" } GT_Contact(in1 := #CNT_Simultaneo.CVD, in2 := 0)
   END_RUNG wire#w2
   RUNG wire#powerrail
      Contact( #Mx_ET61 )
   END_RUNG wire#w1
   RUNG wire#powerrail
      I_Contact( #Mx_ET60 )
      I_Contact( #Mx_ET61 )
   END_RUNG wire#w3
   // the same network as SCL:
   #CNT_Simultaneo(IN := (#Mx_ET60 OR #Mx_ET61) AND #Avance_TR1 AND (#CNT_Simultaneo.CVD > 0),   // "FB910_CNT_UHS"
                   R := NOT #Mx_ET60 AND NOT #Mx_ET61,
                   PV := #V_CNT_Simultaneo,
                   BaseUnidades_ms := "CTE_BaseUnidades_1ms");
END_REGION

REGION Network 98: CONTROL DE SIMULTANEO
   RUNG wire#powerrail
      Contact( #Mx_ET60 )
      wire#w1
      Contact( #STAT_AVTF_MAnt_Mx )
      Contact( #CNT_Simultaneo.QD )
      Contact( #ConfigFB.Simultaneo_E2 )
      I_Contact( #ConfigFB.NoEntrar_E2 )
      I_Contact( #EstadoZona.ParoBlando_CBx )
      S_SR(operand := #Simultaneo_Mx, r1 := wire#w2)
   END_RUNG
   RUNG wire#powerrail
      Contact( #Mx_ET61 )
   END_RUNG wire#w1
   RUNG wire#powerrail
      I_Contact( #Mx_ET60 )
      I_Contact( #Mx_ET61 )
   END_RUNG wire#w2
   // the same network as SCL:
   IF (#Mx_ET60 OR #Mx_ET61) AND #STAT_AVTF_MAnt_Mx AND #CNT_Simultaneo.QD AND #ConfigFB.Simultaneo_E2 AND NOT #ConfigFB.NoEntrar_E2 AND NOT #EstadoZona.ParoBlando_CBx THEN
       #Simultaneo_Mx := TRUE;   // SR flip-flop
   END_IF;
   IF NOT #Mx_ET60 AND NOT #Mx_ET61 THEN #Simultaneo_Mx := FALSE; END_IF;
END_REGION

REGION Network 99: MENSAJES - PRESENCIA
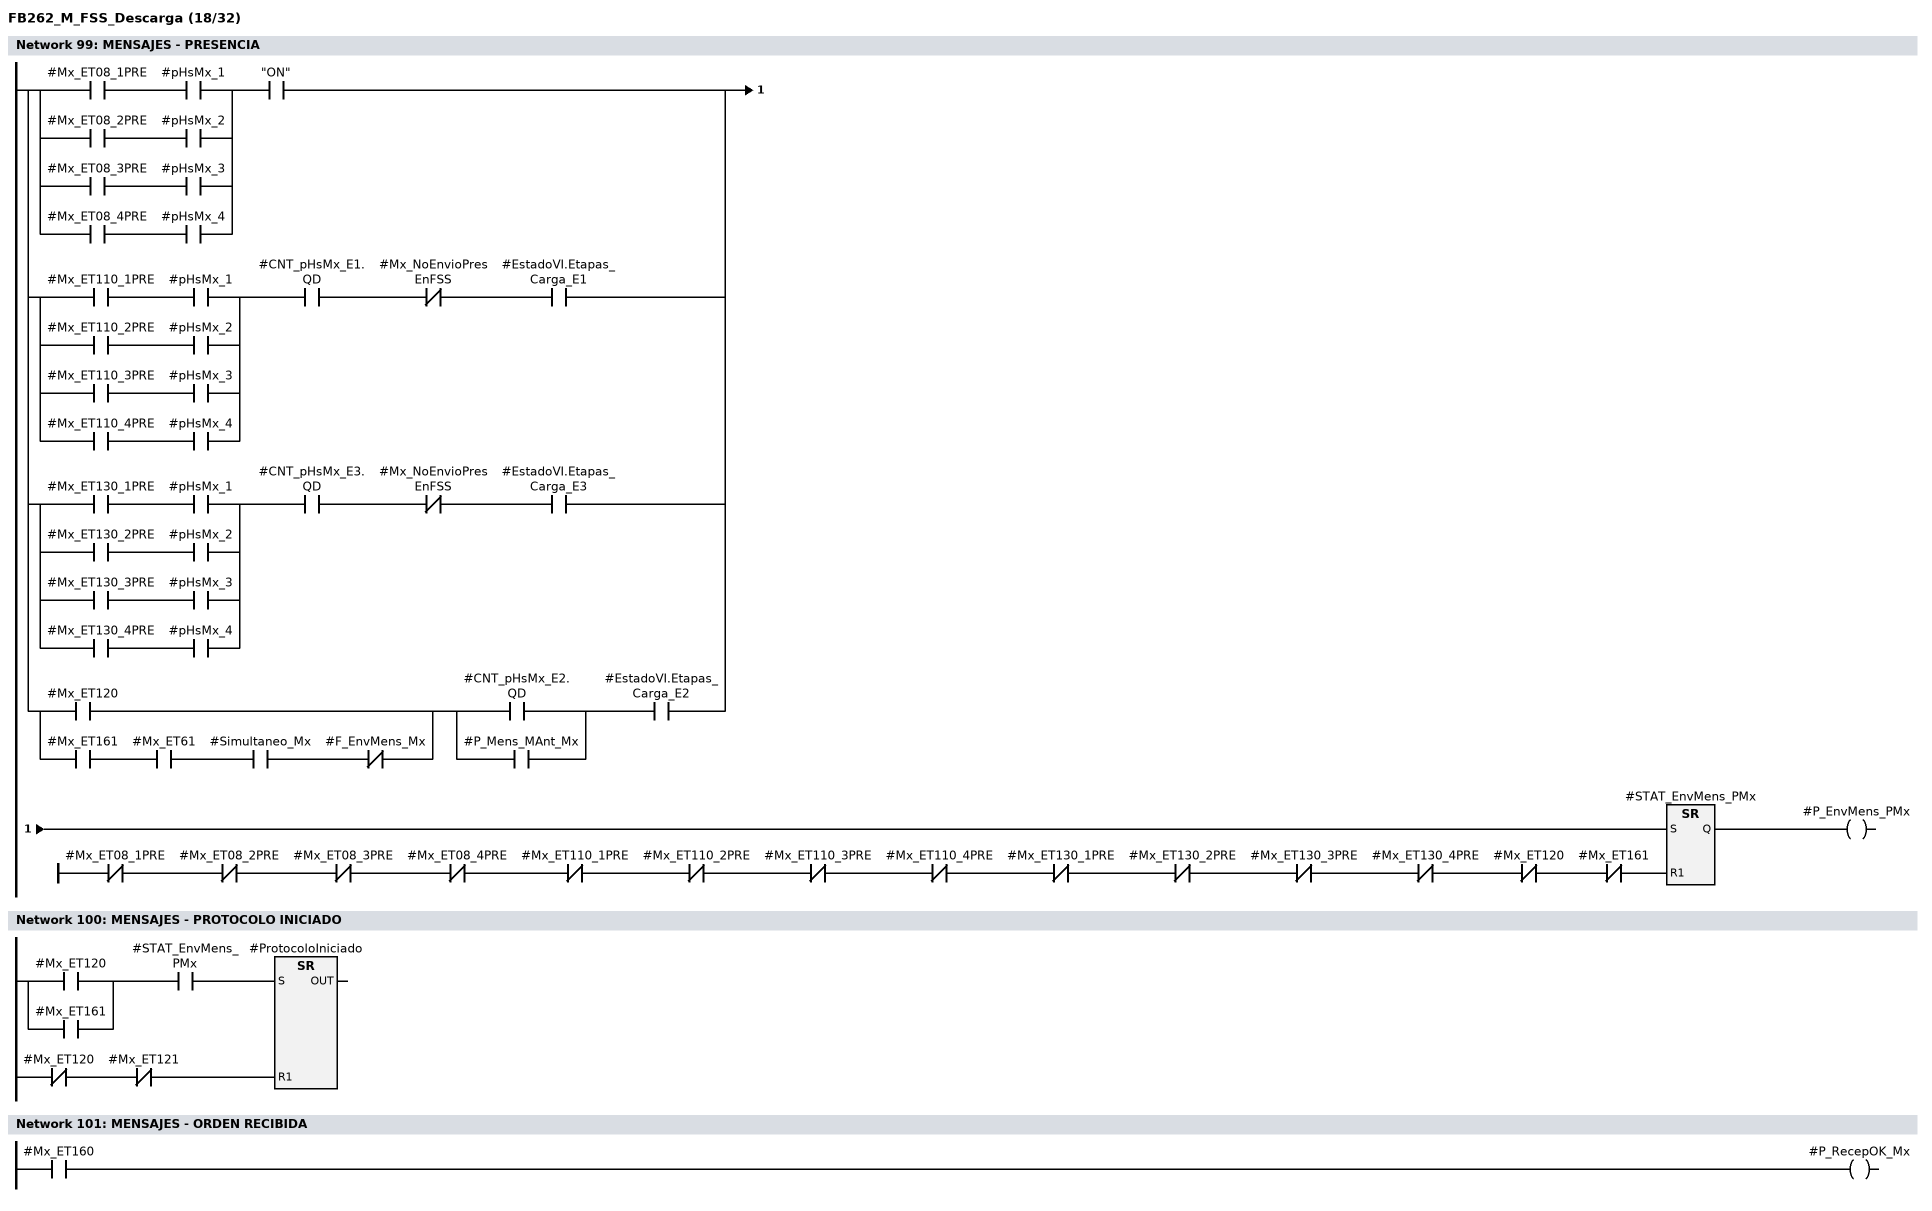
   RUNG wire#powerrail
      Contact( #Mx_ET08_1PRE )
      Contact( #pHsMx_1 )
      wire#w1
      Contact( "ON" )
      wire#w2
      S_SR(operand := #STAT_EnvMens_PMx, r1 := wire#w7)
      Coil( #P_EnvMens_PMx )
   END_RUNG
   RUNG wire#powerrail
      Contact( #Mx_ET08_2PRE )
      Contact( #pHsMx_2 )
   END_RUNG wire#w1
   RUNG wire#powerrail
      Contact( #Mx_ET08_3PRE )
      Contact( #pHsMx_3 )
   END_RUNG wire#w1
   RUNG wire#powerrail
      Contact( #Mx_ET08_4PRE )
      Contact( #pHsMx_4 )
   END_RUNG wire#w1
   RUNG wire#powerrail
      Contact( #Mx_ET110_1PRE )
      Contact( #pHsMx_1 )
      wire#w3
      Contact( #CNT_pHsMx_E1.QD )
      I_Contact( #Mx_NoEnvioPresEnFSS )
      Contact( #EstadoVI.Etapas_Carga_E1 )
   END_RUNG wire#w2
   RUNG wire#powerrail
      Contact( #Mx_ET110_2PRE )
      Contact( #pHsMx_2 )
   END_RUNG wire#w3
   RUNG wire#powerrail
      Contact( #Mx_ET110_3PRE )
      Contact( #pHsMx_3 )
   END_RUNG wire#w3
   RUNG wire#powerrail
      Contact( #Mx_ET110_4PRE )
      Contact( #pHsMx_4 )
   END_RUNG wire#w3
   RUNG wire#powerrail
      Contact( #Mx_ET130_1PRE )
      Contact( #pHsMx_1 )
      wire#w4
      Contact( #CNT_pHsMx_E3.QD )
      I_Contact( #Mx_NoEnvioPresEnFSS )
      Contact( #EstadoVI.Etapas_Carga_E3 )
   END_RUNG wire#w2
   RUNG wire#powerrail
      Contact( #Mx_ET130_2PRE )
      Contact( #pHsMx_2 )
   END_RUNG wire#w4
   RUNG wire#powerrail
      Contact( #Mx_ET130_3PRE )
      Contact( #pHsMx_3 )
   END_RUNG wire#w4
   RUNG wire#powerrail
      Contact( #Mx_ET130_4PRE )
      Contact( #pHsMx_4 )
   END_RUNG wire#w4
   RUNG wire#powerrail
      Contact( #Mx_ET120 )
      wire#w5
      Contact( #CNT_pHsMx_E2.QD )
      wire#w6
      Contact( #EstadoVI.Etapas_Carga_E2 )
   END_RUNG wire#w2
   RUNG wire#powerrail
      Contact( #Mx_ET161 )
      Contact( #Mx_ET61 )
      Contact( #Simultaneo_Mx )
      I_Contact( #F_EnvMens_Mx )
   END_RUNG wire#w5
   RUNG wire#w5
      Contact( #P_Mens_MAnt_Mx )
   END_RUNG wire#w6
   RUNG wire#powerrail
      I_Contact( #Mx_ET08_1PRE )
      I_Contact( #Mx_ET08_2PRE )
      I_Contact( #Mx_ET08_3PRE )
      I_Contact( #Mx_ET08_4PRE )
      I_Contact( #Mx_ET110_1PRE )
      I_Contact( #Mx_ET110_2PRE )
      I_Contact( #Mx_ET110_3PRE )
      I_Contact( #Mx_ET110_4PRE )
      I_Contact( #Mx_ET130_1PRE )
      I_Contact( #Mx_ET130_2PRE )
      I_Contact( #Mx_ET130_3PRE )
      I_Contact( #Mx_ET130_4PRE )
      I_Contact( #Mx_ET120 )
      I_Contact( #Mx_ET161 )
   END_RUNG wire#w7
   // the same network as SCL:
   IF (((#Mx_ET08_1PRE AND #pHsMx_1) OR (#Mx_ET08_2PRE AND #pHsMx_2) OR (#Mx_ET08_3PRE AND #pHsMx_3) OR (#Mx_ET08_4PRE AND #pHsMx_4)) AND "ON") OR (((#Mx_ET110_1PRE AND #pHsMx_1) OR (#Mx_ET110_2PRE AND #pHsMx_2) OR (#Mx_ET110_3PRE AND #pHsMx_3) OR (#Mx_ET110_4PRE AND #pHsMx_4)) AND #CNT_pHsMx_E1.QD AND NOT #Mx_NoEnvioPresEnFSS AND #EstadoVI.Etapas_Carga_E1) OR (((#Mx_ET130_1PRE AND #pHsMx_1) OR (#Mx_ET130_2PRE AND #pHsMx_2) OR (#Mx_ET130_3PRE AND #pHsMx_3) OR (#Mx_ET130_4PRE AND #pHsMx_4)) AND #CNT_pHsMx_E3.QD AND NOT #Mx_NoEnvioPresEnFSS AND #EstadoVI.Etapas_Carga_E3) OR ((#Mx_ET120 OR (#Mx_ET161 AND #Mx_ET61 AND #Simultaneo_Mx AND NOT #F_EnvMens_Mx)) AND (#CNT_pHsMx_E2.QD OR #P_Mens_MAnt_Mx) AND #EstadoVI.Etapas_Carga_E2) THEN
       #STAT_EnvMens_PMx := TRUE;   // SR flip-flop
   END_IF;
   IF NOT #Mx_ET08_1PRE AND NOT #Mx_ET08_2PRE AND NOT #Mx_ET08_3PRE AND NOT #Mx_ET08_4PRE AND NOT #Mx_ET110_1PRE AND NOT #Mx_ET110_2PRE AND NOT #Mx_ET110_3PRE AND NOT #Mx_ET110_4PRE AND NOT #Mx_ET130_1PRE AND NOT #Mx_ET130_2PRE AND NOT #Mx_ET130_3PRE AND NOT #Mx_ET130_4PRE AND NOT #Mx_ET120 AND NOT #Mx_ET161 THEN
       #STAT_EnvMens_PMx := FALSE;
   END_IF;
   #P_EnvMens_PMx := #STAT_EnvMens_PMx;
END_REGION

REGION Network 100: MENSAJES - PROTOCOLO INICIADO
   RUNG wire#powerrail
      Contact( #Mx_ET120 )
      wire#w1
      Contact( #STAT_EnvMens_PMx )
      S_SR(operand := #ProtocoloIniciado, r1 := wire#w2)
   END_RUNG
   RUNG wire#powerrail
      Contact( #Mx_ET161 )
   END_RUNG wire#w1
   RUNG wire#powerrail
      I_Contact( #Mx_ET120 )
      I_Contact( #Mx_ET121 )
   END_RUNG wire#w2
   // the same network as SCL:
   IF (#Mx_ET120 OR #Mx_ET161) AND #STAT_EnvMens_PMx THEN
       #ProtocoloIniciado := TRUE;   // SR flip-flop
   END_IF;
   IF NOT #Mx_ET120 AND NOT #Mx_ET121 THEN #ProtocoloIniciado := FALSE; END_IF;
END_REGION

REGION Network 101: MENSAJES - ORDEN RECIBIDA
   RUNG wire#powerrail
      Contact( #Mx_ET160 )
      Coil( #P_RecepOK_Mx )
   END_RUNG
   // the same network as SCL:
   #P_RecepOK_Mx := #Mx_ET160;
END_REGION

REGION Network 102: VARIABLES INTERNAS - AVANCE DE CARGA >> DESDE FSS
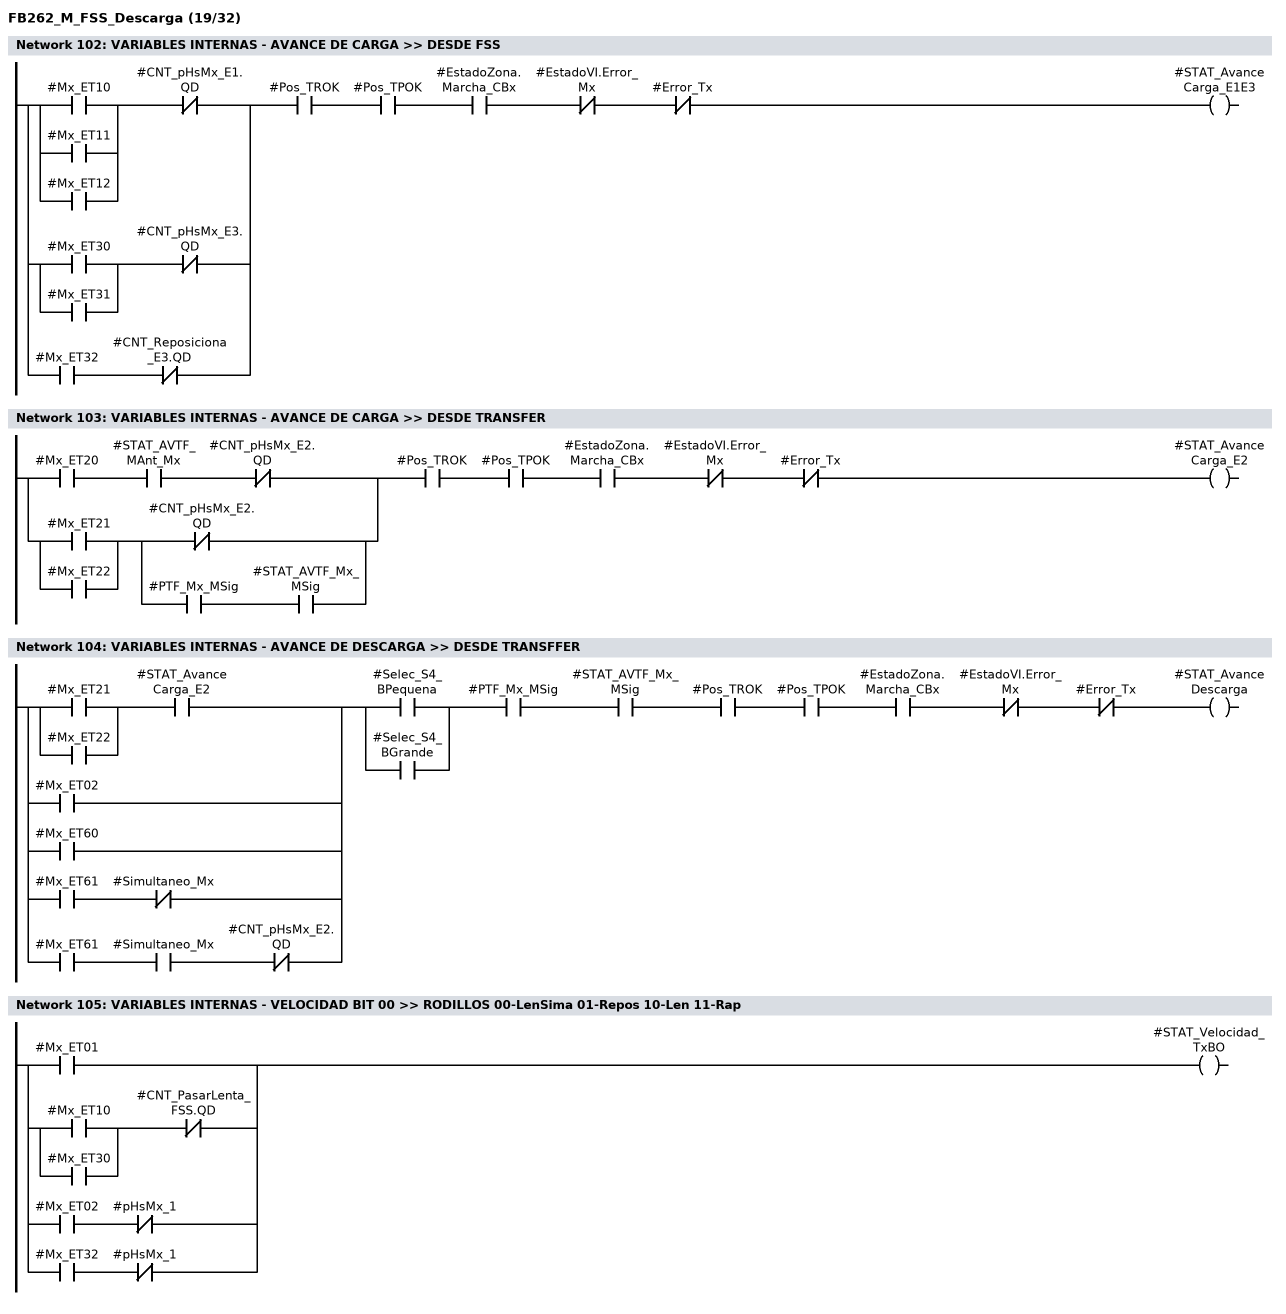
   RUNG wire#powerrail
      Contact( #Mx_ET10 )
      wire#w1
      I_Contact( #CNT_pHsMx_E1.QD )
      wire#w2
      Contact( #Pos_TROK )
      Contact( #Pos_TPOK )
      Contact( #EstadoZona.Marcha_CBx )
      I_Contact( #EstadoVI.Error_Mx )
      I_Contact( #Error_Tx )
      Coil( #STAT_AvanceCarga_E1E3 )
   END_RUNG
   RUNG wire#powerrail
      Contact( #Mx_ET11 )
   END_RUNG wire#w1
   RUNG wire#powerrail
      Contact( #Mx_ET12 )
   END_RUNG wire#w1
   RUNG wire#powerrail
      Contact( #Mx_ET30 )
      wire#w3
      I_Contact( #CNT_pHsMx_E3.QD )
   END_RUNG wire#w2
   RUNG wire#powerrail
      Contact( #Mx_ET31 )
   END_RUNG wire#w3
   RUNG wire#powerrail
      Contact( #Mx_ET32 )
      I_Contact( #CNT_Reposiciona_E3.QD )
   END_RUNG wire#w2
   // the same network as SCL:
   #STAT_AvanceCarga_E1E3 := (((#Mx_ET10 OR #Mx_ET11 OR #Mx_ET12) AND NOT #CNT_pHsMx_E1.QD) OR ((#Mx_ET30 OR #Mx_ET31) AND NOT #CNT_pHsMx_E3.QD) OR (#Mx_ET32 AND NOT #CNT_Reposiciona_E3.QD)) AND #Pos_TROK AND #Pos_TPOK AND #EstadoZona.Marcha_CBx AND NOT #EstadoVI.Error_Mx AND NOT #Error_Tx;
END_REGION

REGION Network 103: VARIABLES INTERNAS - AVANCE DE CARGA >> DESDE TRANSFER
   RUNG wire#powerrail
      Contact( #Mx_ET20 )
      Contact( #STAT_AVTF_MAnt_Mx )
      I_Contact( #CNT_pHsMx_E2.QD )
      wire#w1
      Contact( #Pos_TROK )
      Contact( #Pos_TPOK )
      Contact( #EstadoZona.Marcha_CBx )
      I_Contact( #EstadoVI.Error_Mx )
      I_Contact( #Error_Tx )
      Coil( #STAT_AvanceCarga_E2 )
   END_RUNG
   RUNG wire#powerrail
      Contact( #Mx_ET21 )
      wire#w2
      I_Contact( #CNT_pHsMx_E2.QD )
   END_RUNG wire#w1
   RUNG wire#powerrail
      Contact( #Mx_ET22 )
   END_RUNG wire#w2
   RUNG wire#w2
      Contact( #PTF_Mx_MSig )
      Contact( #STAT_AVTF_Mx_MSig )
   END_RUNG wire#w1
   // the same network as SCL:
   #STAT_AvanceCarga_E2 := ((#Mx_ET20 AND #STAT_AVTF_MAnt_Mx AND NOT #CNT_pHsMx_E2.QD) OR ((#Mx_ET21 OR #Mx_ET22) AND (NOT #CNT_pHsMx_E2.QD OR (#PTF_Mx_MSig AND #STAT_AVTF_Mx_MSig)))) AND #Pos_TROK AND #Pos_TPOK AND #EstadoZona.Marcha_CBx AND NOT #EstadoVI.Error_Mx AND NOT #Error_Tx;
END_REGION

REGION Network 104: VARIABLES INTERNAS - AVANCE DE DESCARGA >> DESDE TRANSFFER
   RUNG wire#powerrail
      Contact( #Mx_ET21 )
      wire#w1
      Contact( #STAT_AvanceCarga_E2 )
      wire#w2
      Contact( #Selec_S4_BPequena )
      wire#w3
      Contact( #PTF_Mx_MSig )
      Contact( #STAT_AVTF_Mx_MSig )
      Contact( #Pos_TROK )
      Contact( #Pos_TPOK )
      Contact( #EstadoZona.Marcha_CBx )
      I_Contact( #EstadoVI.Error_Mx )
      I_Contact( #Error_Tx )
      Coil( #STAT_AvanceDescarga )
   END_RUNG
   RUNG wire#powerrail
      Contact( #Mx_ET22 )
   END_RUNG wire#w1
   RUNG wire#powerrail
      Contact( #Mx_ET02 )
   END_RUNG wire#w2
   RUNG wire#powerrail
      Contact( #Mx_ET60 )
   END_RUNG wire#w2
   RUNG wire#powerrail
      Contact( #Mx_ET61 )
      I_Contact( #Simultaneo_Mx )
   END_RUNG wire#w2
   RUNG wire#powerrail
      Contact( #Mx_ET61 )
      Contact( #Simultaneo_Mx )
      I_Contact( #CNT_pHsMx_E2.QD )
   END_RUNG wire#w2
   RUNG wire#w2
      Contact( #Selec_S4_BGrande )
   END_RUNG wire#w3
   // the same network as SCL:
   #STAT_AvanceDescarga := (((#Mx_ET21 OR #Mx_ET22) AND #STAT_AvanceCarga_E2) OR #Mx_ET02 OR #Mx_ET60 OR (#Mx_ET61 AND NOT #Simultaneo_Mx) OR (#Mx_ET61 AND #Simultaneo_Mx AND NOT #CNT_pHsMx_E2.QD)) AND (#Selec_S4_BPequena OR #Selec_S4_BGrande) AND #PTF_Mx_MSig AND #STAT_AVTF_Mx_MSig AND #Pos_TROK AND #Pos_TPOK AND #EstadoZona.Marcha_CBx AND NOT #EstadoVI.Error_Mx AND NOT #Error_Tx;
END_REGION

REGION Network 105: VARIABLES INTERNAS - VELOCIDAD BIT 00 >> RODILLOS 00-LenSima 01-Repos 10-Len 11-Rap
   RUNG wire#powerrail
      Contact( #Mx_ET01 )
      wire#w1
      Coil( #STAT_Velocidad_TxBO )
   END_RUNG
   RUNG wire#powerrail
      Contact( #Mx_ET10 )
      wire#w2
      I_Contact( #CNT_PasarLenta_FSS.QD )
   END_RUNG wire#w1
   RUNG wire#powerrail
      Contact( #Mx_ET30 )
   END_RUNG wire#w2
   RUNG wire#powerrail
      Contact( #Mx_ET02 )
      I_Contact( #pHsMx_1 )
   END_RUNG wire#w1
   RUNG wire#powerrail
      Contact( #Mx_ET32 )
      I_Contact( #pHsMx_1 )
   END_RUNG wire#w1
   // the same network as SCL:
   #STAT_Velocidad_TxBO := #Mx_ET01 OR ((#Mx_ET10 OR #Mx_ET30) AND NOT #CNT_PasarLenta_FSS.QD) OR (#Mx_ET02 AND NOT #pHsMx_1) OR (#Mx_ET32 AND NOT #pHsMx_1);
END_REGION

REGION Network 106: VARIABLES INTERNAS - VELOCIDAD BIT 01 >> RODILLOS 00-LenSima 01-Repos 10-Len 11-Rap
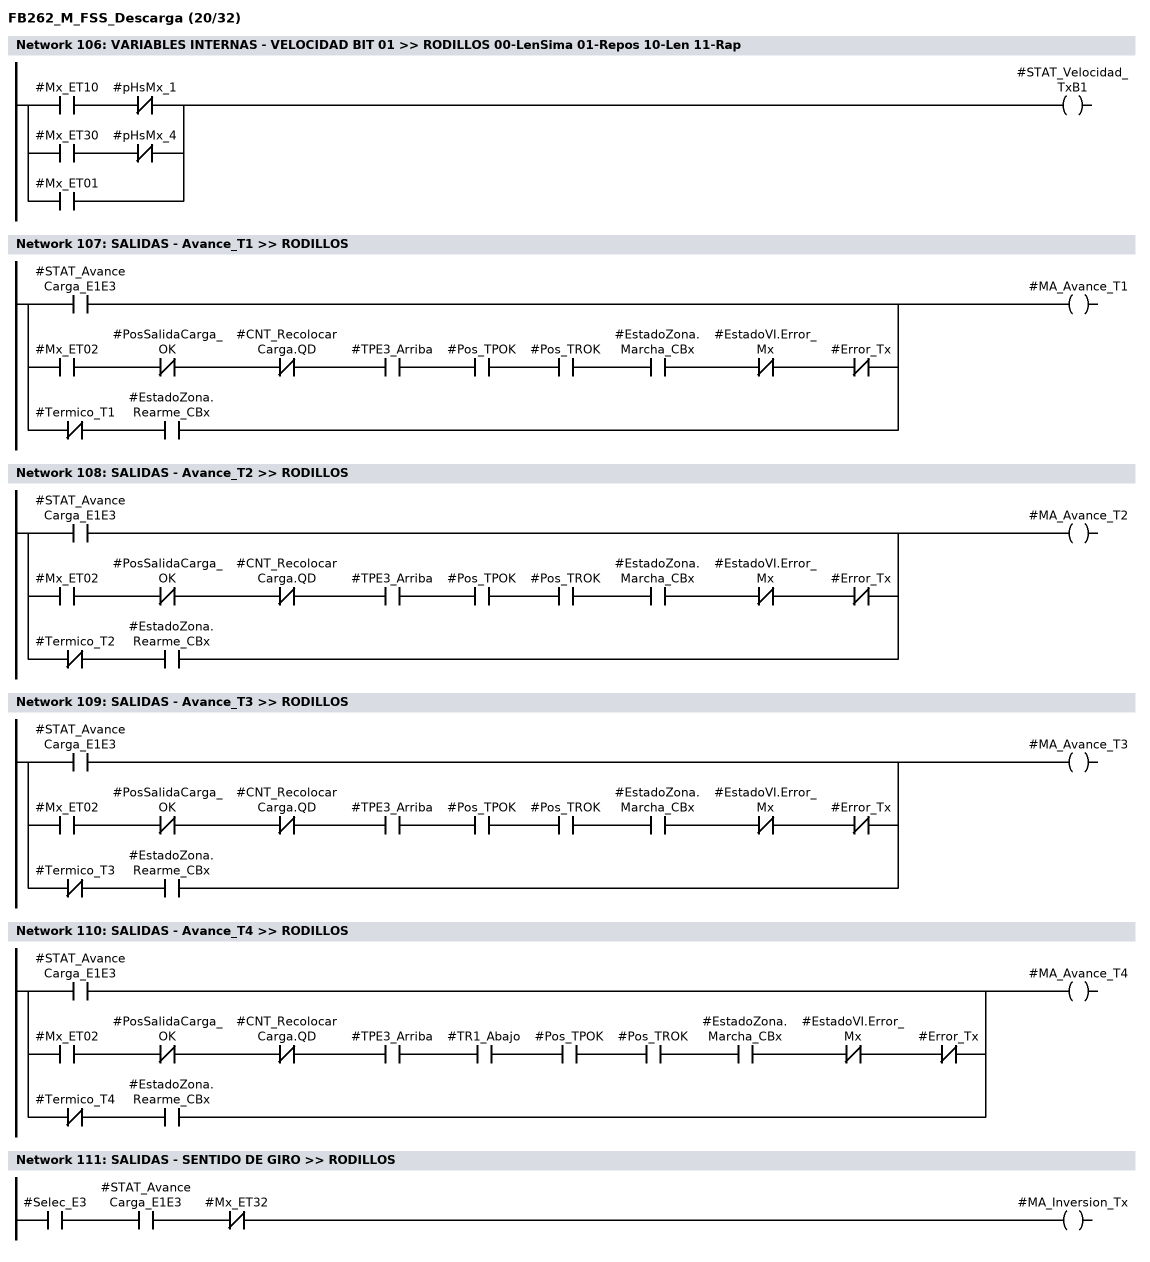
   RUNG wire#powerrail
      Contact( #Mx_ET10 )
      I_Contact( #pHsMx_1 )
      wire#w1
      Coil( #STAT_Velocidad_TxB1 )
   END_RUNG
   RUNG wire#powerrail
      Contact( #Mx_ET30 )
      I_Contact( #pHsMx_4 )
   END_RUNG wire#w1
   RUNG wire#powerrail
      Contact( #Mx_ET01 )
   END_RUNG wire#w1
   // the same network as SCL:
   #STAT_Velocidad_TxB1 := (#Mx_ET10 AND NOT #pHsMx_1) OR (#Mx_ET30 AND NOT #pHsMx_4) OR #Mx_ET01;
END_REGION

REGION Network 107: SALIDAS - Avance_T1 >> RODILLOS
   RUNG wire#powerrail
      Contact( #STAT_AvanceCarga_E1E3 )
      wire#w1
      Coil( #MA_Avance_T1 )
   END_RUNG
   RUNG wire#powerrail
      Contact( #Mx_ET02 )
      I_Contact( #PosSalidaCarga_OK )
      I_Contact( #CNT_RecolocarCarga.QD )
      Contact( #TPE3_Arriba )
      Contact( #Pos_TPOK )
      Contact( #Pos_TROK )
      Contact( #EstadoZona.Marcha_CBx )
      I_Contact( #EstadoVI.Error_Mx )
      I_Contact( #Error_Tx )
   END_RUNG wire#w1
   RUNG wire#powerrail
      I_Contact( #Termico_T1 )
      Contact( #EstadoZona.Rearme_CBx )
   END_RUNG wire#w1
   // the same network as SCL:
   #MA_Avance_T1 := #STAT_AvanceCarga_E1E3 OR (#Mx_ET02 AND NOT #PosSalidaCarga_OK AND NOT #CNT_RecolocarCarga.QD AND #TPE3_Arriba AND #Pos_TPOK AND #Pos_TROK AND #EstadoZona.Marcha_CBx AND NOT #EstadoVI.Error_Mx AND NOT #Error_Tx) OR (NOT #Termico_T1 AND #EstadoZona.Rearme_CBx);
END_REGION

REGION Network 108: SALIDAS - Avance_T2 >> RODILLOS
   RUNG wire#powerrail
      Contact( #STAT_AvanceCarga_E1E3 )
      wire#w1
      Coil( #MA_Avance_T2 )
   END_RUNG
   RUNG wire#powerrail
      Contact( #Mx_ET02 )
      I_Contact( #PosSalidaCarga_OK )
      I_Contact( #CNT_RecolocarCarga.QD )
      Contact( #TPE3_Arriba )
      Contact( #Pos_TPOK )
      Contact( #Pos_TROK )
      Contact( #EstadoZona.Marcha_CBx )
      I_Contact( #EstadoVI.Error_Mx )
      I_Contact( #Error_Tx )
   END_RUNG wire#w1
   RUNG wire#powerrail
      I_Contact( #Termico_T2 )
      Contact( #EstadoZona.Rearme_CBx )
   END_RUNG wire#w1
   // the same network as SCL:
   #MA_Avance_T2 := #STAT_AvanceCarga_E1E3 OR (#Mx_ET02 AND NOT #PosSalidaCarga_OK AND NOT #CNT_RecolocarCarga.QD AND #TPE3_Arriba AND #Pos_TPOK AND #Pos_TROK AND #EstadoZona.Marcha_CBx AND NOT #EstadoVI.Error_Mx AND NOT #Error_Tx) OR (NOT #Termico_T2 AND #EstadoZona.Rearme_CBx);
END_REGION

REGION Network 109: SALIDAS - Avance_T3 >> RODILLOS
   RUNG wire#powerrail
      Contact( #STAT_AvanceCarga_E1E3 )
      wire#w1
      Coil( #MA_Avance_T3 )
   END_RUNG
   RUNG wire#powerrail
      Contact( #Mx_ET02 )
      I_Contact( #PosSalidaCarga_OK )
      I_Contact( #CNT_RecolocarCarga.QD )
      Contact( #TPE3_Arriba )
      Contact( #Pos_TPOK )
      Contact( #Pos_TROK )
      Contact( #EstadoZona.Marcha_CBx )
      I_Contact( #EstadoVI.Error_Mx )
      I_Contact( #Error_Tx )
   END_RUNG wire#w1
   RUNG wire#powerrail
      I_Contact( #Termico_T3 )
      Contact( #EstadoZona.Rearme_CBx )
   END_RUNG wire#w1
   // the same network as SCL:
   #MA_Avance_T3 := #STAT_AvanceCarga_E1E3 OR (#Mx_ET02 AND NOT #PosSalidaCarga_OK AND NOT #CNT_RecolocarCarga.QD AND #TPE3_Arriba AND #Pos_TPOK AND #Pos_TROK AND #EstadoZona.Marcha_CBx AND NOT #EstadoVI.Error_Mx AND NOT #Error_Tx) OR (NOT #Termico_T3 AND #EstadoZona.Rearme_CBx);
END_REGION

REGION Network 110: SALIDAS - Avance_T4 >> RODILLOS
   RUNG wire#powerrail
      Contact( #STAT_AvanceCarga_E1E3 )
      wire#w1
      Coil( #MA_Avance_T4 )
   END_RUNG
   RUNG wire#powerrail
      Contact( #Mx_ET02 )
      I_Contact( #PosSalidaCarga_OK )
      I_Contact( #CNT_RecolocarCarga.QD )
      Contact( #TPE3_Arriba )
      Contact( #TR1_Abajo )
      Contact( #Pos_TPOK )
      Contact( #Pos_TROK )
      Contact( #EstadoZona.Marcha_CBx )
      I_Contact( #EstadoVI.Error_Mx )
      I_Contact( #Error_Tx )
   END_RUNG wire#w1
   RUNG wire#powerrail
      I_Contact( #Termico_T4 )
      Contact( #EstadoZona.Rearme_CBx )
   END_RUNG wire#w1
   // the same network as SCL:
   #MA_Avance_T4 := #STAT_AvanceCarga_E1E3 OR (#Mx_ET02 AND NOT #PosSalidaCarga_OK AND NOT #CNT_RecolocarCarga.QD AND #TPE3_Arriba AND #TR1_Abajo AND #Pos_TPOK AND #Pos_TROK AND #EstadoZona.Marcha_CBx AND NOT #EstadoVI.Error_Mx AND NOT #Error_Tx) OR (NOT #Termico_T4 AND #EstadoZona.Rearme_CBx);
END_REGION

REGION Network 111: SALIDAS - SENTIDO DE GIRO >> RODILLOS
   RUNG wire#powerrail
      Contact( #Selec_E3 )
      Contact( #STAT_AvanceCarga_E1E3 )
      I_Contact( #Mx_ET32 )
      Coil( #MA_Inversion_Tx )
   END_RUNG
   // the same network as SCL:
   #MA_Inversion_Tx := #Selec_E3 AND #STAT_AvanceCarga_E1E3 AND NOT #Mx_ET32;
END_REGION

